(* CODESYS project Trike_PLC_Project.project
   Company: Schneider Electric
   Title: Compact / CANopen / HMI Controller SCU
   Description: ********Disclaimer Of Warranty********
      THE INFORMATION CONTAINED HEREIN IS PROVIDED "AS IS" WITHOUT WARRANTIES OF ANY KIND, EITHER EXPRESS OR IMPLIED, INCLUDING WITHOUT LIMITATION, ALL IMPLIED WARRANTIES OF MERCHANTABILITY, FITNESS FOR A PARTICULAR PURPOSE, NON-INFRINGEMENT OR OTHER VIOLATION OF RIGHTS. SCHNEIDER ELECTRIC DOES NOT WARRANT OR MAKE ANY REPRESENTATIONS REGARDING THE USE, VALIDITY, ACCURACY, OR RELIABILITY OF, OR THE RESULTS OF THE USE OF, OR OTHERWISE, RESPECTING THE MATERIALS, SPECIFICATIONS, CHARACTERISTICS OR OTHER INFORMATION SPECIFIED HEREIN. FURTHERMORE, ALL WARRANTIES, CONDITIONS, REPRESENTATIONS, INDEMNITIES AND GUARANTEES WITH RESPECT TO THE ACCURACY, OPERATION, CAPACITY, SPEED, FUNCTIONALITY, QUALIFICATIONS, OR CAPABILITIES OF THE SOFTWARE, SYSTEMS AND SERVICES COMPRISING OR UTILIZED IN THE COURSE OF APPLYING THIS INFORMATION, SPECIFICATIONS, OR MATERIALS, WHETHER EXPRESS OR IMPLIED, ARISING BY LAW, CUSTOM, PRIOR ORAL OR WRITTEN STATEMENTS BY SCHNEIDER ELECTRIC, OR OTHERWISE (INCLUDING, BUT NOT LIMITED TO ANY WARRANTY OF SATISFACTORY QUALITY, MERCHANTABILITY, FITNESS FOR PARTICULAR PURPOSE, TITLE AND NON-INFRINGEMENT) ARE HEREBY EXPRESSLY EXCLUDED AND DISCLAIMED:
      ********Disclaimer Of Liability*********
      UNDER NO CIRCUMSTANCES (INCLUDING NEGLIGENCE OR FORESEEABLE MISUSE) WILL SCHNEIDER ELECTRIC BE LIABLE FOR ANY DIRECT, INDIRECT, SPECIAL, INCIDENTAL, PUNITIVE OR CONSEQUENTIAL DAMAGES (INCLUDING WITHOUT LIMITATION, BUSINESS INTERRUPTION, DELAYS, LOSS OF DATA OR PROFIT) ARISING OUT OF THE APPLICATION OF THE INFORMATION, SPECIFICATIONS, CHARACTERISTICS OR MATERIALS CONTAINED HEREIN EVEN IF SCHNEIDER ELECTRIC HAS BEEN ADVISED OF THE POSSIBILITY OF SUCH DAMAGES.
      ************************************
      The information, program and configuration contained herein are provided as general training on the products concerned, in part, by way of theoretical and/or hypothetical examples.  Only you, the user, can be aware of all the conditions and factors present during setup, operation, and maintenance of your machine and its application; therefore, only you, the user, can determine the automation equipment and the related safeties and interlocks which can be properly used.  When selecting automation and control equipment and related software for a particular application, you must refer to the applicable local and national standards and regulations.
      ************************************
      Copyright © 2017 Schneider Electric. All rights reserved.
   Author: Machine Solutions
   Version: 4.3.0.0

Project tree, tasks and I/O mapping:
  HMISAC : HMISCUxA5, Schneider Electric, order no. HMISCUxA5, version 3.5.3.59
      settings: OpcUa Enable = False
    application Application
      libraries: MachineEnergyDashboard, 4.1.0.0 (Schneider Electric); Toolbox, 2.2.0.0 (Schneider Electric); SM3_Basic, 3.5.3.83 (3S - Smart Software Solutions GmbH)
      task MAST (cyclic, interval 20 ms, priority 15, watchdog 100 ms x 3) calls Preprocessing, Prg_Joystick6000, Prg_MicroCAN, Prg_Dunker_0A, Prg_Dunker_0B, Prg_Dunker_0C, Prg_Dunker_0D, Prg_Speedgoat, AlarmManager, MAIN, OutputMapping, Prg_WriteParameter
      global variables GVL_Retain
      LXM28A_Node03/
        global variables GVL_LXM28A_Node03
        program Prg_LXM28A_Node03 [CFC]: A02_Ctrl_Lexium, A01_GetNodeState
      program Preprocessing [CFC]: A04_DrvCmd_LXM28A_Node04, A05_DrvCmd_LXM32i_Node11, A03_DrvCmd_LXM28A_Node03
      global variables GVL
      global variables GVL_HmiVar
      LXM32i_Node11/
        global variables GVL_LXM32i_Node11
        program Prg_LXM32i_Node11 [CFC]: A02_Ctrl_Lexium, A01_GetNodeState
      program Prg_WriteParameter [ST]: A_WriteParameter_LXM2804, A_WriteParameter_LXM2803
      Symbols
      program MAIN [ST]: A02_CANopen_State, A04_Device_Error_State, A01_CANopen_Slave_State
      program OutputMapping [LD]
      program AlarmManager [CFC]: A06_Alarms_LXM32i_Node11, A05_Alarms_LXM28A_Node04, A01_Alarms_EStop, A04_Alarms_LXM28A_Node03
      global variables GVL_AlarmMsg
      LXM28A_Node04/
        global variables GVL_LXM28A_Node04
        program Prg_LXM28A_Node04 [CFC]: A01_GetNodeState, A02_Ctrl_Lexium
      Joystick_SD6000/
        program Prg_Joystick6000 [CFC]: A01_GetNodeState
        global variables GVL_Joystick6000
      MicroCAN4aiBOX/
        global variables GVL_MicroCAN
        program Prg_MicroCAN [CFC]: A01_GetNodeState
      Dunker_0A/
        global variables GVL_Dunker_0A
        program Prg_Dunker_0A [CFC]: A01_GetNodeState, A02_Ctrl_Dunker_0A
      Dunker_0B/
        global variables GVL_Dunker_0B
        program Prg_Dunker_0B [CFC]: A01_GetNodeState
      Dunker_0D/
        global variables GVL_Dunker_0D
        program Prg_Dunker_0D [CFC]: A01_GetNodeState
      Dunker_0C/
        global variables GVL_Dunker_0C
        program Prg_Dunker_0C [CFC]: A01_getNodeState
      Speedgoat/
        global variables GVL_Speedgoat
        program Prg_Speedgoat [CFC]: A01_GetNodeState
    HMI Application
    COM1
    Ethernet
    USB
      SoMachine_Network_Manager2 : SoMachine-Network Manager, Schneider Electric, version 4.0.0.2
    CAN
      CANopen_Optimized : CANopen Optimized, Schneider Electric, order no. 1806, version 3.0.1.24
          settings: Heartbeat in Milliseconds = 3000; Heartbeat Node ID = 1; Can Open Node ID = 1; ConfigVersion = 50659584
        LXM28A_Node04 : Lexium 28, Schneider Electric, order no. 0, version 1.4.2.0
            settings: General Options.Optional Device = TRUE; General Options.Not initialize = TRUE; General Options.Reset Node = TRUE; NODEIDSAVED = 23; SDO Timeout = 1000000; EXPERTSETTINGS = True; Emergency-General Parameters.Emergency COBID = 16#97; PDO 16#1400.COBID = 16#0217; PDO 16#1401.COBID = 16#0317; PDO 16#1402.COBID = 16#80000417; PDO 16#1403.COBID = 16#80000517; PDO 16#1800.COBID = 16#40000197; PDO 16#1801.COBID = 16#40000297; PDO 16#1801.Inhibit Time = 100; Generic COBID = '$NODEID+16#C0000280'; PDO 16#1802.COBID = 16#40000397; PDO 16#1802.Inhibit Time = 100; Generic COBID = '$NODEID+16#C0000380'; PDO 16#1803.COBID = 16#C0000497; Generic COBID = '$NODEID+16#C0000480'; driveModeCtrl.Subindex = 16#00; RefA16.Subindex = 16#00; RefB32.Subindex = 16#00; Controlword.Subindex = 16#00; Target Position.Subindex = 16#00; Controlword.Subindex = 16#00; Target Velocity.Subindex = 16#00; driveStat.Subindex = 16#00; mfStat.Subindex = 16#00; motionStat.Subindex = 16#00; driveInput.Subindex = 16#00; Statusword.Subindex = 16#00; Position Actual Value.Subindex = 16#00; Statusword.Subindex = 16#00; Velocity Actual Value.Subindex = 16#00; SDO List.Set Guardtime.Index = 16#100C; SDO List.Set Guardtime.Subindex = 16#00; SDO List.Set Guardtime.Value = 16#00000000; SDO List.Set Guardtime.Size = 16; SDO List.Set Guardtime.AbortIfError = FALSE;
              SDO List.Set Guardtime.JumpToLine = FALSE; SDO List.Set Guardtime.Line = 0; SDO List.Set Lifetime.Index = 16#100D; SDO List.Set Lifetime.Subindex = 16#00; SDO List.Set Lifetime.Value = 16#00000000; SDO List.Set Lifetime.Size = 8; SDO List.Set Lifetime.AbortIfError = FALSE; SDO List.Set Lifetime.JumpToLine = FALSE; SDO List.Set Lifetime.Line = 0; SDO List.Disable Emcy CobID.Index = 16#1014; SDO List.Disable Emcy CobID.Subindex = 16#00; SDO List.Disable Emcy CobID.Value = 16#80000097; SDO List.Disable Emcy CobID.Size = 32; SDO List.Disable Emcy CobID.AbortIfError = FALSE; SDO List.Disable Emcy CobID.JumpToLine = FALSE; SDO List.Disable Emcy CobID.Line = 0; SDO List.Set Emcy CobID.Index = 16#1014; SDO List.Set Emcy CobID.Subindex = 16#00; SDO List.Set Emcy CobID.Value = 16#00000097; SDO List.Set Emcy CobID.Size = 32; SDO List.Set Emcy CobID.AbortIfError = FALSE; SDO List.Set Emcy CobID.JumpToLine = FALSE; SDO List.Set Emcy CobID.Line = 0; SDO List.Set Heartbeat Consumer.Index = 16#1016; SDO List.Set Heartbeat Consumer.Subindex = 16#01; SDO List.Set Heartbeat Consumer.Value = 0; SDO List.Set Heartbeat Consumer.Size = 32; SDO List.Set Heartbeat Consumer.AbortIfError = FALSE; SDO List.Set Heartbeat Consumer.JumpToLine = FALSE; SDO List.Set Heartbeat Consumer.Line = 0; SDO List.Set Heartbeat Consumer.Index = 16#1016; SDO List.Set Heartbeat Consumer.Subindex = 16#02; SDO List.Set Heartbeat Consumer.Value = 0; SDO List.Set Heartbeat Consumer.Size = 32; SDO List.Set Heartbeat Consumer.AbortIfError = FALSE; SDO List.Set Heartbeat Consumer.JumpToLine = FALSE; SDO List.Set Heartbeat Consumer.Line = 0; SDO List.Set Heartbeat Consumer.Index = 16#1016; SDO List.Set Heartbeat Consumer.Subindex = 16#03; SDO List.Set Heartbeat Consumer.Value = 0;
              SDO List.Set Heartbeat Consumer.Size = 32; SDO List.Set Heartbeat Consumer.AbortIfError = FALSE; SDO List.Set Heartbeat Consumer.JumpToLine = FALSE; SDO List.Set Heartbeat Consumer.Line = 0; SDO List.Set Heartbeat Producer.Index = 16#1017; SDO List.Set Heartbeat Producer.Subindex = 16#00; SDO List.Set Heartbeat Producer.Value = 16#00000000; SDO List.Set Heartbeat Producer.Size = 16; SDO List.Set Heartbeat Producer.AbortIfError = FALSE; SDO List.Set Heartbeat Producer.JumpToLine = FALSE; SDO List.Set Heartbeat Producer.Line = 0; SDO List.Disable PDO.Index = 16#1400; SDO List.Disable PDO.Subindex = 16#01; SDO List.Disable PDO.Value = 16#80000217; SDO List.Disable PDO.Size = 32; SDO List.Disable PDO.AbortIfError = FALSE; SDO List.Disable PDO.JumpToLine = FALSE; SDO List.Disable PDO.Line = 0; SDO List.Set transmission type.Index = 16#1400; SDO List.Set transmission type.Subindex = 16#02; SDO List.Set transmission type.Value = 16#FF; SDO List.Set transmission type.Size = 8; SDO List.Set transmission type.AbortIfError = FALSE; SDO List.Set transmission type.JumpToLine = FALSE; SDO List.Set transmission type.Line = 0; SDO List.Clear pdo mapping.Index = 16#1600; SDO List.Clear pdo mapping.Subindex = 16#00; SDO List.Clear pdo mapping.Value = 16#0; SDO List.Clear pdo mapping.Size = 8; SDO List.Clear pdo mapping.AbortIfError = FALSE; SDO List.Clear pdo mapping.JumpToLine = FALSE; SDO List.Clear pdo mapping.Line = 0; SDO List.Set Mapping.Index = 16#1600; SDO List.Set Mapping.Subindex = 16#01; SDO List.Set Mapping.Value = 16#430C0010; SDO List.Set Mapping.Size = 32; SDO List.Set Mapping.AbortIfError = FALSE; SDO List.Set Mapping.JumpToLine = FALSE; SDO List.Set Mapping.Line = 0; SDO List.Set Mapping.Index = 16#1600;
              SDO List.Set Mapping.Subindex = 16#02; SDO List.Set Mapping.Value = 16#430D0010; SDO List.Set Mapping.Size = 32; SDO List.Set Mapping.AbortIfError = FALSE; SDO List.Set Mapping.JumpToLine = FALSE; SDO List.Set Mapping.Line = 0; SDO List.Set Mapping.Index = 16#1600; SDO List.Set Mapping.Subindex = 16#03; SDO List.Set Mapping.Value = 16#430E0020; SDO List.Set Mapping.Size = 32; SDO List.Set Mapping.AbortIfError = FALSE; SDO List.Set Mapping.JumpToLine = FALSE; SDO List.Set Mapping.Line = 0; SDO List.Set number of pdos.Index = 16#1600; SDO List.Set number of pdos.Subindex = 16#00; SDO List.Set number of pdos.Value = 16#03; SDO List.Set number of pdos.Size = 8; SDO List.Set number of pdos.AbortIfError = FALSE; SDO List.Set number of pdos.JumpToLine = FALSE; SDO List.Set number of pdos.Line = 0; SDO List.Set and enable COB-ID.Index = 16#1400; SDO List.Set and enable COB-ID.Subindex = 16#01; SDO List.Set and enable COB-ID.Value = 16#00000217; SDO List.Set and enable COB-ID.Size = 32; SDO List.Set and enable COB-ID.AbortIfError = FALSE; SDO List.Set and enable COB-ID.JumpToLine = FALSE; SDO List.Set and enable COB-ID.Line = 0; SDO List.Set transmission type.Index = 16#1401; SDO List.Set transmission type.Subindex = 16#02; SDO List.Set transmission type.Value = 16#FF; SDO List.Set transmission type.Size = 8; SDO List.Set transmission type.AbortIfError = FALSE; SDO List.Set transmission type.JumpToLine = FALSE; SDO List.Set transmission type.Line = 0; SDO List.Clear pdo mapping.Index = 16#1601; SDO List.Clear pdo mapping.Subindex = 16#00; SDO List.Clear pdo mapping.Value = 16#0; SDO List.Clear pdo mapping.Size = 8; SDO List.Clear pdo mapping.AbortIfError = FALSE; SDO List.Clear pdo mapping.JumpToLine = FALSE;
              SDO List.Clear pdo mapping.Line = 0; SDO List.Set Mapping.Index = 16#1601; SDO List.Set Mapping.Subindex = 16#01; SDO List.Set Mapping.Value = 16#60400010; SDO List.Set Mapping.Size = 32; SDO List.Set Mapping.AbortIfError = FALSE; SDO List.Set Mapping.JumpToLine = FALSE; SDO List.Set Mapping.Line = 0; SDO List.Set Mapping.Index = 16#1601; SDO List.Set Mapping.Subindex = 16#02; SDO List.Set Mapping.Value = 16#607A0020; SDO List.Set Mapping.Size = 32; SDO List.Set Mapping.AbortIfError = FALSE; SDO List.Set Mapping.JumpToLine = FALSE; SDO List.Set Mapping.Line = 0; SDO List.Set number of pdos.Index = 16#1601; SDO List.Set number of pdos.Subindex = 16#00; SDO List.Set number of pdos.Value = 16#02; SDO List.Set number of pdos.Size = 8; SDO List.Set number of pdos.AbortIfError = FALSE; SDO List.Set number of pdos.JumpToLine = FALSE; SDO List.Set number of pdos.Line = 0; SDO List.Set and enable COB-ID.Index = 16#1401; SDO List.Set and enable COB-ID.Subindex = 16#01; SDO List.Set and enable COB-ID.Value = 16#00000317; SDO List.Set and enable COB-ID.Size = 32; SDO List.Set and enable COB-ID.AbortIfError = FALSE; SDO List.Set and enable COB-ID.JumpToLine = FALSE; SDO List.Set and enable COB-ID.Line = 0; SDO List.Disable PDO.Index = 16#1800; SDO List.Disable PDO.Subindex = 16#01; SDO List.Disable PDO.Value = 16#C0000197; SDO List.Disable PDO.Size = 32; SDO List.Disable PDO.AbortIfError = FALSE; SDO List.Disable PDO.JumpToLine = FALSE; SDO List.Disable PDO.Line = 0; SDO List.Set transmission type.Index = 16#1800; SDO List.Set transmission type.Subindex = 16#02; SDO List.Set transmission type.Value = 16#FF; SDO List.Set transmission type.Size = 8;
              SDO List.Set transmission type.AbortIfError = FALSE; SDO List.Set transmission type.JumpToLine = FALSE; SDO List.Set transmission type.Line = 0; SDO List.Set inhibit time.Index = 16#1800; SDO List.Set inhibit time.Subindex = 16#03; SDO List.Set inhibit time.Value = 16#0064; SDO List.Set inhibit time.Size = 16; SDO List.Set inhibit time.AbortIfError = FALSE; SDO List.Set inhibit time.JumpToLine = FALSE; SDO List.Set inhibit time.Line = 0; SDO List.Set event time.Index = 16#1800; SDO List.Set event time.Subindex = 16#05; SDO List.Set event time.Value = 16#0000; SDO List.Set event time.Size = 16; SDO List.Set event time.AbortIfError = FALSE; SDO List.Set event time.JumpToLine = FALSE; SDO List.Set event time.Line = 0; SDO List.Clear pdo mapping.Index = 16#1A00; SDO List.Clear pdo mapping.Subindex = 16#00; SDO List.Clear pdo mapping.Value = 16#0; SDO List.Clear pdo mapping.Size = 8; SDO List.Clear pdo mapping.AbortIfError = FALSE; SDO List.Clear pdo mapping.JumpToLine = FALSE; SDO List.Clear pdo mapping.Line = 0; SDO List.Set Mapping.Index = 16#1A00; SDO List.Set Mapping.Subindex = 16#01; SDO List.Set Mapping.Value = 16#430F0010; SDO List.Set Mapping.Size = 32; SDO List.Set Mapping.AbortIfError = FALSE; SDO List.Set Mapping.JumpToLine = FALSE; SDO List.Set Mapping.Line = 0; SDO List.Set Mapping.Index = 16#1A00; SDO List.Set Mapping.Subindex = 16#02; SDO List.Set Mapping.Value = 16#43100010; SDO List.Set Mapping.Size = 32; SDO List.Set Mapping.AbortIfError = FALSE; SDO List.Set Mapping.JumpToLine = FALSE; SDO List.Set Mapping.Line = 0; SDO List.Set Mapping.Index = 16#1A00; SDO List.Set Mapping.Subindex = 16#03;
              SDO List.Set Mapping.Value = 16#43110010; SDO List.Set Mapping.Size = 32; SDO List.Set Mapping.AbortIfError = FALSE; SDO List.Set Mapping.JumpToLine = FALSE; SDO List.Set Mapping.Line = 0; SDO List.Set Mapping.Index = 16#1A00; SDO List.Set Mapping.Subindex = 16#04; SDO List.Set Mapping.Value = 16#430B0010; SDO List.Set Mapping.Size = 32; SDO List.Set Mapping.AbortIfError = FALSE; SDO List.Set Mapping.JumpToLine = FALSE; SDO List.Set Mapping.Line = 0; SDO List.Set number of pdos.Index = 16#1A00; SDO List.Set number of pdos.Subindex = 16#00; SDO List.Set number of pdos.Value = 16#04; SDO List.Set number of pdos.Size = 8; SDO List.Set number of pdos.AbortIfError = FALSE; SDO List.Set number of pdos.JumpToLine = FALSE; SDO List.Set number of pdos.Line = 0; SDO List.Set and enable COB-ID.Index = 16#1800; SDO List.Set and enable COB-ID.Subindex = 16#01; SDO List.Set and enable COB-ID.Value = 16#40000197; SDO List.Set and enable COB-ID.Size = 32; SDO List.Set and enable COB-ID.AbortIfError = FALSE; SDO List.Set and enable COB-ID.JumpToLine = FALSE; SDO List.Set and enable COB-ID.Line = 0; SDO List.Set transmission type.Index = 16#1801; SDO List.Set transmission type.Subindex = 16#02; SDO List.Set transmission type.Value = 16#FF; SDO List.Set transmission type.Size = 8; SDO List.Set transmission type.AbortIfError = FALSE; SDO List.Set transmission type.JumpToLine = FALSE; SDO List.Set transmission type.Line = 0; SDO List.Set inhibit time.Index = 16#1801; SDO List.Set inhibit time.Subindex = 16#03; SDO List.Set inhibit time.Value = 16#0064; SDO List.Set inhibit time.Size = 16; SDO List.Set inhibit time.AbortIfError = FALSE; SDO List.Set inhibit time.JumpToLine = FALSE; SDO List.Set inhibit time.Line = 0;
              SDO List.Set event time.Index = 16#1801; SDO List.Set event time.Subindex = 16#05; SDO List.Set event time.Value = 16#0064; SDO List.Set event time.Size = 16; SDO List.Set event time.AbortIfError = FALSE; SDO List.Set event time.JumpToLine = FALSE; SDO List.Set event time.Line = 0; SDO List.Clear pdo mapping.Index = 16#1A01; SDO List.Clear pdo mapping.Subindex = 16#00; SDO List.Clear pdo mapping.Value = 16#0; SDO List.Clear pdo mapping.Size = 8; SDO List.Clear pdo mapping.AbortIfError = FALSE; SDO List.Clear pdo mapping.JumpToLine = FALSE; SDO List.Clear pdo mapping.Line = 0; SDO List.Set Mapping.Index = 16#1A01; SDO List.Set Mapping.Subindex = 16#01; SDO List.Set Mapping.Value = 16#60410010; SDO List.Set Mapping.Size = 32; SDO List.Set Mapping.AbortIfError = FALSE; SDO List.Set Mapping.JumpToLine = FALSE; SDO List.Set Mapping.Line = 0; SDO List.Set Mapping.Index = 16#1A01; SDO List.Set Mapping.Subindex = 16#02; SDO List.Set Mapping.Value = 16#60640020; SDO List.Set Mapping.Size = 32; SDO List.Set Mapping.AbortIfError = FALSE; SDO List.Set Mapping.JumpToLine = FALSE; SDO List.Set Mapping.Line = 0; SDO List.Set number of pdos.Index = 16#1A01; SDO List.Set number of pdos.Subindex = 16#00; SDO List.Set number of pdos.Value = 16#02; SDO List.Set number of pdos.Size = 8; SDO List.Set number of pdos.AbortIfError = FALSE; SDO List.Set number of pdos.JumpToLine = FALSE; SDO List.Set number of pdos.Line = 0; SDO List.Set and enable COB-ID.Index = 16#1801; SDO List.Set and enable COB-ID.Subindex = 16#01; SDO List.Set and enable COB-ID.Value = 16#40000297; SDO List.Set and enable COB-ID.Size = 32; SDO List.Set and enable COB-ID.AbortIfError = FALSE;
              SDO List.Set and enable COB-ID.JumpToLine = FALSE; SDO List.Set and enable COB-ID.Line = 0; SDO List.Set transmission type.Index = 16#1802; SDO List.Set transmission type.Subindex = 16#02; SDO List.Set transmission type.Value = 16#FF; SDO List.Set transmission type.Size = 8; SDO List.Set transmission type.AbortIfError = FALSE; SDO List.Set transmission type.JumpToLine = FALSE; SDO List.Set transmission type.Line = 0; SDO List.Set inhibit time.Index = 16#1802; SDO List.Set inhibit time.Subindex = 16#03; SDO List.Set inhibit time.Value = 16#0064; SDO List.Set inhibit time.Size = 16; SDO List.Set inhibit time.AbortIfError = FALSE; SDO List.Set inhibit time.JumpToLine = FALSE; SDO List.Set inhibit time.Line = 0; SDO List.Set event time.Index = 16#1802; SDO List.Set event time.Subindex = 16#05; SDO List.Set event time.Value = 16#0064; SDO List.Set event time.Size = 16; SDO List.Set event time.AbortIfError = FALSE; SDO List.Set event time.JumpToLine = FALSE; SDO List.Set event time.Line = 0; SDO List.Clear pdo mapping.Index = 16#1A02; SDO List.Clear pdo mapping.Subindex = 16#00; SDO List.Clear pdo mapping.Value = 16#0; SDO List.Clear pdo mapping.Size = 8; SDO List.Clear pdo mapping.AbortIfError = FALSE; SDO List.Clear pdo mapping.JumpToLine = FALSE; SDO List.Clear pdo mapping.Line = 0; SDO List.Set Mapping.Index = 16#1A02; SDO List.Set Mapping.Subindex = 16#01; SDO List.Set Mapping.Value = 16#60410010; SDO List.Set Mapping.Size = 32; SDO List.Set Mapping.AbortIfError = FALSE; SDO List.Set Mapping.JumpToLine = FALSE; SDO List.Set Mapping.Line = 0; SDO List.Set Mapping.Index = 16#1A02; SDO List.Set Mapping.Subindex = 16#02; SDO List.Set Mapping.Value = 16#606C0020;
              SDO List.Set Mapping.Size = 32; SDO List.Set Mapping.AbortIfError = FALSE; SDO List.Set Mapping.JumpToLine = FALSE; SDO List.Set Mapping.Line = 0; SDO List.Set number of pdos.Index = 16#1A02; SDO List.Set number of pdos.Subindex = 16#00; SDO List.Set number of pdos.Value = 16#02; SDO List.Set number of pdos.Size = 8; SDO List.Set number of pdos.AbortIfError = FALSE; SDO List.Set number of pdos.JumpToLine = FALSE; SDO List.Set number of pdos.Line = 0; SDO List.Set and enable COB-ID.Index = 16#1802; SDO List.Set and enable COB-ID.Subindex = 16#01; SDO List.Set and enable COB-ID.Value = 16#40000397; SDO List.Set and enable COB-ID.Size = 32; SDO List.Set and enable COB-ID.AbortIfError = FALSE; SDO List.Set and enable COB-ID.JumpToLine = FALSE; SDO List.Set and enable COB-ID.Line = 0; SDO List.PLCopen Mode.Index = 16#430A; SDO List.PLCopen Mode.Subindex = 16#00; SDO List.PLCopen Mode.Value = 1; SDO List.PLCopen Mode.Size = 16; SDO List.PLCopen Mode.AbortIfError = FALSE; SDO List.PLCopen Mode.JumpToLine = FALSE; SDO List.PLCopen Mode.Line = 0; SDO List.PDO1 Event Mask.Index = 16#4312; SDO List.PDO1 Event Mask.Subindex = 16#00; SDO List.PDO1 Event Mask.Value = 15; SDO List.PDO1 Event Mask.Size = 16; SDO List.PDO1 Event Mask.AbortIfError = FALSE; SDO List.PDO1 Event Mask.JumpToLine = FALSE; SDO List.PDO1 Event Mask.Line = 0; SDO List.ReadyToSwitchOn automatically.Index = 16#4320; SDO List.ReadyToSwitchOn automatically.Subindex = 16#00; SDO List.ReadyToSwitchOn automatically.Value = 0; SDO List.ReadyToSwitchOn automatically.Size = 16; SDO List.ReadyToSwitchOn automatically.AbortIfError = FALSE; SDO List.ReadyToSwitchOn automatically.JumpToLine = FALSE; SDO List.ReadyToSwitchOn automatically.Line = 0; SDO List.Torque Slope Enable.Index = 16#450F;
              SDO List.Torque Slope Enable.Subindex = 16#00; SDO List.Torque Slope Enable.Value = 1; SDO List.Torque Slope Enable.Size = 16; SDO List.Torque Slope Enable.AbortIfError = FALSE; SDO List.Torque Slope Enable.JumpToLine = FALSE; SDO List.Torque Slope Enable.Line = 0; ConfigVersion = 50659584
            input  Application.GVL_LXM28A_Node04.diActlPos : DINT  // Position Actual Value
            input  Application.GVL_LXM28A_Node04.diActlVelo : DINT  // Velocity Actual Value
            unmapped channels: driveModeCtrl, RefA16, RefB32, Controlword, Target Position, driveStat, mfStat, motionStat, driveInput, Statusword, Statusword
        LXM28A_Node03 : Lexium 28, Schneider Electric, order no. 0, version 1.4.2.0
            settings: General Options.Optional Device = TRUE; General Options.Not initialize = TRUE; General Options.Reset Node = TRUE; NODEIDSAVED = 22; SDO Timeout = 1000000; EXPERTSETTINGS = True; Emergency-General Parameters.Emergency COBID = 16#96; PDO 16#1400.COBID = 16#0216; PDO 16#1401.COBID = 16#80000316; PDO 16#1402.COBID = 16#80000416; PDO 16#1403.COBID = 16#80000516; PDO 16#1800.COBID = 16#40000196; PDO 16#1801.COBID = 16#40000296; PDO 16#1801.Inhibit Time = 100; Generic COBID = '$NODEID+16#C0000280'; PDO 16#1802.COBID = 16#40000396; PDO 16#1802.Inhibit Time = 100; Generic COBID = '$NODEID+16#C0000380'; PDO 16#1803.COBID = 16#C0000496; Generic COBID = '$NODEID+16#C0000480'; driveModeCtrl.Subindex = 16#00; RefA16.Subindex = 16#00; RefB32.Subindex = 16#00; Controlword.Subindex = 16#00; Target Position.Subindex = 16#00; Controlword.Subindex = 16#00; Target Velocity.Subindex = 16#00; driveStat.Subindex = 16#00; mfStat.Subindex = 16#00; motionStat.Subindex = 16#00; driveInput.Subindex = 16#00; Statusword.Subindex = 16#00; Position Actual Value.Subindex = 16#00; Statusword.Subindex = 16#00; Velocity Actual Value.Subindex = 16#00; SDO List.Set Guardtime.Index = 16#100C; SDO List.Set Guardtime.Subindex = 16#00; SDO List.Set Guardtime.Value = 16#00000000; SDO List.Set Guardtime.Size = 16; SDO List.Set Guardtime.AbortIfError = FALSE;
              SDO List.Set Guardtime.JumpToLine = FALSE; SDO List.Set Guardtime.Line = 0; SDO List.Set Lifetime.Index = 16#100D; SDO List.Set Lifetime.Subindex = 16#00; SDO List.Set Lifetime.Value = 16#00000000; SDO List.Set Lifetime.Size = 8; SDO List.Set Lifetime.AbortIfError = FALSE; SDO List.Set Lifetime.JumpToLine = FALSE; SDO List.Set Lifetime.Line = 0; SDO List.Disable Emcy CobID.Index = 16#1014; SDO List.Disable Emcy CobID.Subindex = 16#00; SDO List.Disable Emcy CobID.Value = 16#80000096; SDO List.Disable Emcy CobID.Size = 32; SDO List.Disable Emcy CobID.AbortIfError = FALSE; SDO List.Disable Emcy CobID.JumpToLine = FALSE; SDO List.Disable Emcy CobID.Line = 0; SDO List.Set Emcy CobID.Index = 16#1014; SDO List.Set Emcy CobID.Subindex = 16#00; SDO List.Set Emcy CobID.Value = 16#00000096; SDO List.Set Emcy CobID.Size = 32; SDO List.Set Emcy CobID.AbortIfError = FALSE; SDO List.Set Emcy CobID.JumpToLine = FALSE; SDO List.Set Emcy CobID.Line = 0; SDO List.Set Heartbeat Consumer.Index = 16#1016; SDO List.Set Heartbeat Consumer.Subindex = 16#01; SDO List.Set Heartbeat Consumer.Value = 0; SDO List.Set Heartbeat Consumer.Size = 32; SDO List.Set Heartbeat Consumer.AbortIfError = FALSE; SDO List.Set Heartbeat Consumer.JumpToLine = FALSE; SDO List.Set Heartbeat Consumer.Line = 0; SDO List.Set Heartbeat Consumer.Index = 16#1016; SDO List.Set Heartbeat Consumer.Subindex = 16#02; SDO List.Set Heartbeat Consumer.Value = 0; SDO List.Set Heartbeat Consumer.Size = 32; SDO List.Set Heartbeat Consumer.AbortIfError = FALSE; SDO List.Set Heartbeat Consumer.JumpToLine = FALSE; SDO List.Set Heartbeat Consumer.Line = 0; SDO List.Set Heartbeat Consumer.Index = 16#1016; SDO List.Set Heartbeat Consumer.Subindex = 16#03; SDO List.Set Heartbeat Consumer.Value = 0;
              SDO List.Set Heartbeat Consumer.Size = 32; SDO List.Set Heartbeat Consumer.AbortIfError = FALSE; SDO List.Set Heartbeat Consumer.JumpToLine = FALSE; SDO List.Set Heartbeat Consumer.Line = 0; SDO List.Set Heartbeat Producer.Index = 16#1017; SDO List.Set Heartbeat Producer.Subindex = 16#00; SDO List.Set Heartbeat Producer.Value = 16#00000000; SDO List.Set Heartbeat Producer.Size = 16; SDO List.Set Heartbeat Producer.AbortIfError = FALSE; SDO List.Set Heartbeat Producer.JumpToLine = FALSE; SDO List.Set Heartbeat Producer.Line = 0; SDO List.Disable PDO.Index = 16#1400; SDO List.Disable PDO.Subindex = 16#01; SDO List.Disable PDO.Value = 16#80000216; SDO List.Disable PDO.Size = 32; SDO List.Disable PDO.AbortIfError = FALSE; SDO List.Disable PDO.JumpToLine = FALSE; SDO List.Disable PDO.Line = 0; SDO List.Set transmission type.Index = 16#1400; SDO List.Set transmission type.Subindex = 16#02; SDO List.Set transmission type.Value = 16#FF; SDO List.Set transmission type.Size = 8; SDO List.Set transmission type.AbortIfError = FALSE; SDO List.Set transmission type.JumpToLine = FALSE; SDO List.Set transmission type.Line = 0; SDO List.Clear pdo mapping.Index = 16#1600; SDO List.Clear pdo mapping.Subindex = 16#00; SDO List.Clear pdo mapping.Value = 16#0; SDO List.Clear pdo mapping.Size = 8; SDO List.Clear pdo mapping.AbortIfError = FALSE; SDO List.Clear pdo mapping.JumpToLine = FALSE; SDO List.Clear pdo mapping.Line = 0; SDO List.Set Mapping.Index = 16#1600; SDO List.Set Mapping.Subindex = 16#01; SDO List.Set Mapping.Value = 16#430C0010; SDO List.Set Mapping.Size = 32; SDO List.Set Mapping.AbortIfError = FALSE; SDO List.Set Mapping.JumpToLine = FALSE; SDO List.Set Mapping.Line = 0; SDO List.Set Mapping.Index = 16#1600;
              SDO List.Set Mapping.Subindex = 16#02; SDO List.Set Mapping.Value = 16#430D0010; SDO List.Set Mapping.Size = 32; SDO List.Set Mapping.AbortIfError = FALSE; SDO List.Set Mapping.JumpToLine = FALSE; SDO List.Set Mapping.Line = 0; SDO List.Set Mapping.Index = 16#1600; SDO List.Set Mapping.Subindex = 16#03; SDO List.Set Mapping.Value = 16#430E0020; SDO List.Set Mapping.Size = 32; SDO List.Set Mapping.AbortIfError = FALSE; SDO List.Set Mapping.JumpToLine = FALSE; SDO List.Set Mapping.Line = 0; SDO List.Set number of pdos.Index = 16#1600; SDO List.Set number of pdos.Subindex = 16#00; SDO List.Set number of pdos.Value = 16#03; SDO List.Set number of pdos.Size = 8; SDO List.Set number of pdos.AbortIfError = FALSE; SDO List.Set number of pdos.JumpToLine = FALSE; SDO List.Set number of pdos.Line = 0; SDO List.Set and enable COB-ID.Index = 16#1400; SDO List.Set and enable COB-ID.Subindex = 16#01; SDO List.Set and enable COB-ID.Value = 16#00000216; SDO List.Set and enable COB-ID.Size = 32; SDO List.Set and enable COB-ID.AbortIfError = FALSE; SDO List.Set and enable COB-ID.JumpToLine = FALSE; SDO List.Set and enable COB-ID.Line = 0; SDO List.Disable PDO.Index = 16#1800; SDO List.Disable PDO.Subindex = 16#01; SDO List.Disable PDO.Value = 16#C0000196; SDO List.Disable PDO.Size = 32; SDO List.Disable PDO.AbortIfError = FALSE; SDO List.Disable PDO.JumpToLine = FALSE; SDO List.Disable PDO.Line = 0; SDO List.Set transmission type.Index = 16#1800; SDO List.Set transmission type.Subindex = 16#02; SDO List.Set transmission type.Value = 16#FF; SDO List.Set transmission type.Size = 8; SDO List.Set transmission type.AbortIfError = FALSE; SDO List.Set transmission type.JumpToLine = FALSE;
              SDO List.Set transmission type.Line = 0; SDO List.Set inhibit time.Index = 16#1800; SDO List.Set inhibit time.Subindex = 16#03; SDO List.Set inhibit time.Value = 16#0064; SDO List.Set inhibit time.Size = 16; SDO List.Set inhibit time.AbortIfError = FALSE; SDO List.Set inhibit time.JumpToLine = FALSE; SDO List.Set inhibit time.Line = 0; SDO List.Set event time.Index = 16#1800; SDO List.Set event time.Subindex = 16#05; SDO List.Set event time.Value = 16#0000; SDO List.Set event time.Size = 16; SDO List.Set event time.AbortIfError = FALSE; SDO List.Set event time.JumpToLine = FALSE; SDO List.Set event time.Line = 0; SDO List.Clear pdo mapping.Index = 16#1A00; SDO List.Clear pdo mapping.Subindex = 16#00; SDO List.Clear pdo mapping.Value = 16#0; SDO List.Clear pdo mapping.Size = 8; SDO List.Clear pdo mapping.AbortIfError = FALSE; SDO List.Clear pdo mapping.JumpToLine = FALSE; SDO List.Clear pdo mapping.Line = 0; SDO List.Set Mapping.Index = 16#1A00; SDO List.Set Mapping.Subindex = 16#01; SDO List.Set Mapping.Value = 16#430F0010; SDO List.Set Mapping.Size = 32; SDO List.Set Mapping.AbortIfError = FALSE; SDO List.Set Mapping.JumpToLine = FALSE; SDO List.Set Mapping.Line = 0; SDO List.Set Mapping.Index = 16#1A00; SDO List.Set Mapping.Subindex = 16#02; SDO List.Set Mapping.Value = 16#43100010; SDO List.Set Mapping.Size = 32; SDO List.Set Mapping.AbortIfError = FALSE; SDO List.Set Mapping.JumpToLine = FALSE; SDO List.Set Mapping.Line = 0; SDO List.Set Mapping.Index = 16#1A00; SDO List.Set Mapping.Subindex = 16#03; SDO List.Set Mapping.Value = 16#43110010; SDO List.Set Mapping.Size = 32;
              SDO List.Set Mapping.AbortIfError = FALSE; SDO List.Set Mapping.JumpToLine = FALSE; SDO List.Set Mapping.Line = 0; SDO List.Set Mapping.Index = 16#1A00; SDO List.Set Mapping.Subindex = 16#04; SDO List.Set Mapping.Value = 16#430B0010; SDO List.Set Mapping.Size = 32; SDO List.Set Mapping.AbortIfError = FALSE; SDO List.Set Mapping.JumpToLine = FALSE; SDO List.Set Mapping.Line = 0; SDO List.Set number of pdos.Index = 16#1A00; SDO List.Set number of pdos.Subindex = 16#00; SDO List.Set number of pdos.Value = 16#04; SDO List.Set number of pdos.Size = 8; SDO List.Set number of pdos.AbortIfError = FALSE; SDO List.Set number of pdos.JumpToLine = FALSE; SDO List.Set number of pdos.Line = 0; SDO List.Set and enable COB-ID.Index = 16#1800; SDO List.Set and enable COB-ID.Subindex = 16#01; SDO List.Set and enable COB-ID.Value = 16#40000196; SDO List.Set and enable COB-ID.Size = 32; SDO List.Set and enable COB-ID.AbortIfError = FALSE; SDO List.Set and enable COB-ID.JumpToLine = FALSE; SDO List.Set and enable COB-ID.Line = 0; SDO List.Set transmission type.Index = 16#1801; SDO List.Set transmission type.Subindex = 16#02; SDO List.Set transmission type.Value = 16#FF; SDO List.Set transmission type.Size = 8; SDO List.Set transmission type.AbortIfError = FALSE; SDO List.Set transmission type.JumpToLine = FALSE; SDO List.Set transmission type.Line = 0; SDO List.Set inhibit time.Index = 16#1801; SDO List.Set inhibit time.Subindex = 16#03; SDO List.Set inhibit time.Value = 16#0064; SDO List.Set inhibit time.Size = 16; SDO List.Set inhibit time.AbortIfError = FALSE; SDO List.Set inhibit time.JumpToLine = FALSE; SDO List.Set inhibit time.Line = 0; SDO List.Set event time.Index = 16#1801; SDO List.Set event time.Subindex = 16#05;
              SDO List.Set event time.Value = 16#0064; SDO List.Set event time.Size = 16; SDO List.Set event time.AbortIfError = FALSE; SDO List.Set event time.JumpToLine = FALSE; SDO List.Set event time.Line = 0; SDO List.Clear pdo mapping.Index = 16#1A01; SDO List.Clear pdo mapping.Subindex = 16#00; SDO List.Clear pdo mapping.Value = 16#0; SDO List.Clear pdo mapping.Size = 8; SDO List.Clear pdo mapping.AbortIfError = FALSE; SDO List.Clear pdo mapping.JumpToLine = FALSE; SDO List.Clear pdo mapping.Line = 0; SDO List.Set Mapping.Index = 16#1A01; SDO List.Set Mapping.Subindex = 16#01; SDO List.Set Mapping.Value = 16#60410010; SDO List.Set Mapping.Size = 32; SDO List.Set Mapping.AbortIfError = FALSE; SDO List.Set Mapping.JumpToLine = FALSE; SDO List.Set Mapping.Line = 0; SDO List.Set Mapping.Index = 16#1A01; SDO List.Set Mapping.Subindex = 16#02; SDO List.Set Mapping.Value = 16#60640020; SDO List.Set Mapping.Size = 32; SDO List.Set Mapping.AbortIfError = FALSE; SDO List.Set Mapping.JumpToLine = FALSE; SDO List.Set Mapping.Line = 0; SDO List.Set number of pdos.Index = 16#1A01; SDO List.Set number of pdos.Subindex = 16#00; SDO List.Set number of pdos.Value = 16#02; SDO List.Set number of pdos.Size = 8; SDO List.Set number of pdos.AbortIfError = FALSE; SDO List.Set number of pdos.JumpToLine = FALSE; SDO List.Set number of pdos.Line = 0; SDO List.Set and enable COB-ID.Index = 16#1801; SDO List.Set and enable COB-ID.Subindex = 16#01; SDO List.Set and enable COB-ID.Value = 16#40000296; SDO List.Set and enable COB-ID.Size = 32; SDO List.Set and enable COB-ID.AbortIfError = FALSE; SDO List.Set and enable COB-ID.JumpToLine = FALSE; SDO List.Set and enable COB-ID.Line = 0;
              SDO List.Set transmission type.Index = 16#1802; SDO List.Set transmission type.Subindex = 16#02; SDO List.Set transmission type.Value = 16#FF; SDO List.Set transmission type.Size = 8; SDO List.Set transmission type.AbortIfError = FALSE; SDO List.Set transmission type.JumpToLine = FALSE; SDO List.Set transmission type.Line = 0; SDO List.Set inhibit time.Index = 16#1802; SDO List.Set inhibit time.Subindex = 16#03; SDO List.Set inhibit time.Value = 16#0064; SDO List.Set inhibit time.Size = 16; SDO List.Set inhibit time.AbortIfError = FALSE; SDO List.Set inhibit time.JumpToLine = FALSE; SDO List.Set inhibit time.Line = 0; SDO List.Set event time.Index = 16#1802; SDO List.Set event time.Subindex = 16#05; SDO List.Set event time.Value = 16#0064; SDO List.Set event time.Size = 16; SDO List.Set event time.AbortIfError = FALSE; SDO List.Set event time.JumpToLine = FALSE; SDO List.Set event time.Line = 0; SDO List.Clear pdo mapping.Index = 16#1A02; SDO List.Clear pdo mapping.Subindex = 16#00; SDO List.Clear pdo mapping.Value = 16#0; SDO List.Clear pdo mapping.Size = 8; SDO List.Clear pdo mapping.AbortIfError = FALSE; SDO List.Clear pdo mapping.JumpToLine = FALSE; SDO List.Clear pdo mapping.Line = 0; SDO List.Set Mapping.Index = 16#1A02; SDO List.Set Mapping.Subindex = 16#01; SDO List.Set Mapping.Value = 16#60410010; SDO List.Set Mapping.Size = 32; SDO List.Set Mapping.AbortIfError = FALSE; SDO List.Set Mapping.JumpToLine = FALSE; SDO List.Set Mapping.Line = 0; SDO List.Set Mapping.Index = 16#1A02; SDO List.Set Mapping.Subindex = 16#02; SDO List.Set Mapping.Value = 16#606C0020; SDO List.Set Mapping.Size = 32; SDO List.Set Mapping.AbortIfError = FALSE;
              SDO List.Set Mapping.JumpToLine = FALSE; SDO List.Set Mapping.Line = 0; SDO List.Set number of pdos.Index = 16#1A02; SDO List.Set number of pdos.Subindex = 16#00; SDO List.Set number of pdos.Value = 16#02; SDO List.Set number of pdos.Size = 8; SDO List.Set number of pdos.AbortIfError = FALSE; SDO List.Set number of pdos.JumpToLine = FALSE; SDO List.Set number of pdos.Line = 0; SDO List.Set and enable COB-ID.Index = 16#1802; SDO List.Set and enable COB-ID.Subindex = 16#01; SDO List.Set and enable COB-ID.Value = 16#40000396; SDO List.Set and enable COB-ID.Size = 32; SDO List.Set and enable COB-ID.AbortIfError = FALSE; SDO List.Set and enable COB-ID.JumpToLine = FALSE; SDO List.Set and enable COB-ID.Line = 0; SDO List.PLCopen Mode.Index = 16#430A; SDO List.PLCopen Mode.Subindex = 16#00; SDO List.PLCopen Mode.Value = 1; SDO List.PLCopen Mode.Size = 16; SDO List.PLCopen Mode.AbortIfError = FALSE; SDO List.PLCopen Mode.JumpToLine = FALSE; SDO List.PLCopen Mode.Line = 0; SDO List.PDO1 Event Mask.Index = 16#4312; SDO List.PDO1 Event Mask.Subindex = 16#00; SDO List.PDO1 Event Mask.Value = 15; SDO List.PDO1 Event Mask.Size = 16; SDO List.PDO1 Event Mask.AbortIfError = FALSE; SDO List.PDO1 Event Mask.JumpToLine = FALSE; SDO List.PDO1 Event Mask.Line = 0; SDO List.ReadyToSwitchOn automatically.Index = 16#4320; SDO List.ReadyToSwitchOn automatically.Subindex = 16#00; SDO List.ReadyToSwitchOn automatically.Value = 0; SDO List.ReadyToSwitchOn automatically.Size = 16; SDO List.ReadyToSwitchOn automatically.AbortIfError = FALSE; SDO List.ReadyToSwitchOn automatically.JumpToLine = FALSE; SDO List.ReadyToSwitchOn automatically.Line = 0; SDO List.Torque Slope Enable.Index = 16#450F; SDO List.Torque Slope Enable.Subindex = 16#00; SDO List.Torque Slope Enable.Value = 1;
              SDO List.Torque Slope Enable.Size = 16; SDO List.Torque Slope Enable.AbortIfError = FALSE; SDO List.Torque Slope Enable.JumpToLine = FALSE; SDO List.Torque Slope Enable.Line = 0; ConfigVersion = 50659584
            input  Application.GVL_LXM28A_Node03.diActlPos : DINT  // Position Actual Value
            input  Application.GVL_LXM28A_Node03.diActlVelo : DINT  // Velocity Actual Value
            unmapped channels: driveModeCtrl, RefA16, RefB32, driveStat, mfStat, motionStat, driveInput, Statusword, Statusword
        LXM32i_Node11 : Lexium 32 i, Schneider Electric, order no. 93800, version 1.2.6.0
            settings: General Options.Optional Device = TRUE; General Options.Not initialize = TRUE; NODEIDSAVED = 21; SDO Timeout = 1000000; Explicit Deactivate PDOs = FALSE; EXPERTSETTINGS = True; Emergency-General Parameters.Emergency COBID = 16#95; PDO 16#1400.COBID = 16#0215; PDO 16#1401.COBID = 16#80000315; PDO 16#1402.COBID = 16#80000415; PDO 16#1403.COBID = 16#80000515; PDO 16#1800.COBID = 16#40000195; PDO 16#1801.COBID = 16#40000295; PDO 16#1801.Inhibit Time = 100; Generic COBID = '$NODEID+16#C0000280'; PDO 16#1802.COBID = 16#40000395; PDO 16#1802.Inhibit Time = 100; Generic COBID = '$NODEID+16#C0000380'; PDO 16#1803.COBID = 16#C0000495; Generic COBID = '$NODEID+16#C0000480'; Controlword.Subindex = 16#00; Target position.Subindex = 16#00; Controlword.Subindex = 16#00; Target velocity.Subindex = 16#00; Statusword.Subindex = 16#00; Position actual value.Subindex = 16#00; Statusword.Subindex = 16#00; Velocity actual value.Subindex = 16#00; SDO List.Set Guardtime.Index = 16#100C; SDO List.Set Guardtime.Subindex = 16#00; SDO List.Set Guardtime.Value = 16#00000000; SDO List.Set Guardtime.Size = 16; SDO List.Set Guardtime.AbortIfError = FALSE; SDO List.Set Guardtime.JumpToLine = FALSE; SDO List.Set Guardtime.Line = 0; SDO List.Set Lifetime.Index = 16#100D; SDO List.Set Lifetime.Subindex = 16#00; SDO List.Set Lifetime.Value = 16#00000000; SDO List.Set Lifetime.Size = 8; SDO List.Set Lifetime.AbortIfError = FALSE;
              SDO List.Set Lifetime.JumpToLine = FALSE; SDO List.Set Lifetime.Line = 0; SDO List.Disable Emcy CobID.Index = 16#1014; SDO List.Disable Emcy CobID.Subindex = 16#00; SDO List.Disable Emcy CobID.Value = 16#80000095; SDO List.Disable Emcy CobID.Size = 32; SDO List.Disable Emcy CobID.AbortIfError = FALSE; SDO List.Disable Emcy CobID.JumpToLine = FALSE; SDO List.Disable Emcy CobID.Line = 0; SDO List.Set Emcy CobID.Index = 16#1014; SDO List.Set Emcy CobID.Subindex = 16#00; SDO List.Set Emcy CobID.Value = 16#00000095; SDO List.Set Emcy CobID.Size = 32; SDO List.Set Emcy CobID.AbortIfError = FALSE; SDO List.Set Emcy CobID.JumpToLine = FALSE; SDO List.Set Emcy CobID.Line = 0; SDO List.Set Heartbeat Consumer.Index = 16#1016; SDO List.Set Heartbeat Consumer.Subindex = 16#01; SDO List.Set Heartbeat Consumer.Value = 0; SDO List.Set Heartbeat Consumer.Size = 32; SDO List.Set Heartbeat Consumer.AbortIfError = FALSE; SDO List.Set Heartbeat Consumer.JumpToLine = FALSE; SDO List.Set Heartbeat Consumer.Line = 0; SDO List.Set Heartbeat Consumer.Index = 16#1016; SDO List.Set Heartbeat Consumer.Subindex = 16#02; SDO List.Set Heartbeat Consumer.Value = 0; SDO List.Set Heartbeat Consumer.Size = 32; SDO List.Set Heartbeat Consumer.AbortIfError = FALSE; SDO List.Set Heartbeat Consumer.JumpToLine = FALSE; SDO List.Set Heartbeat Consumer.Line = 0; SDO List.Set Heartbeat Consumer.Index = 16#1016; SDO List.Set Heartbeat Consumer.Subindex = 16#03; SDO List.Set Heartbeat Consumer.Value = 0; SDO List.Set Heartbeat Consumer.Size = 32; SDO List.Set Heartbeat Consumer.AbortIfError = FALSE; SDO List.Set Heartbeat Consumer.JumpToLine = FALSE; SDO List.Set Heartbeat Consumer.Line = 0; SDO List.Set Heartbeat Producer.Index = 16#1017; SDO List.Set Heartbeat Producer.Subindex = 16#00; SDO List.Set Heartbeat Producer.Value = 16#00000000;
              SDO List.Set Heartbeat Producer.Size = 16; SDO List.Set Heartbeat Producer.AbortIfError = FALSE; SDO List.Set Heartbeat Producer.JumpToLine = FALSE; SDO List.Set Heartbeat Producer.Line = 0; SDO List.Disable PDO.Index = 16#1400; SDO List.Disable PDO.Subindex = 16#01; SDO List.Disable PDO.Value = 16#80000215; SDO List.Disable PDO.Size = 32; SDO List.Disable PDO.AbortIfError = FALSE; SDO List.Disable PDO.JumpToLine = FALSE; SDO List.Disable PDO.Line = 0; SDO List.Set transmission type.Index = 16#1400; SDO List.Set transmission type.Subindex = 16#02; SDO List.Set transmission type.Value = 16#FF; SDO List.Set transmission type.Size = 8; SDO List.Set transmission type.AbortIfError = FALSE; SDO List.Set transmission type.JumpToLine = FALSE; SDO List.Set transmission type.Line = 0; SDO List.Clear pdo mapping.Index = 16#1600; SDO List.Clear pdo mapping.Subindex = 16#00; SDO List.Clear pdo mapping.Value = 16#0; SDO List.Clear pdo mapping.Size = 8; SDO List.Clear pdo mapping.AbortIfError = FALSE; SDO List.Clear pdo mapping.JumpToLine = FALSE; SDO List.Clear pdo mapping.Line = 0; SDO List.Set Mapping.Index = 16#1600; SDO List.Set Mapping.Subindex = 16#01; SDO List.Set Mapping.Value = 16#301B1F10; SDO List.Set Mapping.Size = 32; SDO List.Set Mapping.AbortIfError = FALSE; SDO List.Set Mapping.JumpToLine = FALSE; SDO List.Set Mapping.Line = 0; SDO List.Set Mapping.Index = 16#1600; SDO List.Set Mapping.Subindex = 16#02; SDO List.Set Mapping.Value = 16#301B2210; SDO List.Set Mapping.Size = 32; SDO List.Set Mapping.AbortIfError = FALSE; SDO List.Set Mapping.JumpToLine = FALSE; SDO List.Set Mapping.Line = 0; SDO List.Set Mapping.Index = 16#1600;
              SDO List.Set Mapping.Subindex = 16#03; SDO List.Set Mapping.Value = 16#301B2120; SDO List.Set Mapping.Size = 32; SDO List.Set Mapping.AbortIfError = FALSE; SDO List.Set Mapping.JumpToLine = FALSE; SDO List.Set Mapping.Line = 0; SDO List.Set number of pdos.Index = 16#1600; SDO List.Set number of pdos.Subindex = 16#00; SDO List.Set number of pdos.Value = 16#03; SDO List.Set number of pdos.Size = 8; SDO List.Set number of pdos.AbortIfError = FALSE; SDO List.Set number of pdos.JumpToLine = FALSE; SDO List.Set number of pdos.Line = 0; SDO List.Set and enable COB-ID.Index = 16#1400; SDO List.Set and enable COB-ID.Subindex = 16#01; SDO List.Set and enable COB-ID.Value = 16#00000215; SDO List.Set and enable COB-ID.Size = 32; SDO List.Set and enable COB-ID.AbortIfError = FALSE; SDO List.Set and enable COB-ID.JumpToLine = FALSE; SDO List.Set and enable COB-ID.Line = 0; SDO List.Disable PDO.Index = 16#1401; SDO List.Disable PDO.Subindex = 16#01; SDO List.Disable PDO.Value = 16#80000315; SDO List.Disable PDO.Size = 32; SDO List.Disable PDO.AbortIfError = FALSE; SDO List.Disable PDO.JumpToLine = FALSE; SDO List.Disable PDO.Line = 0; SDO List.Disable PDO.Index = 16#1402; SDO List.Disable PDO.Subindex = 16#01; SDO List.Disable PDO.Value = 16#80000415; SDO List.Disable PDO.Size = 32; SDO List.Disable PDO.AbortIfError = FALSE; SDO List.Disable PDO.JumpToLine = FALSE; SDO List.Disable PDO.Line = 0; SDO List.Disable PDO.Index = 16#1403; SDO List.Disable PDO.Subindex = 16#01; SDO List.Disable PDO.Value = 16#80000515; SDO List.Disable PDO.Size = 32; SDO List.Disable PDO.AbortIfError = FALSE; SDO List.Disable PDO.JumpToLine = FALSE;
              SDO List.Disable PDO.Line = 0; SDO List.Disable PDO.Index = 16#1800; SDO List.Disable PDO.Subindex = 16#01; SDO List.Disable PDO.Value = 16#C0000195; SDO List.Disable PDO.Size = 32; SDO List.Disable PDO.AbortIfError = FALSE; SDO List.Disable PDO.JumpToLine = FALSE; SDO List.Disable PDO.Line = 0; SDO List.Set transmission type.Index = 16#1800; SDO List.Set transmission type.Subindex = 16#02; SDO List.Set transmission type.Value = 16#FF; SDO List.Set transmission type.Size = 8; SDO List.Set transmission type.AbortIfError = FALSE; SDO List.Set transmission type.JumpToLine = FALSE; SDO List.Set transmission type.Line = 0; SDO List.Set inhibit time.Index = 16#1800; SDO List.Set inhibit time.Subindex = 16#03; SDO List.Set inhibit time.Value = 16#0064; SDO List.Set inhibit time.Size = 16; SDO List.Set inhibit time.AbortIfError = FALSE; SDO List.Set inhibit time.JumpToLine = FALSE; SDO List.Set inhibit time.Line = 0; SDO List.Set event time.Index = 16#1800; SDO List.Set event time.Subindex = 16#05; SDO List.Set event time.Value = 16#0000; SDO List.Set event time.Size = 16; SDO List.Set event time.AbortIfError = FALSE; SDO List.Set event time.JumpToLine = FALSE; SDO List.Set event time.Line = 0; SDO List.Clear pdo mapping.Index = 16#1A00; SDO List.Clear pdo mapping.Subindex = 16#00; SDO List.Clear pdo mapping.Value = 16#0; SDO List.Clear pdo mapping.Size = 8; SDO List.Clear pdo mapping.AbortIfError = FALSE; SDO List.Clear pdo mapping.JumpToLine = FALSE; SDO List.Clear pdo mapping.Line = 0; SDO List.Set Mapping.Index = 16#1A00; SDO List.Set Mapping.Subindex = 16#01; SDO List.Set Mapping.Value = 16#301B2510; SDO List.Set Mapping.Size = 32;
              SDO List.Set Mapping.AbortIfError = FALSE; SDO List.Set Mapping.JumpToLine = FALSE; SDO List.Set Mapping.Line = 0; SDO List.Set Mapping.Index = 16#1A00; SDO List.Set Mapping.Subindex = 16#02; SDO List.Set Mapping.Value = 16#301B2610; SDO List.Set Mapping.Size = 32; SDO List.Set Mapping.AbortIfError = FALSE; SDO List.Set Mapping.JumpToLine = FALSE; SDO List.Set Mapping.Line = 0; SDO List.Set Mapping.Index = 16#1A00; SDO List.Set Mapping.Subindex = 16#03; SDO List.Set Mapping.Value = 16#301B2710; SDO List.Set Mapping.Size = 32; SDO List.Set Mapping.AbortIfError = FALSE; SDO List.Set Mapping.JumpToLine = FALSE; SDO List.Set Mapping.Line = 0; SDO List.Set Mapping.Index = 16#1A00; SDO List.Set Mapping.Subindex = 16#04; SDO List.Set Mapping.Value = 16#301B2810; SDO List.Set Mapping.Size = 32; SDO List.Set Mapping.AbortIfError = FALSE; SDO List.Set Mapping.JumpToLine = FALSE; SDO List.Set Mapping.Line = 0; SDO List.Set number of pdos.Index = 16#1A00; SDO List.Set number of pdos.Subindex = 16#00; SDO List.Set number of pdos.Value = 16#04; SDO List.Set number of pdos.Size = 8; SDO List.Set number of pdos.AbortIfError = FALSE; SDO List.Set number of pdos.JumpToLine = FALSE; SDO List.Set number of pdos.Line = 0; SDO List.Set and enable COB-ID.Index = 16#1800; SDO List.Set and enable COB-ID.Subindex = 16#01; SDO List.Set and enable COB-ID.Value = 16#40000195; SDO List.Set and enable COB-ID.Size = 32; SDO List.Set and enable COB-ID.AbortIfError = FALSE; SDO List.Set and enable COB-ID.JumpToLine = FALSE; SDO List.Set and enable COB-ID.Line = 0; SDO List.Disable PDO.Index = 16#1801; SDO List.Disable PDO.Subindex = 16#01;
              SDO List.Disable PDO.Value = 16#C0000295; SDO List.Disable PDO.Size = 32; SDO List.Disable PDO.AbortIfError = FALSE; SDO List.Disable PDO.JumpToLine = FALSE; SDO List.Disable PDO.Line = 0; SDO List.Set transmission type.Index = 16#1801; SDO List.Set transmission type.Subindex = 16#02; SDO List.Set transmission type.Value = 16#FF; SDO List.Set transmission type.Size = 8; SDO List.Set transmission type.AbortIfError = FALSE; SDO List.Set transmission type.JumpToLine = FALSE; SDO List.Set transmission type.Line = 0; SDO List.Set inhibit time.Index = 16#1801; SDO List.Set inhibit time.Subindex = 16#03; SDO List.Set inhibit time.Value = 16#0064; SDO List.Set inhibit time.Size = 16; SDO List.Set inhibit time.AbortIfError = FALSE; SDO List.Set inhibit time.JumpToLine = FALSE; SDO List.Set inhibit time.Line = 0; SDO List.Set event time.Index = 16#1801; SDO List.Set event time.Subindex = 16#05; SDO List.Set event time.Value = 16#0064; SDO List.Set event time.Size = 16; SDO List.Set event time.AbortIfError = FALSE; SDO List.Set event time.JumpToLine = FALSE; SDO List.Set event time.Line = 0; SDO List.Clear pdo mapping.Index = 16#1A01; SDO List.Clear pdo mapping.Subindex = 16#00; SDO List.Clear pdo mapping.Value = 16#0; SDO List.Clear pdo mapping.Size = 8; SDO List.Clear pdo mapping.AbortIfError = FALSE; SDO List.Clear pdo mapping.JumpToLine = FALSE; SDO List.Clear pdo mapping.Line = 0; SDO List.Set Mapping.Index = 16#1A01; SDO List.Set Mapping.Subindex = 16#01; SDO List.Set Mapping.Value = 16#60410010; SDO List.Set Mapping.Size = 32; SDO List.Set Mapping.AbortIfError = FALSE; SDO List.Set Mapping.JumpToLine = FALSE; SDO List.Set Mapping.Line = 0;
              SDO List.Set Mapping.Index = 16#1A01; SDO List.Set Mapping.Subindex = 16#02; SDO List.Set Mapping.Value = 16#60640020; SDO List.Set Mapping.Size = 32; SDO List.Set Mapping.AbortIfError = FALSE; SDO List.Set Mapping.JumpToLine = FALSE; SDO List.Set Mapping.Line = 0; SDO List.Set number of pdos.Index = 16#1A01; SDO List.Set number of pdos.Subindex = 16#00; SDO List.Set number of pdos.Value = 16#02; SDO List.Set number of pdos.Size = 8; SDO List.Set number of pdos.AbortIfError = FALSE; SDO List.Set number of pdos.JumpToLine = FALSE; SDO List.Set number of pdos.Line = 0; SDO List.Set and enable COB-ID.Index = 16#1801; SDO List.Set and enable COB-ID.Subindex = 16#01; SDO List.Set and enable COB-ID.Value = 16#40000295; SDO List.Set and enable COB-ID.Size = 32; SDO List.Set and enable COB-ID.AbortIfError = FALSE; SDO List.Set and enable COB-ID.JumpToLine = FALSE; SDO List.Set and enable COB-ID.Line = 0; SDO List.Disable PDO.Index = 16#1802; SDO List.Disable PDO.Subindex = 16#01; SDO List.Disable PDO.Value = 16#C0000395; SDO List.Disable PDO.Size = 32; SDO List.Disable PDO.AbortIfError = FALSE; SDO List.Disable PDO.JumpToLine = FALSE; SDO List.Disable PDO.Line = 0; SDO List.Set transmission type.Index = 16#1802; SDO List.Set transmission type.Subindex = 16#02; SDO List.Set transmission type.Value = 16#FF; SDO List.Set transmission type.Size = 8; SDO List.Set transmission type.AbortIfError = FALSE; SDO List.Set transmission type.JumpToLine = FALSE; SDO List.Set transmission type.Line = 0; SDO List.Set inhibit time.Index = 16#1802; SDO List.Set inhibit time.Subindex = 16#03; SDO List.Set inhibit time.Value = 16#0064; SDO List.Set inhibit time.Size = 16; SDO List.Set inhibit time.AbortIfError = FALSE;
              SDO List.Set inhibit time.JumpToLine = FALSE; SDO List.Set inhibit time.Line = 0; SDO List.Set event time.Index = 16#1802; SDO List.Set event time.Subindex = 16#05; SDO List.Set event time.Value = 16#0064; SDO List.Set event time.Size = 16; SDO List.Set event time.AbortIfError = FALSE; SDO List.Set event time.JumpToLine = FALSE; SDO List.Set event time.Line = 0; SDO List.Clear pdo mapping.Index = 16#1A02; SDO List.Clear pdo mapping.Subindex = 16#00; SDO List.Clear pdo mapping.Value = 16#0; SDO List.Clear pdo mapping.Size = 8; SDO List.Clear pdo mapping.AbortIfError = FALSE; SDO List.Clear pdo mapping.JumpToLine = FALSE; SDO List.Clear pdo mapping.Line = 0; SDO List.Set Mapping.Index = 16#1A02; SDO List.Set Mapping.Subindex = 16#01; SDO List.Set Mapping.Value = 16#60410010; SDO List.Set Mapping.Size = 32; SDO List.Set Mapping.AbortIfError = FALSE; SDO List.Set Mapping.JumpToLine = FALSE; SDO List.Set Mapping.Line = 0; SDO List.Set Mapping.Index = 16#1A02; SDO List.Set Mapping.Subindex = 16#02; SDO List.Set Mapping.Value = 16#606C0020; SDO List.Set Mapping.Size = 32; SDO List.Set Mapping.AbortIfError = FALSE; SDO List.Set Mapping.JumpToLine = FALSE; SDO List.Set Mapping.Line = 0; SDO List.Set number of pdos.Index = 16#1A02; SDO List.Set number of pdos.Subindex = 16#00; SDO List.Set number of pdos.Value = 16#02; SDO List.Set number of pdos.Size = 8; SDO List.Set number of pdos.AbortIfError = FALSE; SDO List.Set number of pdos.JumpToLine = FALSE; SDO List.Set number of pdos.Line = 0; SDO List.Set and enable COB-ID.Index = 16#1802; SDO List.Set and enable COB-ID.Subindex = 16#01; SDO List.Set and enable COB-ID.Value = 16#40000395;
              SDO List.Set and enable COB-ID.Size = 32; SDO List.Set and enable COB-ID.AbortIfError = FALSE; SDO List.Set and enable COB-ID.JumpToLine = FALSE; SDO List.Set and enable COB-ID.Line = 0; SDO List.Disable PDO.Index = 16#1803; SDO List.Disable PDO.Subindex = 16#01; SDO List.Disable PDO.Value = 16#C0000495; SDO List.Disable PDO.Size = 32; SDO List.Disable PDO.AbortIfError = FALSE; SDO List.Disable PDO.JumpToLine = FALSE; SDO List.Disable PDO.Line = 0; SDO List.Automap SDO1.Index = 16#3041; SDO List.Automap SDO1.Subindex = 16#0B; SDO List.Automap SDO1.Value = 15; SDO List.Automap SDO1.Size = 16; SDO List.Automap SDO1.AbortIfError = FALSE; SDO List.Automap SDO1.JumpToLine = FALSE; SDO List.Automap SDO1.Line = 0; SDO List.Automap SDO2.Index = 16#301B; SDO List.Automap SDO2.Subindex = 16#08; SDO List.Automap SDO2.Value = 1; SDO List.Automap SDO2.Size = 16; SDO List.Automap SDO2.AbortIfError = FALSE; SDO List.Automap SDO2.JumpToLine = FALSE; SDO List.Automap SDO2.Line = 0; SDO List.Automap SDO3.Index = 16#3023; SDO List.Automap SDO3.Subindex = 16#09; SDO List.Automap SDO3.Value = 1; SDO List.Automap SDO3.Size = 16; SDO List.Automap SDO3.AbortIfError = FALSE; SDO List.Automap SDO3.JumpToLine = FALSE; SDO List.Automap SDO3.Line = 0; SDO List.IOsigLIMN.Index = 16#3006; SDO List.IOsigLIMN.Subindex = 16#0F; SDO List.IOsigLIMN.Value = 0; SDO List.IOsigLIMN.Size = 16; SDO List.IOsigLIMN.AbortIfError = FALSE; SDO List.IOsigLIMN.JumpToLine = FALSE; SDO List.IOsigLIMN.Line = 0; SDO List.IOsigLIMP.Index = 16#3006;
              SDO List.IOsigLIMP.Subindex = 16#10; SDO List.IOsigLIMP.Value = 0; SDO List.IOsigLIMP.Size = 16; SDO List.IOsigLIMP.AbortIfError = FALSE; SDO List.IOsigLIMP.JumpToLine = FALSE; SDO List.IOsigLIMP.Line = 0; ConfigVersion = 50659584
            input  Application.GVL_LXM32i_Node11.diActlPos : DINT  // Position actual value
            input  Application.GVL_LXM32i_Node11.diActlVelo : DINT  // Velocity actual value
            unmapped channels: driveModeCtrl, RefA16, RefB32, driveStat, mfStat, motionStat, driveInput, Statusword, Statusword
        BG75ci_0A : BG75ci, Dunkermotoren GmbH, order no. 0, version Revision=16#00000001, FileVersion=2.20, File=Dunker_BG75ci.eds
            settings: NODEIDSAVED = 10; SDO Timeout = 1000000; EXPERTSETTINGS = True; Emergency-General Parameters.Emergency COBID = 16#8A; Heartbeat-Producer Time = 3000; PDO 16#1400.COBID = 16#4000020A; PDO 16#1401.COBID = 16#4000030A; PDO 16#1402.COBID = 16#C000040A; PDO 16#1403.COBID = 16#C000050A; PDO 16#1404.COBID = 16#C0000000; Generic COBID = '16#C0000000'; PDO 16#1405.COBID = 16#C0000000; Generic COBID = '16#C0000000'; PDO 16#1406.COBID = 16#C0000000; Generic COBID = '16#C0000000'; PDO 16#1414.COBID = 16#C0000000; Generic COBID = '16#C0000000'; PDO 16#1800.COBID = 16#018A; PDO 16#1800.Inhibit Time = 1000; PDO 16#1800.Event Timer = 1000; PDO 16#1801.COBID = 16#028A; PDO 16#1801.Inhibit Time = 1000; PDO 16#1801.Event Timer = 1000; PDO 16#1802.COBID = 16#8000038A; PDO 16#1802.Event Timer = 0; PDO 16#1803.COBID = 16#8000048A; PDO 16#1803.Event Timer = 0; PDO 16#1804.Event Timer = 0; PDO 16#1805.Event Timer = 0; PDO 16#1806.Event Timer = 0; PDO 16#1814.Event Timer = 0; Heartbeat-Consuming1.Heartbeat-Time = 4500 ms; Controlword.Index = 16#6040; Controlword.Subindex = 16#00; Controlword.ObjectLength = 16; Brake.Index = 16#3150; Brake.Subindex = 16#00; Brake.ObjectLength = 16; Modes of operation.Index = 16#6060; Modes of operation.Subindex = 16#00;
              Modes of operation.ObjectLength = 8; Target position.Index = 16#607A; Target position.Subindex = 16#00; Target position.ObjectLength = 32; Target velocity.Index = 16#60FF; Target velocity.Subindex = 16#00; Target velocity.ObjectLength = 32; Statusword.Index = 16#6041; Statusword.Subindex = 16#00; Statusword.ObjectLength = 16; Modes of operation display.Index = 16#6061; Modes of operation display.Subindex = 16#00; Modes of operation display.ObjectLength = 8; Current actual value.Index = 16#6078; Current actual value.Subindex = 16#00; Current actual value.ObjectLength = 16; Torque actual value.Index = 16#6077; Torque actual value.Subindex = 16#00; Torque actual value.ObjectLength = 16; Position actual value.Index = 16#6064; Position actual value.Subindex = 16#00; Position actual value.ObjectLength = 32; Velocity actual value.Index = 16#606C; Velocity actual value.Subindex = 16#00; Velocity actual value.ObjectLength = 32; SDO List.Disable TIME.Index = 16#1012; SDO List.Disable TIME.Subindex = 16#00; SDO List.Disable TIME.Value = 16#00000100; SDO List.Disable TIME.Size = 32; SDO List.Disable TIME.AbortIfError = FALSE; SDO List.Disable TIME.JumpToLine = FALSE; SDO List.Disable TIME.Line = 0; SDO List.Set Guardtime.Index = 16#100C; SDO List.Set Guardtime.Subindex = 16#00; SDO List.Set Guardtime.Value = 16#00000000; SDO List.Set Guardtime.Size = 16; SDO List.Set Guardtime.AbortIfError = FALSE; SDO List.Set Guardtime.JumpToLine = FALSE; SDO List.Set Guardtime.Line = 0; SDO List.Set Lifetime.Index = 16#100D;
              SDO List.Set Lifetime.Subindex = 16#00; SDO List.Set Lifetime.Value = 16#00000000; SDO List.Set Lifetime.Size = 8; SDO List.Set Lifetime.AbortIfError = FALSE; SDO List.Set Lifetime.JumpToLine = FALSE; SDO List.Set Lifetime.Line = 0; SDO List.Disable Emcy CobID.Index = 16#1014; SDO List.Disable Emcy CobID.Subindex = 16#00; SDO List.Disable Emcy CobID.Value = 16#8000008A; SDO List.Disable Emcy CobID.Size = 32; SDO List.Disable Emcy CobID.AbortIfError = FALSE; SDO List.Disable Emcy CobID.JumpToLine = FALSE; SDO List.Disable Emcy CobID.Line = 0; SDO List.Set Emcy CobID.Index = 16#1014; SDO List.Set Emcy CobID.Subindex = 16#00; SDO List.Set Emcy CobID.Value = 16#0000008A; SDO List.Set Emcy CobID.Size = 32; SDO List.Set Emcy CobID.AbortIfError = FALSE; SDO List.Set Emcy CobID.JumpToLine = FALSE; SDO List.Set Emcy CobID.Line = 0; SDO List.Set Heartbeat Consumer.Index = 16#1016; SDO List.Set Heartbeat Consumer.Subindex = 16#01; SDO List.Set Heartbeat Consumer.Value = 16#00011194; SDO List.Set Heartbeat Consumer.Size = 32; SDO List.Set Heartbeat Consumer.AbortIfError = FALSE; SDO List.Set Heartbeat Consumer.JumpToLine = FALSE; SDO List.Set Heartbeat Consumer.Line = 0; SDO List.Set Heartbeat Consumer.Index = 16#1016; SDO List.Set Heartbeat Consumer.Subindex = 16#02; SDO List.Set Heartbeat Consumer.Value = 0; SDO List.Set Heartbeat Consumer.Size = 32; SDO List.Set Heartbeat Consumer.AbortIfError = FALSE; SDO List.Set Heartbeat Consumer.JumpToLine = FALSE; SDO List.Set Heartbeat Consumer.Line = 0; SDO List.Set Heartbeat Consumer.Index = 16#1016; SDO List.Set Heartbeat Consumer.Subindex = 16#03; SDO List.Set Heartbeat Consumer.Value = 0; SDO List.Set Heartbeat Consumer.Size = 32; SDO List.Set Heartbeat Consumer.AbortIfError = FALSE; SDO List.Set Heartbeat Consumer.JumpToLine = FALSE;
              SDO List.Set Heartbeat Consumer.Line = 0; SDO List.Set Heartbeat Consumer.Index = 16#1016; SDO List.Set Heartbeat Consumer.Subindex = 16#04; SDO List.Set Heartbeat Consumer.Value = 0; SDO List.Set Heartbeat Consumer.Size = 32; SDO List.Set Heartbeat Consumer.AbortIfError = FALSE; SDO List.Set Heartbeat Consumer.JumpToLine = FALSE; SDO List.Set Heartbeat Consumer.Line = 0; SDO List.Set Heartbeat Producer.Index = 16#1017; SDO List.Set Heartbeat Producer.Subindex = 16#00; SDO List.Set Heartbeat Producer.Value = 16#00000BB8; SDO List.Set Heartbeat Producer.Size = 16; SDO List.Set Heartbeat Producer.AbortIfError = FALSE; SDO List.Set Heartbeat Producer.JumpToLine = FALSE; SDO List.Set Heartbeat Producer.Line = 0; SDO List.Disable PDO.Index = 16#1400; SDO List.Disable PDO.Subindex = 16#01; SDO List.Disable PDO.Value = 16#C000020A; SDO List.Disable PDO.Size = 32; SDO List.Disable PDO.AbortIfError = FALSE; SDO List.Disable PDO.JumpToLine = FALSE; SDO List.Disable PDO.Line = 0; SDO List.Set transmission type.Index = 16#1400; SDO List.Set transmission type.Subindex = 16#02; SDO List.Set transmission type.Value = 16#FF; SDO List.Set transmission type.Size = 8; SDO List.Set transmission type.AbortIfError = FALSE; SDO List.Set transmission type.JumpToLine = FALSE; SDO List.Set transmission type.Line = 0; SDO List.Clear pdo mapping.Index = 16#1600; SDO List.Clear pdo mapping.Subindex = 16#00; SDO List.Clear pdo mapping.Value = 16#0; SDO List.Clear pdo mapping.Size = 8; SDO List.Clear pdo mapping.AbortIfError = FALSE; SDO List.Clear pdo mapping.JumpToLine = FALSE; SDO List.Clear pdo mapping.Line = 0; SDO List.Set Mapping.Index = 16#1600; SDO List.Set Mapping.Subindex = 16#01; SDO List.Set Mapping.Value = 16#60400010; SDO List.Set Mapping.Size = 32;
              SDO List.Set Mapping.AbortIfError = FALSE; SDO List.Set Mapping.JumpToLine = FALSE; SDO List.Set Mapping.Line = 0; SDO List.Set Mapping.Index = 16#1600; SDO List.Set Mapping.Subindex = 16#02; SDO List.Set Mapping.Value = 16#31500010; SDO List.Set Mapping.Size = 32; SDO List.Set Mapping.AbortIfError = FALSE; SDO List.Set Mapping.JumpToLine = FALSE; SDO List.Set Mapping.Line = 0; SDO List.Set Mapping.Index = 16#1600; SDO List.Set Mapping.Subindex = 16#03; SDO List.Set Mapping.Value = 16#60600008; SDO List.Set Mapping.Size = 32; SDO List.Set Mapping.AbortIfError = FALSE; SDO List.Set Mapping.JumpToLine = FALSE; SDO List.Set Mapping.Line = 0; SDO List.Set number of pdos.Index = 16#1600; SDO List.Set number of pdos.Subindex = 16#00; SDO List.Set number of pdos.Value = 16#03; SDO List.Set number of pdos.Size = 8; SDO List.Set number of pdos.AbortIfError = FALSE; SDO List.Set number of pdos.JumpToLine = FALSE; SDO List.Set number of pdos.Line = 0; SDO List.Set and enable COB-ID.Index = 16#1400; SDO List.Set and enable COB-ID.Subindex = 16#01; SDO List.Set and enable COB-ID.Value = 16#4000020A; SDO List.Set and enable COB-ID.Size = 32; SDO List.Set and enable COB-ID.AbortIfError = FALSE; SDO List.Set and enable COB-ID.JumpToLine = FALSE; SDO List.Set and enable COB-ID.Line = 0; SDO List.Disable PDO.Index = 16#1401; SDO List.Disable PDO.Subindex = 16#01; SDO List.Disable PDO.Value = 16#C000030A; SDO List.Disable PDO.Size = 32; SDO List.Disable PDO.AbortIfError = FALSE; SDO List.Disable PDO.JumpToLine = FALSE; SDO List.Disable PDO.Line = 0; SDO List.Set transmission type.Index = 16#1401; SDO List.Set transmission type.Subindex = 16#02;
              SDO List.Set transmission type.Value = 16#FF; SDO List.Set transmission type.Size = 8; SDO List.Set transmission type.AbortIfError = FALSE; SDO List.Set transmission type.JumpToLine = FALSE; SDO List.Set transmission type.Line = 0; SDO List.Clear pdo mapping.Index = 16#1601; SDO List.Clear pdo mapping.Subindex = 16#00; SDO List.Clear pdo mapping.Value = 16#0; SDO List.Clear pdo mapping.Size = 8; SDO List.Clear pdo mapping.AbortIfError = FALSE; SDO List.Clear pdo mapping.JumpToLine = FALSE; SDO List.Clear pdo mapping.Line = 0; SDO List.Set Mapping.Index = 16#1601; SDO List.Set Mapping.Subindex = 16#01; SDO List.Set Mapping.Value = 16#607A0020; SDO List.Set Mapping.Size = 32; SDO List.Set Mapping.AbortIfError = FALSE; SDO List.Set Mapping.JumpToLine = FALSE; SDO List.Set Mapping.Line = 0; SDO List.Set Mapping.Index = 16#1601; SDO List.Set Mapping.Subindex = 16#02; SDO List.Set Mapping.Value = 16#60FF0020; SDO List.Set Mapping.Size = 32; SDO List.Set Mapping.AbortIfError = FALSE; SDO List.Set Mapping.JumpToLine = FALSE; SDO List.Set Mapping.Line = 0; SDO List.Set number of pdos.Index = 16#1601; SDO List.Set number of pdos.Subindex = 16#00; SDO List.Set number of pdos.Value = 16#02; SDO List.Set number of pdos.Size = 8; SDO List.Set number of pdos.AbortIfError = FALSE; SDO List.Set number of pdos.JumpToLine = FALSE; SDO List.Set number of pdos.Line = 0; SDO List.Set and enable COB-ID.Index = 16#1401; SDO List.Set and enable COB-ID.Subindex = 16#01; SDO List.Set and enable COB-ID.Value = 16#4000030A; SDO List.Set and enable COB-ID.Size = 32; SDO List.Set and enable COB-ID.AbortIfError = FALSE; SDO List.Set and enable COB-ID.JumpToLine = FALSE; SDO List.Set and enable COB-ID.Line = 0;
              SDO List.Disable PDO.Index = 16#1402; SDO List.Disable PDO.Subindex = 16#01; SDO List.Disable PDO.Value = 16#C000040A; SDO List.Disable PDO.Size = 32; SDO List.Disable PDO.AbortIfError = FALSE; SDO List.Disable PDO.JumpToLine = FALSE; SDO List.Disable PDO.Line = 0; SDO List.Disable PDO.Index = 16#1403; SDO List.Disable PDO.Subindex = 16#01; SDO List.Disable PDO.Value = 16#C000050A; SDO List.Disable PDO.Size = 32; SDO List.Disable PDO.AbortIfError = FALSE; SDO List.Disable PDO.JumpToLine = FALSE; SDO List.Disable PDO.Line = 0; SDO List.Disable PDO.Index = 16#1800; SDO List.Disable PDO.Subindex = 16#01; SDO List.Disable PDO.Value = 16#8000018A; SDO List.Disable PDO.Size = 32; SDO List.Disable PDO.AbortIfError = FALSE; SDO List.Disable PDO.JumpToLine = FALSE; SDO List.Disable PDO.Line = 0; SDO List.Set transmission type.Index = 16#1800; SDO List.Set transmission type.Subindex = 16#02; SDO List.Set transmission type.Value = 16#FF; SDO List.Set transmission type.Size = 8; SDO List.Set transmission type.AbortIfError = FALSE; SDO List.Set transmission type.JumpToLine = FALSE; SDO List.Set transmission type.Line = 0; SDO List.Set inhibit time.Index = 16#1800; SDO List.Set inhibit time.Subindex = 16#03; SDO List.Set inhibit time.Value = 16#03E8; SDO List.Set inhibit time.Size = 16; SDO List.Set inhibit time.AbortIfError = FALSE; SDO List.Set inhibit time.JumpToLine = FALSE; SDO List.Set inhibit time.Line = 0; SDO List.Set event time.Index = 16#1800; SDO List.Set event time.Subindex = 16#05; SDO List.Set event time.Value = 16#03E8; SDO List.Set event time.Size = 16; SDO List.Set event time.AbortIfError = FALSE;
              SDO List.Set event time.JumpToLine = FALSE; SDO List.Set event time.Line = 0; SDO List.Clear pdo mapping.Index = 16#1A00; SDO List.Clear pdo mapping.Subindex = 16#00; SDO List.Clear pdo mapping.Value = 16#0; SDO List.Clear pdo mapping.Size = 8; SDO List.Clear pdo mapping.AbortIfError = FALSE; SDO List.Clear pdo mapping.JumpToLine = FALSE; SDO List.Clear pdo mapping.Line = 0; SDO List.Set Mapping.Index = 16#1A00; SDO List.Set Mapping.Subindex = 16#01; SDO List.Set Mapping.Value = 16#60410010; SDO List.Set Mapping.Size = 32; SDO List.Set Mapping.AbortIfError = FALSE; SDO List.Set Mapping.JumpToLine = FALSE; SDO List.Set Mapping.Line = 0; SDO List.Set Mapping.Index = 16#1A00; SDO List.Set Mapping.Subindex = 16#02; SDO List.Set Mapping.Value = 16#60610008; SDO List.Set Mapping.Size = 32; SDO List.Set Mapping.AbortIfError = FALSE; SDO List.Set Mapping.JumpToLine = FALSE; SDO List.Set Mapping.Line = 0; SDO List.Set Mapping.Index = 16#1A00; SDO List.Set Mapping.Subindex = 16#03; SDO List.Set Mapping.Value = 16#60780010; SDO List.Set Mapping.Size = 32; SDO List.Set Mapping.AbortIfError = FALSE; SDO List.Set Mapping.JumpToLine = FALSE; SDO List.Set Mapping.Line = 0; SDO List.Set Mapping.Index = 16#1A00; SDO List.Set Mapping.Subindex = 16#04; SDO List.Set Mapping.Value = 16#60770010; SDO List.Set Mapping.Size = 32; SDO List.Set Mapping.AbortIfError = FALSE; SDO List.Set Mapping.JumpToLine = FALSE; SDO List.Set Mapping.Line = 0; SDO List.Set number of pdos.Index = 16#1A00; SDO List.Set number of pdos.Subindex = 16#00; SDO List.Set number of pdos.Value = 16#04;
              SDO List.Set number of pdos.Size = 8; SDO List.Set number of pdos.AbortIfError = FALSE; SDO List.Set number of pdos.JumpToLine = FALSE; SDO List.Set number of pdos.Line = 0; SDO List.Set and enable COB-ID.Index = 16#1800; SDO List.Set and enable COB-ID.Subindex = 16#01; SDO List.Set and enable COB-ID.Value = 16#0000018A; SDO List.Set and enable COB-ID.Size = 32; SDO List.Set and enable COB-ID.AbortIfError = FALSE; SDO List.Set and enable COB-ID.JumpToLine = FALSE; SDO List.Set and enable COB-ID.Line = 0; SDO List.Disable PDO.Index = 16#1801; SDO List.Disable PDO.Subindex = 16#01; SDO List.Disable PDO.Value = 16#8000028A; SDO List.Disable PDO.Size = 32; SDO List.Disable PDO.AbortIfError = FALSE; SDO List.Disable PDO.JumpToLine = FALSE; SDO List.Disable PDO.Line = 0; SDO List.Set transmission type.Index = 16#1801; SDO List.Set transmission type.Subindex = 16#02; SDO List.Set transmission type.Value = 16#FF; SDO List.Set transmission type.Size = 8; SDO List.Set transmission type.AbortIfError = FALSE; SDO List.Set transmission type.JumpToLine = FALSE; SDO List.Set transmission type.Line = 0; SDO List.Set inhibit time.Index = 16#1801; SDO List.Set inhibit time.Subindex = 16#03; SDO List.Set inhibit time.Value = 16#03E8; SDO List.Set inhibit time.Size = 16; SDO List.Set inhibit time.AbortIfError = FALSE; SDO List.Set inhibit time.JumpToLine = FALSE; SDO List.Set inhibit time.Line = 0; SDO List.Clear pdo mapping.Index = 16#1A01; SDO List.Clear pdo mapping.Subindex = 16#00; SDO List.Clear pdo mapping.Value = 16#0; SDO List.Clear pdo mapping.Size = 8; SDO List.Clear pdo mapping.AbortIfError = FALSE; SDO List.Clear pdo mapping.JumpToLine = FALSE; SDO List.Clear pdo mapping.Line = 0; SDO List.Set Mapping.Index = 16#1A01;
              SDO List.Set Mapping.Subindex = 16#01; SDO List.Set Mapping.Value = 16#60640020; SDO List.Set Mapping.Size = 32; SDO List.Set Mapping.AbortIfError = FALSE; SDO List.Set Mapping.JumpToLine = FALSE; SDO List.Set Mapping.Line = 0; SDO List.Set Mapping.Index = 16#1A01; SDO List.Set Mapping.Subindex = 16#02; SDO List.Set Mapping.Value = 16#606C0020; SDO List.Set Mapping.Size = 32; SDO List.Set Mapping.AbortIfError = FALSE; SDO List.Set Mapping.JumpToLine = FALSE; SDO List.Set Mapping.Line = 0; SDO List.Set number of pdos.Index = 16#1A01; SDO List.Set number of pdos.Subindex = 16#00; SDO List.Set number of pdos.Value = 16#02; SDO List.Set number of pdos.Size = 8; SDO List.Set number of pdos.AbortIfError = FALSE; SDO List.Set number of pdos.JumpToLine = FALSE; SDO List.Set number of pdos.Line = 0; SDO List.Set and enable COB-ID.Index = 16#1801; SDO List.Set and enable COB-ID.Subindex = 16#01; SDO List.Set and enable COB-ID.Value = 16#0000028A; SDO List.Set and enable COB-ID.Size = 32; SDO List.Set and enable COB-ID.AbortIfError = FALSE; SDO List.Set and enable COB-ID.JumpToLine = FALSE; SDO List.Set and enable COB-ID.Line = 0; SDO List.Disable PDO.Index = 16#1802; SDO List.Disable PDO.Subindex = 16#01; SDO List.Disable PDO.Value = 16#8000038A; SDO List.Disable PDO.Size = 32; SDO List.Disable PDO.AbortIfError = FALSE; SDO List.Disable PDO.JumpToLine = FALSE; SDO List.Disable PDO.Line = 0; SDO List.Disable PDO.Index = 16#1803; SDO List.Disable PDO.Subindex = 16#01; SDO List.Disable PDO.Value = 16#8000048A; SDO List.Disable PDO.Size = 32; SDO List.Disable PDO.AbortIfError = FALSE; SDO List.Disable PDO.JumpToLine = FALSE;
              SDO List.Disable PDO.Line = 0; ConfigVersion = 50659584
            unmapped channels: Controlword, Brake, Modes of operation, Target position, Target velocity, Statusword, Modes of operation display, Current actual value, Torque actual value, Position actual value, Velocity actual value
        BG75ci_0B : BG75ci, Dunkermotoren GmbH, order no. 0, version Revision=16#00000001, FileVersion=2.20, File=Dunker_BG75ci.eds
            settings: NODEIDSAVED = 11; SDO Timeout = 1000000; EXPERTSETTINGS = True; Emergency-General Parameters.Emergency COBID = 16#8B; Heartbeat-Producer Time = 3000; PDO 16#1400.COBID = 16#4000020B; PDO 16#1401.COBID = 16#4000030B; PDO 16#1402.COBID = 16#C000040B; PDO 16#1403.COBID = 16#C000050B; PDO 16#1404.COBID = 16#C0000000; Generic COBID = '16#C0000000'; PDO 16#1405.COBID = 16#C0000000; Generic COBID = '16#C0000000'; PDO 16#1406.COBID = 16#C0000000; Generic COBID = '16#C0000000'; PDO 16#1414.COBID = 16#C0000000; Generic COBID = '16#C0000000'; PDO 16#1800.COBID = 16#018B; PDO 16#1800.Inhibit Time = 1000; PDO 16#1800.Event Timer = 1000; PDO 16#1801.COBID = 16#028B; PDO 16#1801.Inhibit Time = 1000; PDO 16#1801.Event Timer = 1000; PDO 16#1802.COBID = 16#8000038B; PDO 16#1802.Event Timer = 0; PDO 16#1803.COBID = 16#8000048B; PDO 16#1803.Event Timer = 0; PDO 16#1804.Event Timer = 0; PDO 16#1805.Event Timer = 0; PDO 16#1806.Event Timer = 0; PDO 16#1814.Event Timer = 0; Heartbeat-Consuming1.Heartbeat-Time = 4500 ms; Controlword.Index = 16#6040; Controlword.Subindex = 16#00; Controlword.ObjectLength = 16; Brake.Index = 16#3150; Brake.Subindex = 16#00; Brake.ObjectLength = 16; Modes of operation.Index = 16#6060; Modes of operation.Subindex = 16#00;
              Modes of operation.ObjectLength = 8; Target position.Index = 16#607A; Target position.Subindex = 16#00; Target position.ObjectLength = 32; Target velocity.Index = 16#60FF; Target velocity.Subindex = 16#00; Target velocity.ObjectLength = 32; Statusword.Index = 16#6041; Statusword.Subindex = 16#00; Statusword.ObjectLength = 16; Modes of operation display.Index = 16#6061; Modes of operation display.Subindex = 16#00; Modes of operation display.ObjectLength = 8; Current actual value.Index = 16#6078; Current actual value.Subindex = 16#00; Current actual value.ObjectLength = 16; Torque actual value.Index = 16#6077; Torque actual value.Subindex = 16#00; Torque actual value.ObjectLength = 16; Position actual value.Index = 16#6064; Position actual value.Subindex = 16#00; Position actual value.ObjectLength = 32; Velocity actual value.Index = 16#606C; Velocity actual value.Subindex = 16#00; Velocity actual value.ObjectLength = 32; SDO List.Disable TIME.Index = 16#1012; SDO List.Disable TIME.Subindex = 16#00; SDO List.Disable TIME.Value = 16#00000100; SDO List.Disable TIME.Size = 32; SDO List.Disable TIME.AbortIfError = FALSE; SDO List.Disable TIME.JumpToLine = FALSE; SDO List.Disable TIME.Line = 0; SDO List.Set Guardtime.Index = 16#100C; SDO List.Set Guardtime.Subindex = 16#00; SDO List.Set Guardtime.Value = 16#00000000; SDO List.Set Guardtime.Size = 16; SDO List.Set Guardtime.AbortIfError = FALSE; SDO List.Set Guardtime.JumpToLine = FALSE; SDO List.Set Guardtime.Line = 0; SDO List.Set Lifetime.Index = 16#100D;
              SDO List.Set Lifetime.Subindex = 16#00; SDO List.Set Lifetime.Value = 16#00000000; SDO List.Set Lifetime.Size = 8; SDO List.Set Lifetime.AbortIfError = FALSE; SDO List.Set Lifetime.JumpToLine = FALSE; SDO List.Set Lifetime.Line = 0; SDO List.Disable Emcy CobID.Index = 16#1014; SDO List.Disable Emcy CobID.Subindex = 16#00; SDO List.Disable Emcy CobID.Value = 16#8000008B; SDO List.Disable Emcy CobID.Size = 32; SDO List.Disable Emcy CobID.AbortIfError = FALSE; SDO List.Disable Emcy CobID.JumpToLine = FALSE; SDO List.Disable Emcy CobID.Line = 0; SDO List.Set Emcy CobID.Index = 16#1014; SDO List.Set Emcy CobID.Subindex = 16#00; SDO List.Set Emcy CobID.Value = 16#0000008B; SDO List.Set Emcy CobID.Size = 32; SDO List.Set Emcy CobID.AbortIfError = FALSE; SDO List.Set Emcy CobID.JumpToLine = FALSE; SDO List.Set Emcy CobID.Line = 0; SDO List.Set Heartbeat Consumer.Index = 16#1016; SDO List.Set Heartbeat Consumer.Subindex = 16#01; SDO List.Set Heartbeat Consumer.Value = 16#00011194; SDO List.Set Heartbeat Consumer.Size = 32; SDO List.Set Heartbeat Consumer.AbortIfError = FALSE; SDO List.Set Heartbeat Consumer.JumpToLine = FALSE; SDO List.Set Heartbeat Consumer.Line = 0; SDO List.Set Heartbeat Consumer.Index = 16#1016; SDO List.Set Heartbeat Consumer.Subindex = 16#02; SDO List.Set Heartbeat Consumer.Value = 0; SDO List.Set Heartbeat Consumer.Size = 32; SDO List.Set Heartbeat Consumer.AbortIfError = FALSE; SDO List.Set Heartbeat Consumer.JumpToLine = FALSE; SDO List.Set Heartbeat Consumer.Line = 0; SDO List.Set Heartbeat Consumer.Index = 16#1016; SDO List.Set Heartbeat Consumer.Subindex = 16#03; SDO List.Set Heartbeat Consumer.Value = 0; SDO List.Set Heartbeat Consumer.Size = 32; SDO List.Set Heartbeat Consumer.AbortIfError = FALSE; SDO List.Set Heartbeat Consumer.JumpToLine = FALSE;
              SDO List.Set Heartbeat Consumer.Line = 0; SDO List.Set Heartbeat Consumer.Index = 16#1016; SDO List.Set Heartbeat Consumer.Subindex = 16#04; SDO List.Set Heartbeat Consumer.Value = 0; SDO List.Set Heartbeat Consumer.Size = 32; SDO List.Set Heartbeat Consumer.AbortIfError = FALSE; SDO List.Set Heartbeat Consumer.JumpToLine = FALSE; SDO List.Set Heartbeat Consumer.Line = 0; SDO List.Set Heartbeat Producer.Index = 16#1017; SDO List.Set Heartbeat Producer.Subindex = 16#00; SDO List.Set Heartbeat Producer.Value = 16#00000BB8; SDO List.Set Heartbeat Producer.Size = 16; SDO List.Set Heartbeat Producer.AbortIfError = FALSE; SDO List.Set Heartbeat Producer.JumpToLine = FALSE; SDO List.Set Heartbeat Producer.Line = 0; SDO List.Disable PDO.Index = 16#1400; SDO List.Disable PDO.Subindex = 16#01; SDO List.Disable PDO.Value = 16#C000020B; SDO List.Disable PDO.Size = 32; SDO List.Disable PDO.AbortIfError = FALSE; SDO List.Disable PDO.JumpToLine = FALSE; SDO List.Disable PDO.Line = 0; SDO List.Set transmission type.Index = 16#1400; SDO List.Set transmission type.Subindex = 16#02; SDO List.Set transmission type.Value = 16#FF; SDO List.Set transmission type.Size = 8; SDO List.Set transmission type.AbortIfError = FALSE; SDO List.Set transmission type.JumpToLine = FALSE; SDO List.Set transmission type.Line = 0; SDO List.Clear pdo mapping.Index = 16#1600; SDO List.Clear pdo mapping.Subindex = 16#00; SDO List.Clear pdo mapping.Value = 16#0; SDO List.Clear pdo mapping.Size = 8; SDO List.Clear pdo mapping.AbortIfError = FALSE; SDO List.Clear pdo mapping.JumpToLine = FALSE; SDO List.Clear pdo mapping.Line = 0; SDO List.Set Mapping.Index = 16#1600; SDO List.Set Mapping.Subindex = 16#01; SDO List.Set Mapping.Value = 16#60400010; SDO List.Set Mapping.Size = 32;
              SDO List.Set Mapping.AbortIfError = FALSE; SDO List.Set Mapping.JumpToLine = FALSE; SDO List.Set Mapping.Line = 0; SDO List.Set Mapping.Index = 16#1600; SDO List.Set Mapping.Subindex = 16#02; SDO List.Set Mapping.Value = 16#31500010; SDO List.Set Mapping.Size = 32; SDO List.Set Mapping.AbortIfError = FALSE; SDO List.Set Mapping.JumpToLine = FALSE; SDO List.Set Mapping.Line = 0; SDO List.Set Mapping.Index = 16#1600; SDO List.Set Mapping.Subindex = 16#03; SDO List.Set Mapping.Value = 16#60600008; SDO List.Set Mapping.Size = 32; SDO List.Set Mapping.AbortIfError = FALSE; SDO List.Set Mapping.JumpToLine = FALSE; SDO List.Set Mapping.Line = 0; SDO List.Set number of pdos.Index = 16#1600; SDO List.Set number of pdos.Subindex = 16#00; SDO List.Set number of pdos.Value = 16#03; SDO List.Set number of pdos.Size = 8; SDO List.Set number of pdos.AbortIfError = FALSE; SDO List.Set number of pdos.JumpToLine = FALSE; SDO List.Set number of pdos.Line = 0; SDO List.Set and enable COB-ID.Index = 16#1400; SDO List.Set and enable COB-ID.Subindex = 16#01; SDO List.Set and enable COB-ID.Value = 16#4000020B; SDO List.Set and enable COB-ID.Size = 32; SDO List.Set and enable COB-ID.AbortIfError = FALSE; SDO List.Set and enable COB-ID.JumpToLine = FALSE; SDO List.Set and enable COB-ID.Line = 0; SDO List.Disable PDO.Index = 16#1401; SDO List.Disable PDO.Subindex = 16#01; SDO List.Disable PDO.Value = 16#C000030B; SDO List.Disable PDO.Size = 32; SDO List.Disable PDO.AbortIfError = FALSE; SDO List.Disable PDO.JumpToLine = FALSE; SDO List.Disable PDO.Line = 0; SDO List.Set transmission type.Index = 16#1401; SDO List.Set transmission type.Subindex = 16#02;
              SDO List.Set transmission type.Value = 16#FF; SDO List.Set transmission type.Size = 8; SDO List.Set transmission type.AbortIfError = FALSE; SDO List.Set transmission type.JumpToLine = FALSE; SDO List.Set transmission type.Line = 0; SDO List.Clear pdo mapping.Index = 16#1601; SDO List.Clear pdo mapping.Subindex = 16#00; SDO List.Clear pdo mapping.Value = 16#0; SDO List.Clear pdo mapping.Size = 8; SDO List.Clear pdo mapping.AbortIfError = FALSE; SDO List.Clear pdo mapping.JumpToLine = FALSE; SDO List.Clear pdo mapping.Line = 0; SDO List.Set Mapping.Index = 16#1601; SDO List.Set Mapping.Subindex = 16#01; SDO List.Set Mapping.Value = 16#607A0020; SDO List.Set Mapping.Size = 32; SDO List.Set Mapping.AbortIfError = FALSE; SDO List.Set Mapping.JumpToLine = FALSE; SDO List.Set Mapping.Line = 0; SDO List.Set Mapping.Index = 16#1601; SDO List.Set Mapping.Subindex = 16#02; SDO List.Set Mapping.Value = 16#60FF0020; SDO List.Set Mapping.Size = 32; SDO List.Set Mapping.AbortIfError = FALSE; SDO List.Set Mapping.JumpToLine = FALSE; SDO List.Set Mapping.Line = 0; SDO List.Set number of pdos.Index = 16#1601; SDO List.Set number of pdos.Subindex = 16#00; SDO List.Set number of pdos.Value = 16#02; SDO List.Set number of pdos.Size = 8; SDO List.Set number of pdos.AbortIfError = FALSE; SDO List.Set number of pdos.JumpToLine = FALSE; SDO List.Set number of pdos.Line = 0; SDO List.Set and enable COB-ID.Index = 16#1401; SDO List.Set and enable COB-ID.Subindex = 16#01; SDO List.Set and enable COB-ID.Value = 16#4000030B; SDO List.Set and enable COB-ID.Size = 32; SDO List.Set and enable COB-ID.AbortIfError = FALSE; SDO List.Set and enable COB-ID.JumpToLine = FALSE; SDO List.Set and enable COB-ID.Line = 0;
              SDO List.Disable PDO.Index = 16#1402; SDO List.Disable PDO.Subindex = 16#01; SDO List.Disable PDO.Value = 16#C000040B; SDO List.Disable PDO.Size = 32; SDO List.Disable PDO.AbortIfError = FALSE; SDO List.Disable PDO.JumpToLine = FALSE; SDO List.Disable PDO.Line = 0; SDO List.Disable PDO.Index = 16#1403; SDO List.Disable PDO.Subindex = 16#01; SDO List.Disable PDO.Value = 16#C000050B; SDO List.Disable PDO.Size = 32; SDO List.Disable PDO.AbortIfError = FALSE; SDO List.Disable PDO.JumpToLine = FALSE; SDO List.Disable PDO.Line = 0; SDO List.Disable PDO.Index = 16#1800; SDO List.Disable PDO.Subindex = 16#01; SDO List.Disable PDO.Value = 16#8000018B; SDO List.Disable PDO.Size = 32; SDO List.Disable PDO.AbortIfError = FALSE; SDO List.Disable PDO.JumpToLine = FALSE; SDO List.Disable PDO.Line = 0; SDO List.Set transmission type.Index = 16#1800; SDO List.Set transmission type.Subindex = 16#02; SDO List.Set transmission type.Value = 16#FF; SDO List.Set transmission type.Size = 8; SDO List.Set transmission type.AbortIfError = FALSE; SDO List.Set transmission type.JumpToLine = FALSE; SDO List.Set transmission type.Line = 0; SDO List.Set inhibit time.Index = 16#1800; SDO List.Set inhibit time.Subindex = 16#03; SDO List.Set inhibit time.Value = 16#03E8; SDO List.Set inhibit time.Size = 16; SDO List.Set inhibit time.AbortIfError = FALSE; SDO List.Set inhibit time.JumpToLine = FALSE; SDO List.Set inhibit time.Line = 0; SDO List.Set event time.Index = 16#1800; SDO List.Set event time.Subindex = 16#05; SDO List.Set event time.Value = 16#03E8; SDO List.Set event time.Size = 16; SDO List.Set event time.AbortIfError = FALSE;
              SDO List.Set event time.JumpToLine = FALSE; SDO List.Set event time.Line = 0; SDO List.Clear pdo mapping.Index = 16#1A00; SDO List.Clear pdo mapping.Subindex = 16#00; SDO List.Clear pdo mapping.Value = 16#0; SDO List.Clear pdo mapping.Size = 8; SDO List.Clear pdo mapping.AbortIfError = FALSE; SDO List.Clear pdo mapping.JumpToLine = FALSE; SDO List.Clear pdo mapping.Line = 0; SDO List.Set Mapping.Index = 16#1A00; SDO List.Set Mapping.Subindex = 16#01; SDO List.Set Mapping.Value = 16#60410010; SDO List.Set Mapping.Size = 32; SDO List.Set Mapping.AbortIfError = FALSE; SDO List.Set Mapping.JumpToLine = FALSE; SDO List.Set Mapping.Line = 0; SDO List.Set Mapping.Index = 16#1A00; SDO List.Set Mapping.Subindex = 16#02; SDO List.Set Mapping.Value = 16#60610008; SDO List.Set Mapping.Size = 32; SDO List.Set Mapping.AbortIfError = FALSE; SDO List.Set Mapping.JumpToLine = FALSE; SDO List.Set Mapping.Line = 0; SDO List.Set Mapping.Index = 16#1A00; SDO List.Set Mapping.Subindex = 16#03; SDO List.Set Mapping.Value = 16#60780010; SDO List.Set Mapping.Size = 32; SDO List.Set Mapping.AbortIfError = FALSE; SDO List.Set Mapping.JumpToLine = FALSE; SDO List.Set Mapping.Line = 0; SDO List.Set Mapping.Index = 16#1A00; SDO List.Set Mapping.Subindex = 16#04; SDO List.Set Mapping.Value = 16#60770010; SDO List.Set Mapping.Size = 32; SDO List.Set Mapping.AbortIfError = FALSE; SDO List.Set Mapping.JumpToLine = FALSE; SDO List.Set Mapping.Line = 0; SDO List.Set number of pdos.Index = 16#1A00; SDO List.Set number of pdos.Subindex = 16#00; SDO List.Set number of pdos.Value = 16#04;
              SDO List.Set number of pdos.Size = 8; SDO List.Set number of pdos.AbortIfError = FALSE; SDO List.Set number of pdos.JumpToLine = FALSE; SDO List.Set number of pdos.Line = 0; SDO List.Set and enable COB-ID.Index = 16#1800; SDO List.Set and enable COB-ID.Subindex = 16#01; SDO List.Set and enable COB-ID.Value = 16#0000018B; SDO List.Set and enable COB-ID.Size = 32; SDO List.Set and enable COB-ID.AbortIfError = FALSE; SDO List.Set and enable COB-ID.JumpToLine = FALSE; SDO List.Set and enable COB-ID.Line = 0; SDO List.Disable PDO.Index = 16#1801; SDO List.Disable PDO.Subindex = 16#01; SDO List.Disable PDO.Value = 16#8000028B; SDO List.Disable PDO.Size = 32; SDO List.Disable PDO.AbortIfError = FALSE; SDO List.Disable PDO.JumpToLine = FALSE; SDO List.Disable PDO.Line = 0; SDO List.Set transmission type.Index = 16#1801; SDO List.Set transmission type.Subindex = 16#02; SDO List.Set transmission type.Value = 16#FF; SDO List.Set transmission type.Size = 8; SDO List.Set transmission type.AbortIfError = FALSE; SDO List.Set transmission type.JumpToLine = FALSE; SDO List.Set transmission type.Line = 0; SDO List.Set inhibit time.Index = 16#1801; SDO List.Set inhibit time.Subindex = 16#03; SDO List.Set inhibit time.Value = 16#03E8; SDO List.Set inhibit time.Size = 16; SDO List.Set inhibit time.AbortIfError = FALSE; SDO List.Set inhibit time.JumpToLine = FALSE; SDO List.Set inhibit time.Line = 0; SDO List.Clear pdo mapping.Index = 16#1A01; SDO List.Clear pdo mapping.Subindex = 16#00; SDO List.Clear pdo mapping.Value = 16#0; SDO List.Clear pdo mapping.Size = 8; SDO List.Clear pdo mapping.AbortIfError = FALSE; SDO List.Clear pdo mapping.JumpToLine = FALSE; SDO List.Clear pdo mapping.Line = 0; SDO List.Set Mapping.Index = 16#1A01;
              SDO List.Set Mapping.Subindex = 16#01; SDO List.Set Mapping.Value = 16#60640020; SDO List.Set Mapping.Size = 32; SDO List.Set Mapping.AbortIfError = FALSE; SDO List.Set Mapping.JumpToLine = FALSE; SDO List.Set Mapping.Line = 0; SDO List.Set Mapping.Index = 16#1A01; SDO List.Set Mapping.Subindex = 16#02; SDO List.Set Mapping.Value = 16#606C0020; SDO List.Set Mapping.Size = 32; SDO List.Set Mapping.AbortIfError = FALSE; SDO List.Set Mapping.JumpToLine = FALSE; SDO List.Set Mapping.Line = 0; SDO List.Set number of pdos.Index = 16#1A01; SDO List.Set number of pdos.Subindex = 16#00; SDO List.Set number of pdos.Value = 16#02; SDO List.Set number of pdos.Size = 8; SDO List.Set number of pdos.AbortIfError = FALSE; SDO List.Set number of pdos.JumpToLine = FALSE; SDO List.Set number of pdos.Line = 0; SDO List.Set and enable COB-ID.Index = 16#1801; SDO List.Set and enable COB-ID.Subindex = 16#01; SDO List.Set and enable COB-ID.Value = 16#0000028B; SDO List.Set and enable COB-ID.Size = 32; SDO List.Set and enable COB-ID.AbortIfError = FALSE; SDO List.Set and enable COB-ID.JumpToLine = FALSE; SDO List.Set and enable COB-ID.Line = 0; SDO List.Disable PDO.Index = 16#1802; SDO List.Disable PDO.Subindex = 16#01; SDO List.Disable PDO.Value = 16#8000038B; SDO List.Disable PDO.Size = 32; SDO List.Disable PDO.AbortIfError = FALSE; SDO List.Disable PDO.JumpToLine = FALSE; SDO List.Disable PDO.Line = 0; SDO List.Disable PDO.Index = 16#1803; SDO List.Disable PDO.Subindex = 16#01; SDO List.Disable PDO.Value = 16#8000048B; SDO List.Disable PDO.Size = 32; SDO List.Disable PDO.AbortIfError = FALSE; SDO List.Disable PDO.JumpToLine = FALSE;
              SDO List.Disable PDO.Line = 0; ConfigVersion = 50659584
            unmapped channels: Controlword, Brake, Modes of operation, Target position, Target velocity, Statusword, Modes of operation display, Current actual value, Torque actual value, Position actual value, Velocity actual value
        BG75ci_0C : BG75ci, Dunkermotoren GmbH, order no. 0, version Revision=16#00000001, FileVersion=2.20, File=Dunker_BG75ci.eds
            settings: NODEIDSAVED = 12; SDO Timeout = 1000000; EXPERTSETTINGS = True; Emergency-General Parameters.Emergency COBID = 16#8C; Heartbeat-Producer Time = 3000; PDO 16#1400.COBID = 16#4000020C; PDO 16#1401.COBID = 16#4000030C; PDO 16#1402.COBID = 16#C000040C; PDO 16#1403.COBID = 16#C000050C; PDO 16#1404.COBID = 16#C0000000; Generic COBID = '16#C0000000'; PDO 16#1405.COBID = 16#C0000000; Generic COBID = '16#C0000000'; PDO 16#1406.COBID = 16#C0000000; Generic COBID = '16#C0000000'; PDO 16#1414.COBID = 16#C0000000; Generic COBID = '16#C0000000'; PDO 16#1800.COBID = 16#018C; PDO 16#1800.Inhibit Time = 1000; PDO 16#1800.Event Timer = 1000; PDO 16#1801.COBID = 16#028C; PDO 16#1801.Inhibit Time = 1000; PDO 16#1801.Event Timer = 1000; PDO 16#1802.COBID = 16#8000038C; PDO 16#1802.Event Timer = 0; PDO 16#1803.COBID = 16#8000048C; PDO 16#1803.Event Timer = 0; PDO 16#1804.Event Timer = 0; PDO 16#1805.Event Timer = 0; PDO 16#1806.Event Timer = 0; PDO 16#1814.Event Timer = 0; Heartbeat-Consuming1.Heartbeat-Time = 4500 ms; Controlword.Index = 16#6040; Controlword.Subindex = 16#00; Controlword.ObjectLength = 16; Brake.Index = 16#3150; Brake.Subindex = 16#00; Brake.ObjectLength = 16; Modes of operation.Index = 16#6060; Modes of operation.Subindex = 16#00;
              Modes of operation.ObjectLength = 8; Target position.Index = 16#607A; Target position.Subindex = 16#00; Target position.ObjectLength = 32; Target velocity.Index = 16#60FF; Target velocity.Subindex = 16#00; Target velocity.ObjectLength = 32; Statusword.Index = 16#6041; Statusword.Subindex = 16#00; Statusword.ObjectLength = 16; Modes of operation display.Index = 16#6061; Modes of operation display.Subindex = 16#00; Modes of operation display.ObjectLength = 8; Current actual value.Index = 16#6078; Current actual value.Subindex = 16#00; Current actual value.ObjectLength = 16; Torque actual value.Index = 16#6077; Torque actual value.Subindex = 16#00; Torque actual value.ObjectLength = 16; Position actual value.Index = 16#6064; Position actual value.Subindex = 16#00; Position actual value.ObjectLength = 32; Velocity actual value.Index = 16#606C; Velocity actual value.Subindex = 16#00; Velocity actual value.ObjectLength = 32; SDO List.Disable TIME.Index = 16#1012; SDO List.Disable TIME.Subindex = 16#00; SDO List.Disable TIME.Value = 16#00000100; SDO List.Disable TIME.Size = 32; SDO List.Disable TIME.AbortIfError = FALSE; SDO List.Disable TIME.JumpToLine = FALSE; SDO List.Disable TIME.Line = 0; SDO List.Set Guardtime.Index = 16#100C; SDO List.Set Guardtime.Subindex = 16#00; SDO List.Set Guardtime.Value = 16#00000000; SDO List.Set Guardtime.Size = 16; SDO List.Set Guardtime.AbortIfError = FALSE; SDO List.Set Guardtime.JumpToLine = FALSE; SDO List.Set Guardtime.Line = 0; SDO List.Set Lifetime.Index = 16#100D;
              SDO List.Set Lifetime.Subindex = 16#00; SDO List.Set Lifetime.Value = 16#00000000; SDO List.Set Lifetime.Size = 8; SDO List.Set Lifetime.AbortIfError = FALSE; SDO List.Set Lifetime.JumpToLine = FALSE; SDO List.Set Lifetime.Line = 0; SDO List.Disable Emcy CobID.Index = 16#1014; SDO List.Disable Emcy CobID.Subindex = 16#00; SDO List.Disable Emcy CobID.Value = 16#8000008C; SDO List.Disable Emcy CobID.Size = 32; SDO List.Disable Emcy CobID.AbortIfError = FALSE; SDO List.Disable Emcy CobID.JumpToLine = FALSE; SDO List.Disable Emcy CobID.Line = 0; SDO List.Set Emcy CobID.Index = 16#1014; SDO List.Set Emcy CobID.Subindex = 16#00; SDO List.Set Emcy CobID.Value = 16#0000008C; SDO List.Set Emcy CobID.Size = 32; SDO List.Set Emcy CobID.AbortIfError = FALSE; SDO List.Set Emcy CobID.JumpToLine = FALSE; SDO List.Set Emcy CobID.Line = 0; SDO List.Set Heartbeat Consumer.Index = 16#1016; SDO List.Set Heartbeat Consumer.Subindex = 16#01; SDO List.Set Heartbeat Consumer.Value = 16#00011194; SDO List.Set Heartbeat Consumer.Size = 32; SDO List.Set Heartbeat Consumer.AbortIfError = FALSE; SDO List.Set Heartbeat Consumer.JumpToLine = FALSE; SDO List.Set Heartbeat Consumer.Line = 0; SDO List.Set Heartbeat Consumer.Index = 16#1016; SDO List.Set Heartbeat Consumer.Subindex = 16#02; SDO List.Set Heartbeat Consumer.Value = 0; SDO List.Set Heartbeat Consumer.Size = 32; SDO List.Set Heartbeat Consumer.AbortIfError = FALSE; SDO List.Set Heartbeat Consumer.JumpToLine = FALSE; SDO List.Set Heartbeat Consumer.Line = 0; SDO List.Set Heartbeat Consumer.Index = 16#1016; SDO List.Set Heartbeat Consumer.Subindex = 16#03; SDO List.Set Heartbeat Consumer.Value = 0; SDO List.Set Heartbeat Consumer.Size = 32; SDO List.Set Heartbeat Consumer.AbortIfError = FALSE; SDO List.Set Heartbeat Consumer.JumpToLine = FALSE;
              SDO List.Set Heartbeat Consumer.Line = 0; SDO List.Set Heartbeat Consumer.Index = 16#1016; SDO List.Set Heartbeat Consumer.Subindex = 16#04; SDO List.Set Heartbeat Consumer.Value = 0; SDO List.Set Heartbeat Consumer.Size = 32; SDO List.Set Heartbeat Consumer.AbortIfError = FALSE; SDO List.Set Heartbeat Consumer.JumpToLine = FALSE; SDO List.Set Heartbeat Consumer.Line = 0; SDO List.Set Heartbeat Producer.Index = 16#1017; SDO List.Set Heartbeat Producer.Subindex = 16#00; SDO List.Set Heartbeat Producer.Value = 16#00000BB8; SDO List.Set Heartbeat Producer.Size = 16; SDO List.Set Heartbeat Producer.AbortIfError = FALSE; SDO List.Set Heartbeat Producer.JumpToLine = FALSE; SDO List.Set Heartbeat Producer.Line = 0; SDO List.Disable PDO.Index = 16#1400; SDO List.Disable PDO.Subindex = 16#01; SDO List.Disable PDO.Value = 16#C000020C; SDO List.Disable PDO.Size = 32; SDO List.Disable PDO.AbortIfError = FALSE; SDO List.Disable PDO.JumpToLine = FALSE; SDO List.Disable PDO.Line = 0; SDO List.Set transmission type.Index = 16#1400; SDO List.Set transmission type.Subindex = 16#02; SDO List.Set transmission type.Value = 16#FF; SDO List.Set transmission type.Size = 8; SDO List.Set transmission type.AbortIfError = FALSE; SDO List.Set transmission type.JumpToLine = FALSE; SDO List.Set transmission type.Line = 0; SDO List.Clear pdo mapping.Index = 16#1600; SDO List.Clear pdo mapping.Subindex = 16#00; SDO List.Clear pdo mapping.Value = 16#0; SDO List.Clear pdo mapping.Size = 8; SDO List.Clear pdo mapping.AbortIfError = FALSE; SDO List.Clear pdo mapping.JumpToLine = FALSE; SDO List.Clear pdo mapping.Line = 0; SDO List.Set Mapping.Index = 16#1600; SDO List.Set Mapping.Subindex = 16#01; SDO List.Set Mapping.Value = 16#60400010; SDO List.Set Mapping.Size = 32;
              SDO List.Set Mapping.AbortIfError = FALSE; SDO List.Set Mapping.JumpToLine = FALSE; SDO List.Set Mapping.Line = 0; SDO List.Set Mapping.Index = 16#1600; SDO List.Set Mapping.Subindex = 16#02; SDO List.Set Mapping.Value = 16#31500010; SDO List.Set Mapping.Size = 32; SDO List.Set Mapping.AbortIfError = FALSE; SDO List.Set Mapping.JumpToLine = FALSE; SDO List.Set Mapping.Line = 0; SDO List.Set Mapping.Index = 16#1600; SDO List.Set Mapping.Subindex = 16#03; SDO List.Set Mapping.Value = 16#60600008; SDO List.Set Mapping.Size = 32; SDO List.Set Mapping.AbortIfError = FALSE; SDO List.Set Mapping.JumpToLine = FALSE; SDO List.Set Mapping.Line = 0; SDO List.Set number of pdos.Index = 16#1600; SDO List.Set number of pdos.Subindex = 16#00; SDO List.Set number of pdos.Value = 16#03; SDO List.Set number of pdos.Size = 8; SDO List.Set number of pdos.AbortIfError = FALSE; SDO List.Set number of pdos.JumpToLine = FALSE; SDO List.Set number of pdos.Line = 0; SDO List.Set and enable COB-ID.Index = 16#1400; SDO List.Set and enable COB-ID.Subindex = 16#01; SDO List.Set and enable COB-ID.Value = 16#4000020C; SDO List.Set and enable COB-ID.Size = 32; SDO List.Set and enable COB-ID.AbortIfError = FALSE; SDO List.Set and enable COB-ID.JumpToLine = FALSE; SDO List.Set and enable COB-ID.Line = 0; SDO List.Disable PDO.Index = 16#1401; SDO List.Disable PDO.Subindex = 16#01; SDO List.Disable PDO.Value = 16#C000030C; SDO List.Disable PDO.Size = 32; SDO List.Disable PDO.AbortIfError = FALSE; SDO List.Disable PDO.JumpToLine = FALSE; SDO List.Disable PDO.Line = 0; SDO List.Set transmission type.Index = 16#1401; SDO List.Set transmission type.Subindex = 16#02;
              SDO List.Set transmission type.Value = 16#FF; SDO List.Set transmission type.Size = 8; SDO List.Set transmission type.AbortIfError = FALSE; SDO List.Set transmission type.JumpToLine = FALSE; SDO List.Set transmission type.Line = 0; SDO List.Clear pdo mapping.Index = 16#1601; SDO List.Clear pdo mapping.Subindex = 16#00; SDO List.Clear pdo mapping.Value = 16#0; SDO List.Clear pdo mapping.Size = 8; SDO List.Clear pdo mapping.AbortIfError = FALSE; SDO List.Clear pdo mapping.JumpToLine = FALSE; SDO List.Clear pdo mapping.Line = 0; SDO List.Set Mapping.Index = 16#1601; SDO List.Set Mapping.Subindex = 16#01; SDO List.Set Mapping.Value = 16#607A0020; SDO List.Set Mapping.Size = 32; SDO List.Set Mapping.AbortIfError = FALSE; SDO List.Set Mapping.JumpToLine = FALSE; SDO List.Set Mapping.Line = 0; SDO List.Set Mapping.Index = 16#1601; SDO List.Set Mapping.Subindex = 16#02; SDO List.Set Mapping.Value = 16#60FF0020; SDO List.Set Mapping.Size = 32; SDO List.Set Mapping.AbortIfError = FALSE; SDO List.Set Mapping.JumpToLine = FALSE; SDO List.Set Mapping.Line = 0; SDO List.Set number of pdos.Index = 16#1601; SDO List.Set number of pdos.Subindex = 16#00; SDO List.Set number of pdos.Value = 16#02; SDO List.Set number of pdos.Size = 8; SDO List.Set number of pdos.AbortIfError = FALSE; SDO List.Set number of pdos.JumpToLine = FALSE; SDO List.Set number of pdos.Line = 0; SDO List.Set and enable COB-ID.Index = 16#1401; SDO List.Set and enable COB-ID.Subindex = 16#01; SDO List.Set and enable COB-ID.Value = 16#4000030C; SDO List.Set and enable COB-ID.Size = 32; SDO List.Set and enable COB-ID.AbortIfError = FALSE; SDO List.Set and enable COB-ID.JumpToLine = FALSE; SDO List.Set and enable COB-ID.Line = 0;
              SDO List.Disable PDO.Index = 16#1402; SDO List.Disable PDO.Subindex = 16#01; SDO List.Disable PDO.Value = 16#C000040C; SDO List.Disable PDO.Size = 32; SDO List.Disable PDO.AbortIfError = FALSE; SDO List.Disable PDO.JumpToLine = FALSE; SDO List.Disable PDO.Line = 0; SDO List.Disable PDO.Index = 16#1403; SDO List.Disable PDO.Subindex = 16#01; SDO List.Disable PDO.Value = 16#C000050C; SDO List.Disable PDO.Size = 32; SDO List.Disable PDO.AbortIfError = FALSE; SDO List.Disable PDO.JumpToLine = FALSE; SDO List.Disable PDO.Line = 0; SDO List.Disable PDO.Index = 16#1800; SDO List.Disable PDO.Subindex = 16#01; SDO List.Disable PDO.Value = 16#8000018C; SDO List.Disable PDO.Size = 32; SDO List.Disable PDO.AbortIfError = FALSE; SDO List.Disable PDO.JumpToLine = FALSE; SDO List.Disable PDO.Line = 0; SDO List.Set transmission type.Index = 16#1800; SDO List.Set transmission type.Subindex = 16#02; SDO List.Set transmission type.Value = 16#FF; SDO List.Set transmission type.Size = 8; SDO List.Set transmission type.AbortIfError = FALSE; SDO List.Set transmission type.JumpToLine = FALSE; SDO List.Set transmission type.Line = 0; SDO List.Set inhibit time.Index = 16#1800; SDO List.Set inhibit time.Subindex = 16#03; SDO List.Set inhibit time.Value = 16#03E8; SDO List.Set inhibit time.Size = 16; SDO List.Set inhibit time.AbortIfError = FALSE; SDO List.Set inhibit time.JumpToLine = FALSE; SDO List.Set inhibit time.Line = 0; SDO List.Set event time.Index = 16#1800; SDO List.Set event time.Subindex = 16#05; SDO List.Set event time.Value = 16#03E8; SDO List.Set event time.Size = 16; SDO List.Set event time.AbortIfError = FALSE;
              SDO List.Set event time.JumpToLine = FALSE; SDO List.Set event time.Line = 0; SDO List.Clear pdo mapping.Index = 16#1A00; SDO List.Clear pdo mapping.Subindex = 16#00; SDO List.Clear pdo mapping.Value = 16#0; SDO List.Clear pdo mapping.Size = 8; SDO List.Clear pdo mapping.AbortIfError = FALSE; SDO List.Clear pdo mapping.JumpToLine = FALSE; SDO List.Clear pdo mapping.Line = 0; SDO List.Set Mapping.Index = 16#1A00; SDO List.Set Mapping.Subindex = 16#01; SDO List.Set Mapping.Value = 16#60410010; SDO List.Set Mapping.Size = 32; SDO List.Set Mapping.AbortIfError = FALSE; SDO List.Set Mapping.JumpToLine = FALSE; SDO List.Set Mapping.Line = 0; SDO List.Set Mapping.Index = 16#1A00; SDO List.Set Mapping.Subindex = 16#02; SDO List.Set Mapping.Value = 16#60610008; SDO List.Set Mapping.Size = 32; SDO List.Set Mapping.AbortIfError = FALSE; SDO List.Set Mapping.JumpToLine = FALSE; SDO List.Set Mapping.Line = 0; SDO List.Set Mapping.Index = 16#1A00; SDO List.Set Mapping.Subindex = 16#03; SDO List.Set Mapping.Value = 16#60780010; SDO List.Set Mapping.Size = 32; SDO List.Set Mapping.AbortIfError = FALSE; SDO List.Set Mapping.JumpToLine = FALSE; SDO List.Set Mapping.Line = 0; SDO List.Set Mapping.Index = 16#1A00; SDO List.Set Mapping.Subindex = 16#04; SDO List.Set Mapping.Value = 16#60770010; SDO List.Set Mapping.Size = 32; SDO List.Set Mapping.AbortIfError = FALSE; SDO List.Set Mapping.JumpToLine = FALSE; SDO List.Set Mapping.Line = 0; SDO List.Set number of pdos.Index = 16#1A00; SDO List.Set number of pdos.Subindex = 16#00; SDO List.Set number of pdos.Value = 16#04;
              SDO List.Set number of pdos.Size = 8; SDO List.Set number of pdos.AbortIfError = FALSE; SDO List.Set number of pdos.JumpToLine = FALSE; SDO List.Set number of pdos.Line = 0; SDO List.Set and enable COB-ID.Index = 16#1800; SDO List.Set and enable COB-ID.Subindex = 16#01; SDO List.Set and enable COB-ID.Value = 16#0000018C; SDO List.Set and enable COB-ID.Size = 32; SDO List.Set and enable COB-ID.AbortIfError = FALSE; SDO List.Set and enable COB-ID.JumpToLine = FALSE; SDO List.Set and enable COB-ID.Line = 0; SDO List.Disable PDO.Index = 16#1801; SDO List.Disable PDO.Subindex = 16#01; SDO List.Disable PDO.Value = 16#8000028C; SDO List.Disable PDO.Size = 32; SDO List.Disable PDO.AbortIfError = FALSE; SDO List.Disable PDO.JumpToLine = FALSE; SDO List.Disable PDO.Line = 0; SDO List.Set transmission type.Index = 16#1801; SDO List.Set transmission type.Subindex = 16#02; SDO List.Set transmission type.Value = 16#FF; SDO List.Set transmission type.Size = 8; SDO List.Set transmission type.AbortIfError = FALSE; SDO List.Set transmission type.JumpToLine = FALSE; SDO List.Set transmission type.Line = 0; SDO List.Set inhibit time.Index = 16#1801; SDO List.Set inhibit time.Subindex = 16#03; SDO List.Set inhibit time.Value = 16#03E8; SDO List.Set inhibit time.Size = 16; SDO List.Set inhibit time.AbortIfError = FALSE; SDO List.Set inhibit time.JumpToLine = FALSE; SDO List.Set inhibit time.Line = 0; SDO List.Clear pdo mapping.Index = 16#1A01; SDO List.Clear pdo mapping.Subindex = 16#00; SDO List.Clear pdo mapping.Value = 16#0; SDO List.Clear pdo mapping.Size = 8; SDO List.Clear pdo mapping.AbortIfError = FALSE; SDO List.Clear pdo mapping.JumpToLine = FALSE; SDO List.Clear pdo mapping.Line = 0; SDO List.Set Mapping.Index = 16#1A01;
              SDO List.Set Mapping.Subindex = 16#01; SDO List.Set Mapping.Value = 16#60640020; SDO List.Set Mapping.Size = 32; SDO List.Set Mapping.AbortIfError = FALSE; SDO List.Set Mapping.JumpToLine = FALSE; SDO List.Set Mapping.Line = 0; SDO List.Set Mapping.Index = 16#1A01; SDO List.Set Mapping.Subindex = 16#02; SDO List.Set Mapping.Value = 16#606C0020; SDO List.Set Mapping.Size = 32; SDO List.Set Mapping.AbortIfError = FALSE; SDO List.Set Mapping.JumpToLine = FALSE; SDO List.Set Mapping.Line = 0; SDO List.Set number of pdos.Index = 16#1A01; SDO List.Set number of pdos.Subindex = 16#00; SDO List.Set number of pdos.Value = 16#02; SDO List.Set number of pdos.Size = 8; SDO List.Set number of pdos.AbortIfError = FALSE; SDO List.Set number of pdos.JumpToLine = FALSE; SDO List.Set number of pdos.Line = 0; SDO List.Set and enable COB-ID.Index = 16#1801; SDO List.Set and enable COB-ID.Subindex = 16#01; SDO List.Set and enable COB-ID.Value = 16#0000028C; SDO List.Set and enable COB-ID.Size = 32; SDO List.Set and enable COB-ID.AbortIfError = FALSE; SDO List.Set and enable COB-ID.JumpToLine = FALSE; SDO List.Set and enable COB-ID.Line = 0; SDO List.Disable PDO.Index = 16#1802; SDO List.Disable PDO.Subindex = 16#01; SDO List.Disable PDO.Value = 16#8000038C; SDO List.Disable PDO.Size = 32; SDO List.Disable PDO.AbortIfError = FALSE; SDO List.Disable PDO.JumpToLine = FALSE; SDO List.Disable PDO.Line = 0; SDO List.Disable PDO.Index = 16#1803; SDO List.Disable PDO.Subindex = 16#01; SDO List.Disable PDO.Value = 16#8000048C; SDO List.Disable PDO.Size = 32; SDO List.Disable PDO.AbortIfError = FALSE; SDO List.Disable PDO.JumpToLine = FALSE;
              SDO List.Disable PDO.Line = 0; ConfigVersion = 50659584
            unmapped channels: Controlword, Brake, Modes of operation, Target position, Target velocity, Statusword, Modes of operation display, Current actual value, Torque actual value, Position actual value, Velocity actual value
        BG75ci_0D : BG75ci, Dunkermotoren GmbH, order no. 0, version Revision=16#00000001, FileVersion=2.20, File=Dunker_BG75ci.eds
            settings: NODEIDSAVED = 13; SDO Timeout = 1000000; EXPERTSETTINGS = True; Emergency-General Parameters.Emergency COBID = 16#8D; Heartbeat-Producer Time = 3000; PDO 16#1400.COBID = 16#4000020D; PDO 16#1401.COBID = 16#4000030D; PDO 16#1402.COBID = 16#C000040D; PDO 16#1403.COBID = 16#C000050D; PDO 16#1404.COBID = 16#C0000000; Generic COBID = '16#C0000000'; PDO 16#1405.COBID = 16#C0000000; Generic COBID = '16#C0000000'; PDO 16#1406.COBID = 16#C0000000; Generic COBID = '16#C0000000'; PDO 16#1414.COBID = 16#C0000000; Generic COBID = '16#C0000000'; PDO 16#1800.COBID = 16#018D; PDO 16#1800.Inhibit Time = 1000; PDO 16#1800.Event Timer = 1000; PDO 16#1801.COBID = 16#028D; PDO 16#1801.Inhibit Time = 1000; PDO 16#1801.Event Timer = 1000; PDO 16#1802.COBID = 16#8000038D; PDO 16#1802.Event Timer = 0; PDO 16#1803.COBID = 16#8000048D; PDO 16#1803.Event Timer = 0; PDO 16#1804.Event Timer = 0; PDO 16#1805.Event Timer = 0; PDO 16#1806.Event Timer = 0; PDO 16#1814.Event Timer = 0; Heartbeat-Consuming1.Heartbeat-Time = 4500 ms; Controlword.Index = 16#6040; Controlword.Subindex = 16#00; Controlword.ObjectLength = 16; Brake.Index = 16#3150; Brake.Subindex = 16#00; Brake.ObjectLength = 16; Modes of operation.Index = 16#6060; Modes of operation.Subindex = 16#00;
              Modes of operation.ObjectLength = 8; Target position.Index = 16#607A; Target position.Subindex = 16#00; Target position.ObjectLength = 32; Target velocity.Index = 16#60FF; Target velocity.Subindex = 16#00; Target velocity.ObjectLength = 32; Statusword.Index = 16#6041; Statusword.Subindex = 16#00; Statusword.ObjectLength = 16; Modes of operation display.Index = 16#6061; Modes of operation display.Subindex = 16#00; Modes of operation display.ObjectLength = 8; Current actual value.Index = 16#6078; Current actual value.Subindex = 16#00; Current actual value.ObjectLength = 16; Torque actual value.Index = 16#6077; Torque actual value.Subindex = 16#00; Torque actual value.ObjectLength = 16; Position actual value.Index = 16#6064; Position actual value.Subindex = 16#00; Position actual value.ObjectLength = 32; Velocity actual value.Index = 16#606C; Velocity actual value.Subindex = 16#00; Velocity actual value.ObjectLength = 32; SDO List.Disable TIME.Index = 16#1012; SDO List.Disable TIME.Subindex = 16#00; SDO List.Disable TIME.Value = 16#00000100; SDO List.Disable TIME.Size = 32; SDO List.Disable TIME.AbortIfError = FALSE; SDO List.Disable TIME.JumpToLine = FALSE; SDO List.Disable TIME.Line = 0; SDO List.Set Guardtime.Index = 16#100C; SDO List.Set Guardtime.Subindex = 16#00; SDO List.Set Guardtime.Value = 16#00000000; SDO List.Set Guardtime.Size = 16; SDO List.Set Guardtime.AbortIfError = FALSE; SDO List.Set Guardtime.JumpToLine = FALSE; SDO List.Set Guardtime.Line = 0; SDO List.Set Lifetime.Index = 16#100D;
              SDO List.Set Lifetime.Subindex = 16#00; SDO List.Set Lifetime.Value = 16#00000000; SDO List.Set Lifetime.Size = 8; SDO List.Set Lifetime.AbortIfError = FALSE; SDO List.Set Lifetime.JumpToLine = FALSE; SDO List.Set Lifetime.Line = 0; SDO List.Disable Emcy CobID.Index = 16#1014; SDO List.Disable Emcy CobID.Subindex = 16#00; SDO List.Disable Emcy CobID.Value = 16#8000008D; SDO List.Disable Emcy CobID.Size = 32; SDO List.Disable Emcy CobID.AbortIfError = FALSE; SDO List.Disable Emcy CobID.JumpToLine = FALSE; SDO List.Disable Emcy CobID.Line = 0; SDO List.Set Emcy CobID.Index = 16#1014; SDO List.Set Emcy CobID.Subindex = 16#00; SDO List.Set Emcy CobID.Value = 16#0000008D; SDO List.Set Emcy CobID.Size = 32; SDO List.Set Emcy CobID.AbortIfError = FALSE; SDO List.Set Emcy CobID.JumpToLine = FALSE; SDO List.Set Emcy CobID.Line = 0; SDO List.Set Heartbeat Consumer.Index = 16#1016; SDO List.Set Heartbeat Consumer.Subindex = 16#01; SDO List.Set Heartbeat Consumer.Value = 16#00011194; SDO List.Set Heartbeat Consumer.Size = 32; SDO List.Set Heartbeat Consumer.AbortIfError = FALSE; SDO List.Set Heartbeat Consumer.JumpToLine = FALSE; SDO List.Set Heartbeat Consumer.Line = 0; SDO List.Set Heartbeat Consumer.Index = 16#1016; SDO List.Set Heartbeat Consumer.Subindex = 16#02; SDO List.Set Heartbeat Consumer.Value = 0; SDO List.Set Heartbeat Consumer.Size = 32; SDO List.Set Heartbeat Consumer.AbortIfError = FALSE; SDO List.Set Heartbeat Consumer.JumpToLine = FALSE; SDO List.Set Heartbeat Consumer.Line = 0; SDO List.Set Heartbeat Consumer.Index = 16#1016; SDO List.Set Heartbeat Consumer.Subindex = 16#03; SDO List.Set Heartbeat Consumer.Value = 0; SDO List.Set Heartbeat Consumer.Size = 32; SDO List.Set Heartbeat Consumer.AbortIfError = FALSE; SDO List.Set Heartbeat Consumer.JumpToLine = FALSE;
              SDO List.Set Heartbeat Consumer.Line = 0; SDO List.Set Heartbeat Consumer.Index = 16#1016; SDO List.Set Heartbeat Consumer.Subindex = 16#04; SDO List.Set Heartbeat Consumer.Value = 0; SDO List.Set Heartbeat Consumer.Size = 32; SDO List.Set Heartbeat Consumer.AbortIfError = FALSE; SDO List.Set Heartbeat Consumer.JumpToLine = FALSE; SDO List.Set Heartbeat Consumer.Line = 0; SDO List.Set Heartbeat Producer.Index = 16#1017; SDO List.Set Heartbeat Producer.Subindex = 16#00; SDO List.Set Heartbeat Producer.Value = 16#00000BB8; SDO List.Set Heartbeat Producer.Size = 16; SDO List.Set Heartbeat Producer.AbortIfError = FALSE; SDO List.Set Heartbeat Producer.JumpToLine = FALSE; SDO List.Set Heartbeat Producer.Line = 0; SDO List.Disable PDO.Index = 16#1400; SDO List.Disable PDO.Subindex = 16#01; SDO List.Disable PDO.Value = 16#C000020D; SDO List.Disable PDO.Size = 32; SDO List.Disable PDO.AbortIfError = FALSE; SDO List.Disable PDO.JumpToLine = FALSE; SDO List.Disable PDO.Line = 0; SDO List.Set transmission type.Index = 16#1400; SDO List.Set transmission type.Subindex = 16#02; SDO List.Set transmission type.Value = 16#FF; SDO List.Set transmission type.Size = 8; SDO List.Set transmission type.AbortIfError = FALSE; SDO List.Set transmission type.JumpToLine = FALSE; SDO List.Set transmission type.Line = 0; SDO List.Clear pdo mapping.Index = 16#1600; SDO List.Clear pdo mapping.Subindex = 16#00; SDO List.Clear pdo mapping.Value = 16#0; SDO List.Clear pdo mapping.Size = 8; SDO List.Clear pdo mapping.AbortIfError = FALSE; SDO List.Clear pdo mapping.JumpToLine = FALSE; SDO List.Clear pdo mapping.Line = 0; SDO List.Set Mapping.Index = 16#1600; SDO List.Set Mapping.Subindex = 16#01; SDO List.Set Mapping.Value = 16#60400010; SDO List.Set Mapping.Size = 32;
              SDO List.Set Mapping.AbortIfError = FALSE; SDO List.Set Mapping.JumpToLine = FALSE; SDO List.Set Mapping.Line = 0; SDO List.Set Mapping.Index = 16#1600; SDO List.Set Mapping.Subindex = 16#02; SDO List.Set Mapping.Value = 16#31500010; SDO List.Set Mapping.Size = 32; SDO List.Set Mapping.AbortIfError = FALSE; SDO List.Set Mapping.JumpToLine = FALSE; SDO List.Set Mapping.Line = 0; SDO List.Set Mapping.Index = 16#1600; SDO List.Set Mapping.Subindex = 16#03; SDO List.Set Mapping.Value = 16#60600008; SDO List.Set Mapping.Size = 32; SDO List.Set Mapping.AbortIfError = FALSE; SDO List.Set Mapping.JumpToLine = FALSE; SDO List.Set Mapping.Line = 0; SDO List.Set number of pdos.Index = 16#1600; SDO List.Set number of pdos.Subindex = 16#00; SDO List.Set number of pdos.Value = 16#03; SDO List.Set number of pdos.Size = 8; SDO List.Set number of pdos.AbortIfError = FALSE; SDO List.Set number of pdos.JumpToLine = FALSE; SDO List.Set number of pdos.Line = 0; SDO List.Set and enable COB-ID.Index = 16#1400; SDO List.Set and enable COB-ID.Subindex = 16#01; SDO List.Set and enable COB-ID.Value = 16#4000020D; SDO List.Set and enable COB-ID.Size = 32; SDO List.Set and enable COB-ID.AbortIfError = FALSE; SDO List.Set and enable COB-ID.JumpToLine = FALSE; SDO List.Set and enable COB-ID.Line = 0; SDO List.Disable PDO.Index = 16#1401; SDO List.Disable PDO.Subindex = 16#01; SDO List.Disable PDO.Value = 16#C000030D; SDO List.Disable PDO.Size = 32; SDO List.Disable PDO.AbortIfError = FALSE; SDO List.Disable PDO.JumpToLine = FALSE; SDO List.Disable PDO.Line = 0; SDO List.Set transmission type.Index = 16#1401; SDO List.Set transmission type.Subindex = 16#02;
              SDO List.Set transmission type.Value = 16#FF; SDO List.Set transmission type.Size = 8; SDO List.Set transmission type.AbortIfError = FALSE; SDO List.Set transmission type.JumpToLine = FALSE; SDO List.Set transmission type.Line = 0; SDO List.Clear pdo mapping.Index = 16#1601; SDO List.Clear pdo mapping.Subindex = 16#00; SDO List.Clear pdo mapping.Value = 16#0; SDO List.Clear pdo mapping.Size = 8; SDO List.Clear pdo mapping.AbortIfError = FALSE; SDO List.Clear pdo mapping.JumpToLine = FALSE; SDO List.Clear pdo mapping.Line = 0; SDO List.Set Mapping.Index = 16#1601; SDO List.Set Mapping.Subindex = 16#01; SDO List.Set Mapping.Value = 16#607A0020; SDO List.Set Mapping.Size = 32; SDO List.Set Mapping.AbortIfError = FALSE; SDO List.Set Mapping.JumpToLine = FALSE; SDO List.Set Mapping.Line = 0; SDO List.Set Mapping.Index = 16#1601; SDO List.Set Mapping.Subindex = 16#02; SDO List.Set Mapping.Value = 16#60FF0020; SDO List.Set Mapping.Size = 32; SDO List.Set Mapping.AbortIfError = FALSE; SDO List.Set Mapping.JumpToLine = FALSE; SDO List.Set Mapping.Line = 0; SDO List.Set number of pdos.Index = 16#1601; SDO List.Set number of pdos.Subindex = 16#00; SDO List.Set number of pdos.Value = 16#02; SDO List.Set number of pdos.Size = 8; SDO List.Set number of pdos.AbortIfError = FALSE; SDO List.Set number of pdos.JumpToLine = FALSE; SDO List.Set number of pdos.Line = 0; SDO List.Set and enable COB-ID.Index = 16#1401; SDO List.Set and enable COB-ID.Subindex = 16#01; SDO List.Set and enable COB-ID.Value = 16#4000030D; SDO List.Set and enable COB-ID.Size = 32; SDO List.Set and enable COB-ID.AbortIfError = FALSE; SDO List.Set and enable COB-ID.JumpToLine = FALSE; SDO List.Set and enable COB-ID.Line = 0;
              SDO List.Disable PDO.Index = 16#1402; SDO List.Disable PDO.Subindex = 16#01; SDO List.Disable PDO.Value = 16#C000040D; SDO List.Disable PDO.Size = 32; SDO List.Disable PDO.AbortIfError = FALSE; SDO List.Disable PDO.JumpToLine = FALSE; SDO List.Disable PDO.Line = 0; SDO List.Disable PDO.Index = 16#1403; SDO List.Disable PDO.Subindex = 16#01; SDO List.Disable PDO.Value = 16#C000050D; SDO List.Disable PDO.Size = 32; SDO List.Disable PDO.AbortIfError = FALSE; SDO List.Disable PDO.JumpToLine = FALSE; SDO List.Disable PDO.Line = 0; SDO List.Disable PDO.Index = 16#1800; SDO List.Disable PDO.Subindex = 16#01; SDO List.Disable PDO.Value = 16#8000018D; SDO List.Disable PDO.Size = 32; SDO List.Disable PDO.AbortIfError = FALSE; SDO List.Disable PDO.JumpToLine = FALSE; SDO List.Disable PDO.Line = 0; SDO List.Set transmission type.Index = 16#1800; SDO List.Set transmission type.Subindex = 16#02; SDO List.Set transmission type.Value = 16#FF; SDO List.Set transmission type.Size = 8; SDO List.Set transmission type.AbortIfError = FALSE; SDO List.Set transmission type.JumpToLine = FALSE; SDO List.Set transmission type.Line = 0; SDO List.Set inhibit time.Index = 16#1800; SDO List.Set inhibit time.Subindex = 16#03; SDO List.Set inhibit time.Value = 16#03E8; SDO List.Set inhibit time.Size = 16; SDO List.Set inhibit time.AbortIfError = FALSE; SDO List.Set inhibit time.JumpToLine = FALSE; SDO List.Set inhibit time.Line = 0; SDO List.Set event time.Index = 16#1800; SDO List.Set event time.Subindex = 16#05; SDO List.Set event time.Value = 16#03E8; SDO List.Set event time.Size = 16; SDO List.Set event time.AbortIfError = FALSE;
              SDO List.Set event time.JumpToLine = FALSE; SDO List.Set event time.Line = 0; SDO List.Clear pdo mapping.Index = 16#1A00; SDO List.Clear pdo mapping.Subindex = 16#00; SDO List.Clear pdo mapping.Value = 16#0; SDO List.Clear pdo mapping.Size = 8; SDO List.Clear pdo mapping.AbortIfError = FALSE; SDO List.Clear pdo mapping.JumpToLine = FALSE; SDO List.Clear pdo mapping.Line = 0; SDO List.Set Mapping.Index = 16#1A00; SDO List.Set Mapping.Subindex = 16#01; SDO List.Set Mapping.Value = 16#60410010; SDO List.Set Mapping.Size = 32; SDO List.Set Mapping.AbortIfError = FALSE; SDO List.Set Mapping.JumpToLine = FALSE; SDO List.Set Mapping.Line = 0; SDO List.Set Mapping.Index = 16#1A00; SDO List.Set Mapping.Subindex = 16#02; SDO List.Set Mapping.Value = 16#60610008; SDO List.Set Mapping.Size = 32; SDO List.Set Mapping.AbortIfError = FALSE; SDO List.Set Mapping.JumpToLine = FALSE; SDO List.Set Mapping.Line = 0; SDO List.Set Mapping.Index = 16#1A00; SDO List.Set Mapping.Subindex = 16#03; SDO List.Set Mapping.Value = 16#60780010; SDO List.Set Mapping.Size = 32; SDO List.Set Mapping.AbortIfError = FALSE; SDO List.Set Mapping.JumpToLine = FALSE; SDO List.Set Mapping.Line = 0; SDO List.Set Mapping.Index = 16#1A00; SDO List.Set Mapping.Subindex = 16#04; SDO List.Set Mapping.Value = 16#60770010; SDO List.Set Mapping.Size = 32; SDO List.Set Mapping.AbortIfError = FALSE; SDO List.Set Mapping.JumpToLine = FALSE; SDO List.Set Mapping.Line = 0; SDO List.Set number of pdos.Index = 16#1A00; SDO List.Set number of pdos.Subindex = 16#00; SDO List.Set number of pdos.Value = 16#04;
              SDO List.Set number of pdos.Size = 8; SDO List.Set number of pdos.AbortIfError = FALSE; SDO List.Set number of pdos.JumpToLine = FALSE; SDO List.Set number of pdos.Line = 0; SDO List.Set and enable COB-ID.Index = 16#1800; SDO List.Set and enable COB-ID.Subindex = 16#01; SDO List.Set and enable COB-ID.Value = 16#0000018D; SDO List.Set and enable COB-ID.Size = 32; SDO List.Set and enable COB-ID.AbortIfError = FALSE; SDO List.Set and enable COB-ID.JumpToLine = FALSE; SDO List.Set and enable COB-ID.Line = 0; SDO List.Disable PDO.Index = 16#1801; SDO List.Disable PDO.Subindex = 16#01; SDO List.Disable PDO.Value = 16#8000028D; SDO List.Disable PDO.Size = 32; SDO List.Disable PDO.AbortIfError = FALSE; SDO List.Disable PDO.JumpToLine = FALSE; SDO List.Disable PDO.Line = 0; SDO List.Set transmission type.Index = 16#1801; SDO List.Set transmission type.Subindex = 16#02; SDO List.Set transmission type.Value = 16#FF; SDO List.Set transmission type.Size = 8; SDO List.Set transmission type.AbortIfError = FALSE; SDO List.Set transmission type.JumpToLine = FALSE; SDO List.Set transmission type.Line = 0; SDO List.Set inhibit time.Index = 16#1801; SDO List.Set inhibit time.Subindex = 16#03; SDO List.Set inhibit time.Value = 16#03E8; SDO List.Set inhibit time.Size = 16; SDO List.Set inhibit time.AbortIfError = FALSE; SDO List.Set inhibit time.JumpToLine = FALSE; SDO List.Set inhibit time.Line = 0; SDO List.Clear pdo mapping.Index = 16#1A01; SDO List.Clear pdo mapping.Subindex = 16#00; SDO List.Clear pdo mapping.Value = 16#0; SDO List.Clear pdo mapping.Size = 8; SDO List.Clear pdo mapping.AbortIfError = FALSE; SDO List.Clear pdo mapping.JumpToLine = FALSE; SDO List.Clear pdo mapping.Line = 0; SDO List.Set Mapping.Index = 16#1A01;
              SDO List.Set Mapping.Subindex = 16#01; SDO List.Set Mapping.Value = 16#60640020; SDO List.Set Mapping.Size = 32; SDO List.Set Mapping.AbortIfError = FALSE; SDO List.Set Mapping.JumpToLine = FALSE; SDO List.Set Mapping.Line = 0; SDO List.Set Mapping.Index = 16#1A01; SDO List.Set Mapping.Subindex = 16#02; SDO List.Set Mapping.Value = 16#606C0020; SDO List.Set Mapping.Size = 32; SDO List.Set Mapping.AbortIfError = FALSE; SDO List.Set Mapping.JumpToLine = FALSE; SDO List.Set Mapping.Line = 0; SDO List.Set number of pdos.Index = 16#1A01; SDO List.Set number of pdos.Subindex = 16#00; SDO List.Set number of pdos.Value = 16#02; SDO List.Set number of pdos.Size = 8; SDO List.Set number of pdos.AbortIfError = FALSE; SDO List.Set number of pdos.JumpToLine = FALSE; SDO List.Set number of pdos.Line = 0; SDO List.Set and enable COB-ID.Index = 16#1801; SDO List.Set and enable COB-ID.Subindex = 16#01; SDO List.Set and enable COB-ID.Value = 16#0000028D; SDO List.Set and enable COB-ID.Size = 32; SDO List.Set and enable COB-ID.AbortIfError = FALSE; SDO List.Set and enable COB-ID.JumpToLine = FALSE; SDO List.Set and enable COB-ID.Line = 0; SDO List.Disable PDO.Index = 16#1802; SDO List.Disable PDO.Subindex = 16#01; SDO List.Disable PDO.Value = 16#8000038D; SDO List.Disable PDO.Size = 32; SDO List.Disable PDO.AbortIfError = FALSE; SDO List.Disable PDO.JumpToLine = FALSE; SDO List.Disable PDO.Line = 0; SDO List.Disable PDO.Index = 16#1803; SDO List.Disable PDO.Subindex = 16#01; SDO List.Disable PDO.Value = 16#8000048D; SDO List.Disable PDO.Size = 32; SDO List.Disable PDO.AbortIfError = FALSE; SDO List.Disable PDO.JumpToLine = FALSE;
              SDO List.Disable PDO.Line = 0; ConfigVersion = 50659584
            unmapped channels: Controlword, Brake, Modes of operation, Target position, Target velocity, Statusword, Modes of operation display, Current actual value, Torque actual value, Position actual value, Velocity actual value
        Joystick_SD6000 : Joystick, Sauer-Danfoss, order no. 0, version Revision=16#00010001, FileVersion=1.1, File=Sauer-Danfoss JS6000 Joystick.eds
            settings: NODEIDSAVED = 2; SDO Timeout = 1000000; EXPERTSETTINGS = True; Emergency-General Parameters.Emergency COBID = 16#82; Heartbeat-Producer Time = 3000; PDO 16#1800.COBID = 16#0182; PDO 16#1801.COBID = 16#0282; PDO 16#1802.COBID = 16#40000382; Generic COBID = '16#40000382'; PDO 16#1803.COBID = 16#0482; Freeze Status.Subindex = 16#01; Button 1 to 8.Subindex = 16#02; Button 9 to 16.Subindex = 16#03; Button 17 to 24.Subindex = 16#04; Button 25 to 32.Subindex = 16#05; Proportional 1.Subindex = 16#01; Proportional 2.Subindex = 16#02; Proportional 3.Subindex = 16#03; Proportional 6.Subindex = 16#06; SDO List.Set Heartbeat Producer.Index = 16#1017; SDO List.Set Heartbeat Producer.Subindex = 16#00; SDO List.Set Heartbeat Producer.Value = 16#00000BB8; SDO List.Set Heartbeat Producer.Size = 16; SDO List.Set Heartbeat Producer.AbortIfError = FALSE; SDO List.Set Heartbeat Producer.JumpToLine = FALSE; SDO List.Set Heartbeat Producer.Line = 0; ConfigVersion = 50659584
            unmapped channels: Freeze Status, Button 1 to 8, Button 9 to 16, Button 17 to 24, Button 25 to 32, Proportional 1, Proportional 2, Proportional 3, Proportional 4, Proportional 6, Proportional 7, Proportional 8
        microCAN4aiBOX : µCAN.4.ai-BOX, MicroControl GmbH & Co. KG, order no. 12.44.001, version Revision=16#0302040A, FileVersion=1.1, File=mcan4aiv_box.eds
            settings: General Options.Reset Node = FALSE; NODEIDSAVED = 16; SDO Timeout = 1000000; EXPERTSETTINGS = True; Emergency-General Parameters.Emergency COBID = 16#90; Heartbeat-Producer Time = 3000; PDO 16#1800.COBID = 16#C0000190; PDO 16#1801.COBID = 16#C0000290; Heartbeat-Consuming1.Heartbeat-Time = 4500 ms; PV Channel 1.Subindex = 16#01; PV Channel 2.Subindex = 16#02; PV Channel 3.Subindex = 16#03; PV Channel 4.Subindex = 16#04; FV Channel 1.Subindex = 16#01; FV Channel 2.Subindex = 16#02; FV Channel 3.Subindex = 16#03; FV Channel 4.Subindex = 16#04; SDO List.Set Guardtime.Index = 16#100C; SDO List.Set Guardtime.Subindex = 16#00; SDO List.Set Guardtime.Value = 16#00000000; SDO List.Set Guardtime.Size = 16; SDO List.Set Guardtime.AbortIfError = FALSE; SDO List.Set Guardtime.JumpToLine = FALSE; SDO List.Set Guardtime.Line = 0; SDO List.Set Lifetime.Index = 16#100D; SDO List.Set Lifetime.Subindex = 16#00; SDO List.Set Lifetime.Value = 16#00000000; SDO List.Set Lifetime.Size = 8; SDO List.Set Lifetime.AbortIfError = FALSE; SDO List.Set Lifetime.JumpToLine = FALSE; SDO List.Set Lifetime.Line = 0; SDO List.Disable Emcy CobID.Index = 16#1014; SDO List.Disable Emcy CobID.Subindex = 16#00; SDO List.Disable Emcy CobID.Value = 16#80000090; SDO List.Disable Emcy CobID.Size = 32; SDO List.Disable Emcy CobID.AbortIfError = FALSE; SDO List.Disable Emcy CobID.JumpToLine = FALSE; SDO List.Disable Emcy CobID.Line = 0; SDO List.Set Emcy CobID.Index = 16#1014; SDO List.Set Emcy CobID.Subindex = 16#00;
              SDO List.Set Emcy CobID.Value = 16#00000090; SDO List.Set Emcy CobID.Size = 32; SDO List.Set Emcy CobID.AbortIfError = FALSE; SDO List.Set Emcy CobID.JumpToLine = FALSE; SDO List.Set Emcy CobID.Line = 0; SDO List.Set Heartbeat Consumer.Index = 16#1016; SDO List.Set Heartbeat Consumer.Subindex = 16#01; SDO List.Set Heartbeat Consumer.Value = 16#00011194; SDO List.Set Heartbeat Consumer.Size = 32; SDO List.Set Heartbeat Consumer.AbortIfError = FALSE; SDO List.Set Heartbeat Consumer.JumpToLine = FALSE; SDO List.Set Heartbeat Consumer.Line = 0; SDO List.Set Heartbeat Consumer.Index = 16#1016; SDO List.Set Heartbeat Consumer.Subindex = 16#02; SDO List.Set Heartbeat Consumer.Value = 0; SDO List.Set Heartbeat Consumer.Size = 32; SDO List.Set Heartbeat Consumer.AbortIfError = FALSE; SDO List.Set Heartbeat Consumer.JumpToLine = FALSE; SDO List.Set Heartbeat Consumer.Line = 0; SDO List.Set Heartbeat Producer.Index = 16#1017; SDO List.Set Heartbeat Producer.Subindex = 16#00; SDO List.Set Heartbeat Producer.Value = 16#00000BB8; SDO List.Set Heartbeat Producer.Size = 16; SDO List.Set Heartbeat Producer.AbortIfError = FALSE; SDO List.Set Heartbeat Producer.JumpToLine = FALSE; SDO List.Set Heartbeat Producer.Line = 0; SDO List.Disable PDO.Index = 16#1800; SDO List.Disable PDO.Subindex = 16#01; SDO List.Disable PDO.Value = 16#C0000190; SDO List.Disable PDO.Size = 32; SDO List.Disable PDO.AbortIfError = FALSE; SDO List.Disable PDO.JumpToLine = FALSE; SDO List.Disable PDO.Line = 0; SDO List.Disable PDO.Index = 16#1801; SDO List.Disable PDO.Subindex = 16#01; SDO List.Disable PDO.Value = 16#C0000290; SDO List.Disable PDO.Size = 32; SDO List.Disable PDO.AbortIfError = FALSE; SDO List.Disable PDO.JumpToLine = FALSE; SDO List.Disable PDO.Line = 0;
              ConfigVersion = 50659584
        Baseline_S_real_time_target_machine : Baseline S real-time target machine, Speedgoat GmbH, order no. 0, version Revision=16#00000501, FileVersion=1.1, File=Speedgoat.eds
            settings: NODEIDSAVED = 5; SDO Timeout = 1000000; EXPERTSETTINGS = True; Heartbeat-Producer Time = 3000; SDO List.Set Heartbeat Producer.Index = 16#1017; SDO List.Set Heartbeat Producer.Subindex = 16#00; SDO List.Set Heartbeat Producer.Value = 16#00000BB8; SDO List.Set Heartbeat Producer.Size = 16; SDO List.Set Heartbeat Producer.AbortIfError = FALSE; SDO List.Set Heartbeat Producer.JumpToLine = FALSE; SDO List.Set Heartbeat Producer.Line = 0; ConfigVersion = 50659584
    Embedded Functions
      HSC : HSC, Schneider Electric, order no. HSC, version 3.5.3.59
      PTO_PWM : PTO_PWM, Schneider Electric, order no. PTO_PWM, version 3.5.3.59
      IO : IO, Schneider Electric, order no. IO, version 3.5.3.59
          input  Application.GVL.xButnRev : BOOL  // In.DI0
          input  Application.GVL.xButnStop : BOOL  // In.DI1
          input  Application.GVL.xButnFwd : BOOL  // In.DI2
          input  Application.GVL.xEStop : BOOL  // In.DI3
          input  Application.GVL.xDoorMain : BOOL  // In.DI4
          output Application.GVL.xGrenOperLEDon : BOOL  // Out.DQ0
          output Application.GVL.xWhitPwrLEDon : BOOL  // Out.DQ1
          output Application.GVL.xRedErrLEDon : BOOL  // Out.DQ2
          output Application.GVL.xDC_ContactorCtrl : BOOL  // Out.DQ3
          unmapped channels: In, Out
  6c0f7fb6-600b-4c93-9262-20cdc603757e
  Vijeo Designer Project Container
*)

// HMISAC/Application/GVL_Retain
VAR_GLOBAL RETAIN
	udiParaAccLXM2803		:UDINT:=64000000;	// value for profile acceleration in inc/s*s
	udiParaDecLXM2803		:UDINT:=64000000;	// value for profile deceleration in inc/s*s
	udiParaDecStopLXM2803	:UDINT:=640000000;	// value for quick stop deceleration in inc/s*s
	udiParaAccLXM2804		:UDINT:=64000000;	// value for profile acceleration in inc/s*s
	udiParaDecLXM2804		:UDINT:=64000000;	// value for profile deceleration in inc/s*s
	udiParaDecStopLXM2804	:UDINT:=640000000;	// value for quick stop deceleration in inc/s*s
END_VAR
(*
CANopen objects Lexium 28:
6083h	|	Profile Acceleration	|	UDINT	|	unit: inc/s*s
6084h	|	Profile Deceleration	|	UDINT	|	unit: inc/s*s
6085h	|	Quick Stop Deceleration	|	UDINT	|	unit: inc/s*s
Calculation example considering that, the default value for the scaling in CAN mode is 1.280.000 increments per revolution:
- number of revolutions per second: 64.000.0000 / 1.280.000 = 50 r/s*s
- acceleration in rpm/s: 50 * 60 = 3000 rpm/s
=> value 64.000.000 means an acceleration of 3000 rpm/s
*)

// HMISAC/Application/LXM28A_Node04/GVL_LXM28A_Node04
VAR_GLOBAL
	xMcbRdy			:BOOL; // Indicates the state of Motor Circuit Breaker. Mapped to the physical input where the accordingly auxiliary contact of the MCB is connected
	diActlPos		:DINT; // Indicates the actual position. Variable is mapped to TxPDO "Position actual value" of LXM28A
	diActlVelo		:DINT; // Indicates the actual velocity in rpm. Variable is mapped to TxPDO "Velocity actual value" of LXM28A

	xCmdEnPwr		:BOOL; // Command to enable the power stage of the LXM28
	xCmdRst			:BOOL; // Command to acknowledge an error on the LXM28
	xCmdStop		:BOOL; // Command to stop the LXM28
	xCmdJogFwd		:BOOL; // Command to start the drive in jog mode with positive direction
	xCmdJogRev		:BOOL; // Command to start the drive in jog mode with negative direction
	xCmdJogFast		:BOOL; // Defines the used velocity setpoint for jog operation
	diSetJogDist	:DINT := 1280000; // Defines the distance to move for one tip on jog operation. If value = 0 the continuous motion will be performed
	iWaitTimeJog	:INT  := 500; // Define time delay in ms for change to coninous motion after jog via distance
	diSetVeloJogSlow:DINT := 1280000; // Velocity setpoint for jog operation with slow speed
	diSetVeloJogFast:DINT := 3840000; // Velocity setpoint for jog operation with fast speed 
	xCmdMovVelo		:BOOL; // Command to start the drive with continuous velocity
	xCmdMovRel		:BOOL; // Command to start the drive for relative positioning
	xCmdMovAbs		:BOOL; // Command to start the drive for absolute positioning
	diSetVeloMovVelo:DINT := 1280000; // Velocity setpoint for velocity mode in rpm.
	diSetVeloMovRel	:DINT := 1280000; // Velocity setpoint for relative positioning in usr/s2
	diSetVeloMovAbs	:DINT := 1280000; // Velocity setpoint for absolute positioning in usr/s2
	diSetDistMovRel	:DINT; // Distance setpoint for relative positioning in usr
	diSetPosMovAbs	:DINT; // Target position for absoute positioning in usr
	xCmdHoming		:BOOL; // Command to start homing operation
	diSetHomePos	:DINT; // Position to set if homing is finished
	uiSetHomeMod	:UINT := 33; // Defines the mthod for homing operation. 33 = REF+ with index pulse, not inv., inside
	diSetVeloHome	:DINT := 1280000; // Velocity setpoint for search of the reference switch
	diSetVeloOutHome:DINT := 128000; // Velocity setpoint for movement back to edge of reference switch
		
	xStatEnbl		:BOOL; // Indicates the power stage is enabled
	xJogActv		:BOOL; // Indicates a jog operation is active
	xVeloActv		:BOOL; // Indicates the MC_MoveVelocity is active
	xRelActv		:BOOL; // Indicates the MC_MoveRelative is active
	xAbsActv		:BOOL; // Indicates the MC_MoveAbsolute is active
	dwErrID			:DWORD; // Contains the error ID of the LXM28
	xErr			:BOOL; // Indicates an error is detected (dwErrID <> 0)
	xHomeActv		:BOOL; // Indicates the MC_Home is active
	
	xComOk			:BOOL; // Indicates the CANopen node is in state "Operational"
	eComStat		:CIA405.DEVICE_STATE; // Node state provided by the FB Get_State
END_VAR

// HMISAC/Application/LXM28A_Node03/GVL_LXM28A_Node03
VAR_GLOBAL
	xMcbRdy			:BOOL; // Indicates the state of Motor Circuit Breaker. Mapped to the physical input where the accordingly auxiliary contact of the MCB is connected
	diActlPos		:DINT; // Indicates the actual position. Variable is mapped to TxPDO "Position actual value" of LXM28A
	diActlVelo		:DINT; // Indicates the actual velocity in rpm. Variable is mapped to TxPDO "Velocity actual value" of LXM28A

	xCmdEnPwr		:BOOL; // Command to enable the power stage of the LXM28
	xCmdRst			:BOOL; // Command to acknowledge an error on the LXM28
	xCmdStop		:BOOL; // Command to stop the LXM28
	xCmdJogFwd		:BOOL; // Command to start the drive in jog mode with positive direction
	xCmdJogRev		:BOOL; // Command to start the drive in jog mode with negative direction
	xCmdJogFast		:BOOL; // Defines the used velocity setpoint for jog operation
	diSetJogDist	:DINT := 1280000; // Defines the distance to move for one tip on jog operation. If value = 0 the continuous motion will be performed
	iWaitTimeJog	:INT  := 500; // Define time delay in ms for change to coninous motion after jog via distance
	diSetVeloJogSlow:DINT := 1280000; // Velocity setpoint for jog operation with slow speed
	diSetVeloJogFast:DINT := 3840000; // Velocity setpoint for jog operation with fast speed 
	xCmdMovVelo		:BOOL; // Command to start the drive with continuous velocity
	xCmdMovRel		:BOOL; // Command to start the drive for relative positioning
	xCmdMovAbs		:BOOL; // Command to start the drive for absolute positioning
	diSetVeloMovVelo:DINT := 1280000; // Velocity setpoint for velocity mode in rpm.
	diSetVeloMovRel	:DINT := 1280000; // Velocity setpoint for relative positioning in usr/s2
	diSetVeloMovAbs	:DINT := 1280000; // Velocity setpoint for absolute positioning in usr/s2
	diSetDistMovRel	:DINT; // Distance setpoint for relative positioning in usr
	diSetPosMovAbs	:DINT; // Target position for absoute positioning in usr
	xCmdHoming		:BOOL; // Command to start homing operation
	diSetHomePos	:DINT; // Position to set if homing is finished
	uiSetHomeMod	:UINT := 33; // Defines the method for homing operation. 33 = REF+ with index pulse, not inv., inside
	diSetVeloHome	:DINT := 1280000; // Velocity setpoint for search of the reference switch
	diSetVeloOutHome:DINT := 128000; // Velocity setpoint for movement back to edge of reference switch
		
	xStatEnbl		:BOOL; // Indicates the power stage is enabled
	xJogActv		:BOOL; // Indicates a jog operation is active
	xVeloActv		:BOOL; // Indicates the MC_MoveVelocity is active
	xRelActv		:BOOL; // Indicates the MC_MoveRelative is active
	xAbsActv		:BOOL; // Indicates the MC_MoveAbsolute is active
	dwErrID			:DWORD; // Contains the error ID of the LXM28
	xErr			:BOOL; // Indicates an error is detected (dwErrID <> 0)
	xHomeActv		:BOOL; // Indicates the MC_Home is active
	
	xComOk			:BOOL; // Indicates the CANopen node is in state "Operational"
	eComStat		:CIA405.DEVICE_STATE; // Node state provided by the FB Get_State
END_VAR

// HMISAC/Application/LXM32i_Node11/GVL_LXM32i_Node11
VAR_GLOBAL
	xMcbRdy		 	 : BOOL; // Indicates the state of Motor Circuit Breaker. Mapped to the physical input where the accordingly auxiliary contact of the MCB is connected
	diActlPos	  	 : DINT; // Indicates the actual position of the drive. Variable is mapped to TxPDO "Position actual value" of LXM32i
	diActlVelo	 	 : DINT; // Indicates the actual velocity of the drive in rpm. Variable is mapped to TxPDO "Velocity actual value" of LXM32i
	
	xCmdEnPwr	 	 : BOOL; // Command to enable the power stage of to the drive (maintained signal)
	xCmdRst		 	 : BOOL; // Command to reset the drive in case of detected error on the Lexium
	xCmdStop	 	 : BOOL; // Command To stop the LXM32i
	xCmdJogFwd	 	 : BOOL; // Command to jog the drive in positive direction
	xCmdJogRev	 	 : BOOL; // Command to jog the drive in negative direction
	xCmdJogFast  	 : BOOL; // Defines the used velocity setpoint for jog operation
	diSetJogDist 	 : DINT := 20; // Defines the distance to move for one tip on jog operation. If value = 0 the continuous motion will be performed
	iWaitTimeJog	 : INT := 500; // Define time delay in ms for change to coninous motion
	diSetVeloJogSlow : DINT := 60; // Velocity setpoint for jog operation with slow speed 
	diSetVeloJogFast : DINT := 180; // Velocity setpoint for jog operation with fast speed 
	xCmdMovVelo	 	 : BOOL; // Command to start the drive with continuous velocity
	xCmdMovRel	 	 : BOOL; // Command to start the drive for relative positioning
	xCmdMovAbs	 	 : BOOL; // Command to start the drive for absolute positioning
	diSetVeloMovVelo : DINT; // Velocity setpoint for velocity mode in rpm.
	diSetVeloMovRel	 : DINT := 60; // Velocity setpoint for relative positioning in rpm
	diSetVeloMovAbs	 : DINT := 60; // Velocity setpoint for absolute positioning in rpm
	diSetDistMovRel  : DINT; // Distance setpoint for relative positioning in increments
	diSetPosMovAbs	 : DINT; // Target position for absoute positioning in increments
	xCmdHoming	 	 : BOOL; // Command to start homing operation
	diSetHomePos 	 : DINT; // Position to set if homing is finished
	uiSetHomeMod 	 : UINT:=33; // Defines the method for homing operation. 33 = REF+ with index pulse, not inv., inside
	diSetVeloHome	 : DINT := 60; // Velocity setpoint for search of the reference switch
	diSetVeloOutHome : DINT := 6; // Velocity setpoint for movement back to edge of reference switch
	diSetPosOutHome	 : DINT; // Max. distance for movement back to edge of reference switch
	diSetPosDisHome  : DINT := 200; // Distance for positioning starting from edge of reference switch
	diSetDecStop 	 : DINT := 6000; //Set deceleration for stopping 
	
	xStatEnbl	 : BOOL; // If drive is powered xStatEnbl = True
	xJogActv	 : BOOL; // If the drive is operating in jog mode xJogActv = True
	xVeloActv	 : BOOL; // If the drive is operating in velocity mode xVeloActv = True
	xRelActv	 : BOOL; // If the drive is operating in relative position mode xRelActv = True
	xAbsActv	 : BOOL; // If the drive is operating in absolute position mode xAbsActv = True
	wErrID		 : WORD; // Shows the error ID of the LXM32i
	xErr		 : BOOL; // If error is present xErr = True
	xHomeActv	 : BOOL; // If the drive is operating in homing mode xHomeActv = True
	
	xComOk		 : BOOL; // Indicates the CANopen node is in state "Operational"
	eComStat	 : CIA405.DEVICE_STATE;	// Node state provided by the FB GET_STATE
END_VAR

// HMISAC/Application/GVL
VAR_GLOBAL
	// Communication status
	xPulse_1s 		: BOOL;			// Life bit to HMI	
	
	xCANopenSta		: BOOL;			// If CANopen bus is OK then xCANopenSta = TRUE
	xDev06ComOk		: BOOL;			// Indicates the CANopen node is in state "Operational"
	eDev06ComStat	: CIA405.DEVICE_STATE; // Node state provided by the FB Get_State
	
	// Architecture status
	xGrenOperLEDon	: BOOL;			// Green tower LED on indicates that all drives are in operational state
	xWhitPwrLEDon	: BOOL;			// White tower LED on indicates that at least one motor is powered
	xRedErrLEDon	: BOOL;			// Red tower LED on indicates an Error is present
	xBluSafeErrLEDon: BOOL;			// Blue tower LED on indicates that a Safety Problem is present
	xLXMErrSta		: BOOL;			// Min. one LXM is in error state
	

    // Contactor 
    xDC_ContactorCtrl : BOOL;
	xstart           : BOOL;
	
	
	// Local I/O's
	xEStop			: BOOL;			// If EStop is OK xEstop = True
	xDoorMain		: BOOL;			// If door guarding is OK xDoorMain = True
	xButnRev		: BOOL;			// Green Button for reverse command
	xButnStop		: BOOL;			// Red Button for stop command
	xButnFwd		: BOOL;			// Green Button for forward command

	xButnRevLEDon		: BOOL;		// Green Button LED on front door on
	xButnFwdLEDon		: BOOL;		// Yellow Button LED on front door on
	xEStopButnMainLEDon	: BOOL;		// Blue Button LED EStop on
	xDoorButnMainLEDon	: BOOL;		// Blue Button LED Door on
	
	iTemp1			: INT;			// Temperature sensor connected to analog input of OTB TM2AMI4LT
	iTemp2			: INT;			// Temperature sensor connected to analog input of OTB TM2AMI4LT
	iTemp3			: INT;			// Temperature sensor connected to analog input of OTB TM2AMI4LT
	iTemp4			: INT;			// Temperature sensor connected to analog input of OTB TM2AMI4LT
	iTemp5			: INT;			// Temperature sensor connected to analog input of OTB TM2ALM3LT
	iTemp6			: INT;			// Temperature sensor connected to analog input of OTB TM2ALM3LT
	iAnalogOut		: INT; 			// Analog output connected to analog output of OTB TM2ALM3LT
	
END_VAR

// HMISAC/Application/GVL_HmiVar
VAR_GLOBAL
	//LXM32i commands
	xCmdEnPwrLXM32i11		:BOOL; // HMI command to power the drive
	xCmdMovVeloLXM32i11		:BOOL; // HMI command to start the drive with continuous velocity operation
	diSetMovVeloLXM32i11	:DINT:= 60; // HMI command to set velocity for continuous velocity operation,  unit = 0.1 Hz
	xCmdMovRelLXM32i11		:BOOL; // HMI command to start the drive with relative positioning
	xCmdMovAbsLXM32i11		:BOOL; // HMI command to start the drive with absolute positioning
	xCmdJogRevLXM32i11		:BOOL; // HMI command to run axis in negative direction with "jog velocity"
	xCmdJogFwdLXM32i11		:BOOL; // HMI command to run axis in positive direction with "jog velocity"
	xCmdJogFastLXM32i11		:BOOL; // HMI command to enable fast velocity for "jog velocity"
	xCmdStopLXM32i11		:BOOL; // HMI command to stop the axis
	xCmdRstLXM32i11			:BOOL; // HMI command to acknowledge an error on the drive
	xCmdHomingLXM32i11		:BOOL; // HMI command to start homing operation
	
	//LXM28A commands
	xCmdEnPwrLXM28A03		:BOOL; // HMI command to power the drive
	xCmdMovVeloLXM28A03		:BOOL; // HMI command to start the drive with continuous velocity operation
	diSetMovVeloLXM28A03	:DINT:= 1280000; // HMI command to set velocity for continuous velocity operation,  unit = 0.1 Hz
	xCmdMovRelLXM28A03		:BOOL; // HMI command to start the drive with relative positioning
	xCmdMovAbsLXM28A03		:BOOL; // HMI command to start the drive with absolute positioning
	xCmdJogRevLXM28A03		:BOOL; // HMI command to run axis in negative direction with "jog velocity"
	xCmdJogFwdLXM28A03		:BOOL; // HMI command to run axis in positive direction with "jog velocity"
	xCmdJogFastLXM28A03		:BOOL; // HMI command to enable fast velocity for "jog velocity"
	xCmdStopLXM28A03		:BOOL; // HMI command to stop the axis
	xCmdRstLXM28A03			:BOOL; // HMI command to acknowledge an error on the drive
	xCmdHomingLXM28A03		:BOOL; // HMI command to start homing operation
	xCmdWriteParaLXM28A03	:BOOL; // Command to write the parameter to the LXM28 drive
	xWriteParaAccDoneLXM2803		:BOOL; // Status parameter was successfully written
	xWriteParaDecDoneLXM2803		:BOOL; // Status parameter was successfully written
	xWriteParaDecStopDoneLXM2803	:BOOL; // Status parameter was successfully written
	
	xCmdEnPwrLXM28A04		:BOOL; // HMI command to power the drive
	xCmdMovVeloLXM28A04		:BOOL; // HMI command to start the drive with continuous velocity operation
	diSetMovVeloLXM28A04	:DINT:= 1280000; // HMI command to set velocity for continuous velocity operation,  unit = 0.1 Hz
	xCmdMovRelLXM28A04		:BOOL; // HMI command to start the drive with relative positioning
	xCmdMovAbsLXM28A04		:BOOL; // HMI command to start the drive with absolute positioning
	xCmdJogRevLXM28A04		:BOOL; // HMI command to run axis in negative direction with "jog velocity"
	xCmdJogFwdLXM28A04		:BOOL; // HMI command to run axis in positive direction with "jog velocity"
	xCmdJogFastLXM28A04		:BOOL; // HMI command to enable fast velocity for "jog velocity"
	xCmdStopLXM28A04		:BOOL; // HMI command to stop the axis
	xCmdRstLXM28A04			:BOOL; // HMI command to acknowledge an error on the drive
	xCmdHomingLXM28A04		:BOOL; // HMI command to start homing operation
	xCmdWriteParaLXM28A04	:BOOL; // Command to write the parameter to the LXM28 drive
	xWriteParaAccDoneLXM2804		:BOOL; // Status parameter was successfully written
	xWriteParaDecDoneLXM2804		:BOOL; // Status parameter was successfully written
	xWriteParaDecStopDoneLXM2804	:BOOL; // Status parameter was successfully written

END_VAR

// HMISAC/Application/GVL_AlarmMsg
VAR_GLOBAL
	// Emergency alarms
	xEStopAlarm				: BOOL;	// Indicates if EStop is tripped
	xDoorGuardAlarm			: BOOL;	// Indicates if door guarding is tripped

	//Joystick Danfoss  JSD6000 alarms
	xComAlarmJSD6000A02 		: BOOL; // Indicates a communication fault
		
	//LXM28 alarms
	xMcbAlarmLXM28A03		: BOOL;	// Indicates if Mcb is not ready
	xComAlarmLXM28A03 		: BOOL; // Indicates a communication fault
	xAxisAlarmLXM28A03		: BOOL;	// Indicates a axis error
	xAlrmWriteParaLXM28A03	: BOOL; // Error occured during write parameter

	xMcbAlarmLXM28A04 		: BOOL;	// Indicates if Mcb is not ready
	xComAlarmLXM28A04 		: BOOL; // Indicates a communication fault
	xAxisAlarmLXM28A04		: BOOL;	// Indicates a axis error
	xAlrmWriteParaLXM28A04	: BOOL; // Error occured during write parameter
	
	//LXM32i alarms
	xMcbAlarmLXM32i11 		: BOOL;	// Indicates if Mcb is not ready
	xComAlarmLXM32i11 		: BOOL; // Indicates a communication fault
	xAxisAlarmLXM32i11		: BOOL;	// Indicates a axis error
	
END_VAR

// HMISAC/Application/Joystick_SD6000/GVL_Joystick6000
VAR_GLOBAL
	xComOk			:BOOL; // Indicates the CANopen node is in state "Operational"
	eComStat		:CIA405.DEVICE_STATE; // Node state provided by the FB Get_State
END_VAR

// HMISAC/Application/MicroCAN4aiBOX/GVL_MicroCAN
VAR_GLOBAL
	xComOk			:BOOL; // Indicates the CANopen node is in state "Operational"
	eComStat		:CIA405.DEVICE_STATE; // Node state provided by the FB Get_State
END_VAR

// HMISAC/Application/Dunker_0A/GVL_Dunker_0A
VAR_GLOBAL
	xComOk			:BOOL; // Indicates the CANopen node is in state "Operational"
	eComStat		:CIA405.DEVICE_STATE; // Node state provided by the FB Get_State

	xCmdEnPwr	 	 : BOOL:=1; // Command to enable the power stage of to the drive (maintained signal)
	xCmdRst		 	 : BOOL; // Command to reset the drive in case of detected error on the Lexium
	xCmdStop	 	 : BOOL; // Command To stop the LXM32i
	nAixState        : SMC_AXIS_STATE;
	xStatEnbl	     : BOOL; // If drive is powered xStatEnbl = True
//    x_on	         : BOOL; 
//    x_start	         : BOOL; 
//    str_driver	         : STRING(16); 
//    dw_driver	         : DWORD; 
END_VAR

// HMISAC/Application/Dunker_0B/GVL_Dunker_0B
VAR_GLOBAL
	xComOk			:BOOL; // Indicates the CANopen node is in state "Operational"
	eComStat		:CIA405.DEVICE_STATE; // Node state provided by the FB Get_State
END_VAR

// HMISAC/Application/Dunker_0C/GVL_Dunker_0C
VAR_GLOBAL
	xComOk			:BOOL; // Indicates the CANopen node is in state "Operational"
	eComStat		:CIA405.DEVICE_STATE; // Node state provided by the FB Get_State
END_VAR

// HMISAC/Application/Dunker_0D/GVL_Dunker_0D
VAR_GLOBAL
	xComOk			:BOOL; // Indicates the CANopen node is in state "Operational"
	eComStat		:CIA405.DEVICE_STATE; // Node state provided by the FB Get_State
END_VAR

// HMISAC/Application/Speedgoat/GVL_Speedgoat
VAR_GLOBAL
	xComOk			:BOOL; // Indicates the CANopen node is in state "Operational"
	eComStat		:CIA405.DEVICE_STATE; // Node state provided by the FB Get_State
END_VAR

// HMISAC/Application/Preprocessing
PROGRAM Preprocessing
VAR
	fbPowerEnableATV32_01	:SE_TBX.Toggle_FlipFlop;	// FB instance command Power Enable
	fbPowerEnableATV32_02	:SE_TBX.Toggle_FlipFlop;	// FB instance command Power Enable
	fbPowerEnableLXM28_03	:SE_TBX.Toggle_FlipFlop;	// FB instance command Power Enable
	fbPowerEnableLXM28_04	:SE_TBX.Toggle_FlipFlop;	// FB instance command Power Enable
	fbPowerEnableLXM32i_11	:SE_TBX.Toggle_FlipFlop;	// FB instance command Power Enable
	fbJogFastLXM28_03		:SE_TBX.Toggle_FlipFlop;	// FB instance command JogFast
	fbJogFastLXM28_04		:SE_TBX.Toggle_FlipFlop;	// FB instance command JogFast
	fbJogFastLXM32i_11		:SE_TBX.Toggle_FlipFlop;	// FB instance command JogFast
END_VAR
VAR // added by the converter: edge detectors and wires of the graphical bodies
    _rt1, _rt2, _rt3, _rt4, _rt5, _rt6, _rt7, _rt8, _rt9, _rt10, _rt11, _rt12, _rt13, _rt14, _rt15, _rt16, _rt17, _rt18, _rt19, _rt20, _rt21, _rt22, _rt23, _rt24, _rt25, _rt26, _rt27, _rt28, _rt29, _rt30, _rt31, _rt32, _rt33, _rt34, _rt35, _rt36, _rt37, _rt38, _rt39 : R_TRIG;
    _w1, _w2, _w3 : INT;
    _ft1, _ft2, _ft3 : F_TRIG;
END_VAR

ACTION A04_DrvCmd_LXM28A_Node04:
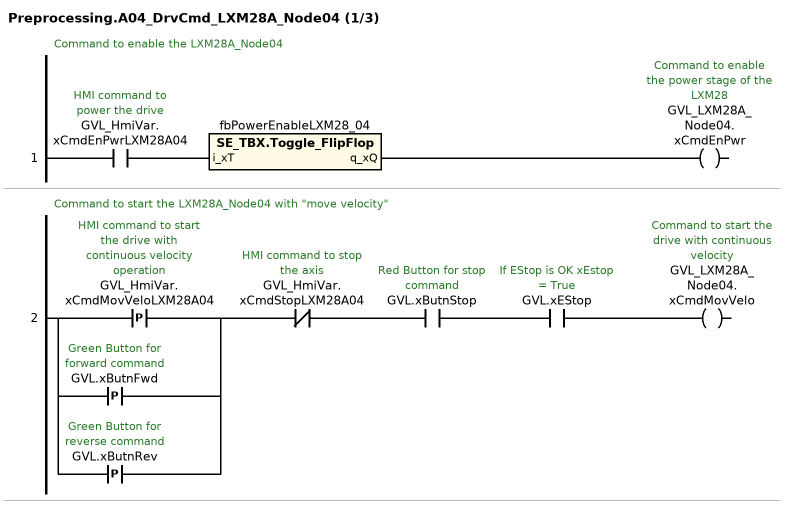
// NETWORK 1
// Command to enable the LXM28A_Node04
//   fbPowerEnableLXM28_04: FB instance command Power Enable
//   GVL_HmiVar.xCmdEnPwrLXM28A04: HMI command to power the drive
//   GVL_LXM28A_Node04.xCmdEnPwr: Command to enable the power stage of the LXM28
fbPowerEnableLXM28_04(i_xT := GVL_HmiVar.xCmdEnPwrLXM28A04); // SE_TBX.Toggle_FlipFlop
GVL_LXM28A_Node04.xCmdEnPwr := fbPowerEnableLXM28_04.q_xQ;

// NETWORK 2
// Command to start the LXM28A_Node04 with "move velocity"
//   GVL_HmiVar.xCmdMovVeloLXM28A04: HMI command to start the drive with continuous velocity operation
//   GVL.xButnFwd: Green Button for forward command
//   GVL.xButnRev: Green Button for reverse command
//   GVL_HmiVar.xCmdStopLXM28A04: HMI command to stop the axis
//   GVL.xButnStop: Red Button for stop command
//   GVL.xEStop: If EStop is OK xEstop = True
//   GVL_LXM28A_Node04.xCmdMovVelo: Command to start the drive with continuous velocity
_rt1(CLK := GVL_HmiVar.xCmdMovVeloLXM28A04);
_rt2(CLK := GVL.xButnFwd);
_rt3(CLK := GVL.xButnRev);
GVL_LXM28A_Node04.xCmdMovVelo := (_rt1.Q OR _rt2.Q OR _rt3.Q) AND NOT GVL_HmiVar.xCmdStopLXM28A04 AND GVL.xButnStop AND GVL.xEStop;

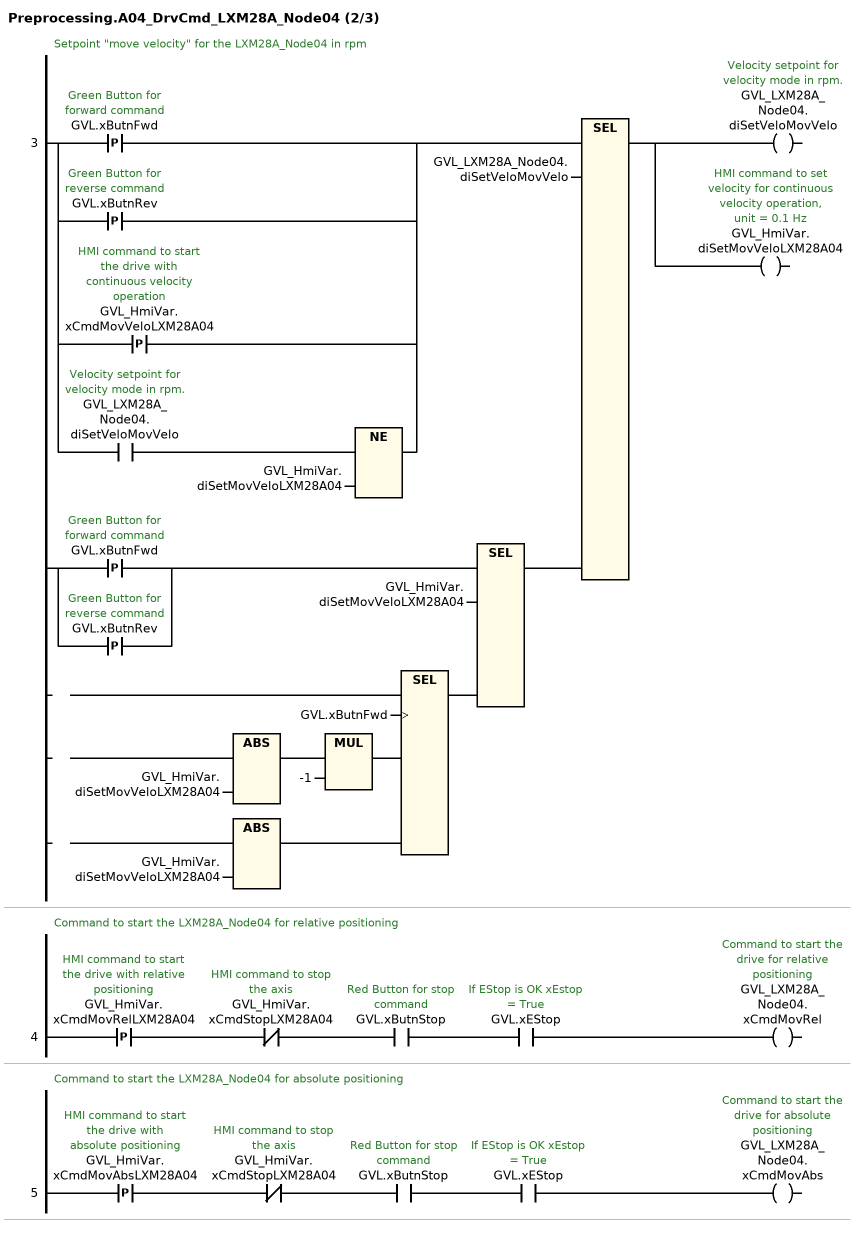
// NETWORK 3
// Setpoint "move velocity" for the LXM28A_Node04 in rpm
//   GVL.xButnFwd: Green Button for forward command
//   GVL.xButnRev: Green Button for reverse command
//   GVL_HmiVar.xCmdMovVeloLXM28A04: HMI command to start the drive with continuous velocity operation
//   GVL_LXM28A_Node04.diSetVeloMovVelo: Velocity setpoint for velocity mode in rpm.
//   GVL_HmiVar.diSetMovVeloLXM28A04: HMI command to set velocity for continuous velocity operation, unit = 0.1 Hz
_rt4(CLK := GVL.xButnFwd);
_rt5(CLK := GVL.xButnRev);
_rt6(CLK := GVL_HmiVar.xCmdMovVeloLXM28A04);
_rt7(CLK := GVL.xButnFwd);
_rt8(CLK := GVL.xButnRev);
_rt9(CLK := GVL.xButnFwd);
_w1 := SEL(_rt4.Q OR _rt5.Q OR _rt6.Q OR GVL_LXM28A_Node04.diSetVeloMovVelo <> GVL_HmiVar.diSetMovVeloLXM28A04, GVL_LXM28A_Node04.diSetVeloMovVelo, SEL(_rt7.Q OR _rt8.Q, GVL_HmiVar.diSetMovVeloLXM28A04, SEL(_rt9.Q, ABS(GVL_HmiVar.diSetMovVeloLXM28A04) * -1, ABS(GVL_HmiVar.diSetMovVeloLXM28A04))));
GVL_LXM28A_Node04.diSetVeloMovVelo := _w1;
GVL_HmiVar.diSetMovVeloLXM28A04 := _w1;

// NETWORK 4
// Command to start the LXM28A_Node04 for relative positioning
//   GVL_HmiVar.xCmdMovRelLXM28A04: HMI command to start the drive with relative positioning
//   GVL_HmiVar.xCmdStopLXM28A04: HMI command to stop the axis
//   GVL.xButnStop: Red Button for stop command
//   GVL.xEStop: If EStop is OK xEstop = True
//   GVL_LXM28A_Node04.xCmdMovRel: Command to start the drive for relative positioning
_rt10(CLK := GVL_HmiVar.xCmdMovRelLXM28A04);
GVL_LXM28A_Node04.xCmdMovRel := _rt10.Q AND NOT GVL_HmiVar.xCmdStopLXM28A04 AND GVL.xButnStop AND GVL.xEStop;

// NETWORK 5
// Command to start the LXM28A_Node04 for absolute positioning
//   GVL_HmiVar.xCmdMovAbsLXM28A04: HMI command to start the drive with absolute positioning
//   GVL_HmiVar.xCmdStopLXM28A04: HMI command to stop the axis
//   GVL.xButnStop: Red Button for stop command
//   GVL.xEStop: If EStop is OK xEstop = True
//   GVL_LXM28A_Node04.xCmdMovAbs: Command to start the drive for absolute positioning
_rt11(CLK := GVL_HmiVar.xCmdMovAbsLXM28A04);
GVL_LXM28A_Node04.xCmdMovAbs := _rt11.Q AND NOT GVL_HmiVar.xCmdStopLXM28A04 AND GVL.xButnStop AND GVL.xEStop;

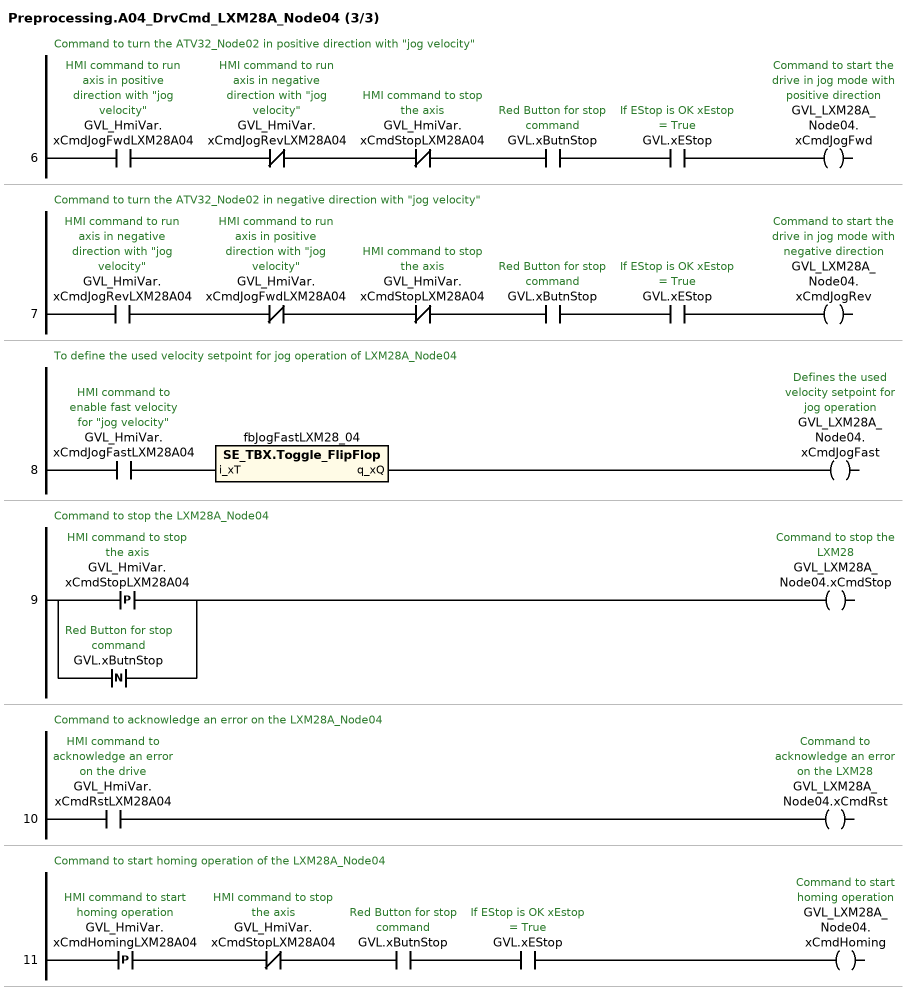
// NETWORK 6
// Command to turn the ATV32_Node02 in positive direction with "jog velocity"
//   GVL_HmiVar.xCmdJogFwdLXM28A04: HMI command to run axis in positive direction with "jog velocity"
//   GVL_HmiVar.xCmdJogRevLXM28A04: HMI command to run axis in negative direction with "jog velocity"
//   GVL_HmiVar.xCmdStopLXM28A04: HMI command to stop the axis
//   GVL.xButnStop: Red Button for stop command
//   GVL.xEStop: If EStop is OK xEstop = True
//   GVL_LXM28A_Node04.xCmdJogFwd: Command to start the drive in jog mode with positive direction
GVL_LXM28A_Node04.xCmdJogFwd := GVL_HmiVar.xCmdJogFwdLXM28A04 AND NOT GVL_HmiVar.xCmdJogRevLXM28A04 AND NOT GVL_HmiVar.xCmdStopLXM28A04 AND GVL.xButnStop AND GVL.xEStop;

// NETWORK 7
// Command to turn the ATV32_Node02 in negative direction with "jog velocity"
//   GVL_HmiVar.xCmdJogRevLXM28A04: HMI command to run axis in negative direction with "jog velocity"
//   GVL_HmiVar.xCmdJogFwdLXM28A04: HMI command to run axis in positive direction with "jog velocity"
//   GVL_HmiVar.xCmdStopLXM28A04: HMI command to stop the axis
//   GVL.xButnStop: Red Button for stop command
//   GVL.xEStop: If EStop is OK xEstop = True
//   GVL_LXM28A_Node04.xCmdJogRev: Command to start the drive in jog mode with negative direction
GVL_LXM28A_Node04.xCmdJogRev := GVL_HmiVar.xCmdJogRevLXM28A04 AND NOT GVL_HmiVar.xCmdJogFwdLXM28A04 AND NOT GVL_HmiVar.xCmdStopLXM28A04 AND GVL.xButnStop AND GVL.xEStop;

// NETWORK 8
// To define the used velocity setpoint for jog operation of LXM28A_Node04
//   fbJogFastLXM28_04: FB instance command JogFast
//   GVL_HmiVar.xCmdJogFastLXM28A04: HMI command to enable fast velocity for "jog velocity"
//   GVL_LXM28A_Node04.xCmdJogFast: Defines the used velocity setpoint for jog operation
fbJogFastLXM28_04(i_xT := GVL_HmiVar.xCmdJogFastLXM28A04); // SE_TBX.Toggle_FlipFlop
GVL_LXM28A_Node04.xCmdJogFast := fbJogFastLXM28_04.q_xQ;

// NETWORK 9
// Command to stop the LXM28A_Node04
//   GVL_HmiVar.xCmdStopLXM28A04: HMI command to stop the axis
//   GVL.xButnStop: Red Button for stop command
//   GVL_LXM28A_Node04.xCmdStop: Command to stop the LXM28
_rt12(CLK := GVL_HmiVar.xCmdStopLXM28A04);
_ft1(CLK := GVL.xButnStop);
GVL_LXM28A_Node04.xCmdStop := _rt12.Q OR _ft1.Q;

// NETWORK 10
// Command to acknowledge an error on the LXM28A_Node04
//   GVL_HmiVar.xCmdRstLXM28A04: HMI command to acknowledge an error on the drive
//   GVL_LXM28A_Node04.xCmdRst: Command to acknowledge an error on the LXM28
GVL_LXM28A_Node04.xCmdRst := GVL_HmiVar.xCmdRstLXM28A04;

// NETWORK 11
// Command to start homing operation of the LXM28A_Node04
//   GVL_HmiVar.xCmdHomingLXM28A04: HMI command to start homing operation
//   GVL_HmiVar.xCmdStopLXM28A04: HMI command to stop the axis
//   GVL.xButnStop: Red Button for stop command
//   GVL.xEStop: If EStop is OK xEstop = True
//   GVL_LXM28A_Node04.xCmdHoming: Command to start homing operation
_rt13(CLK := GVL_HmiVar.xCmdHomingLXM28A04);
GVL_LXM28A_Node04.xCmdHoming := _rt13.Q AND NOT GVL_HmiVar.xCmdStopLXM28A04 AND GVL.xButnStop AND GVL.xEStop;
END_ACTION

ACTION A05_DrvCmd_LXM32i_Node11:
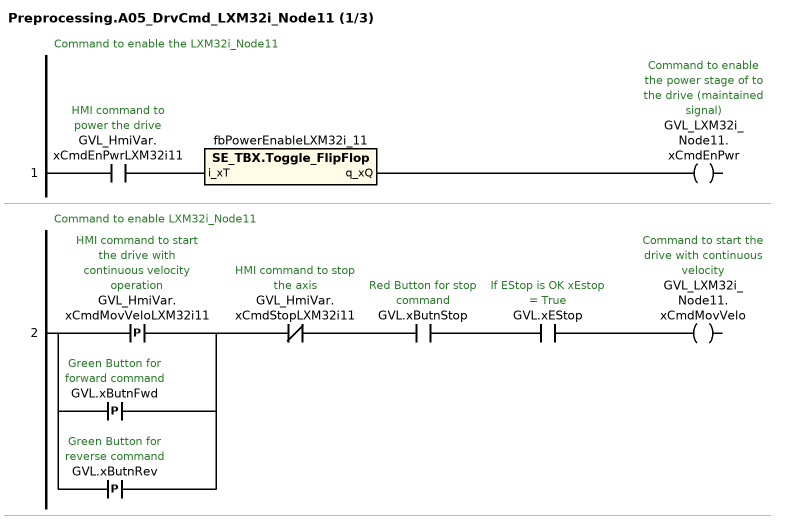
// NETWORK 1
// Command to enable the LXM32i_Node11
//   fbPowerEnableLXM32i_11: FB instance command Power Enable
//   GVL_HmiVar.xCmdEnPwrLXM32i11: HMI command to power the drive
//   GVL_LXM32i_Node11.xCmdEnPwr: Command to enable the power stage of to the drive (maintained signal)
fbPowerEnableLXM32i_11(i_xT := GVL_HmiVar.xCmdEnPwrLXM32i11); // SE_TBX.Toggle_FlipFlop
GVL_LXM32i_Node11.xCmdEnPwr := fbPowerEnableLXM32i_11.q_xQ;

// NETWORK 2
// Command to enable LXM32i_Node11
//   GVL_HmiVar.xCmdMovVeloLXM32i11: HMI command to start the drive with continuous velocity operation
//   GVL.xButnFwd: Green Button for forward command
//   GVL.xButnRev: Green Button for reverse command
//   GVL_HmiVar.xCmdStopLXM32i11: HMI command to stop the axis
//   GVL.xButnStop: Red Button for stop command
//   GVL.xEStop: If EStop is OK xEstop = True
//   GVL_LXM32i_Node11.xCmdMovVelo: Command to start the drive with continuous velocity
_rt14(CLK := GVL_HmiVar.xCmdMovVeloLXM32i11);
_rt15(CLK := GVL.xButnFwd);
_rt16(CLK := GVL.xButnRev);
GVL_LXM32i_Node11.xCmdMovVelo := (_rt14.Q OR _rt15.Q OR _rt16.Q) AND NOT GVL_HmiVar.xCmdStopLXM32i11 AND GVL.xButnStop AND GVL.xEStop;

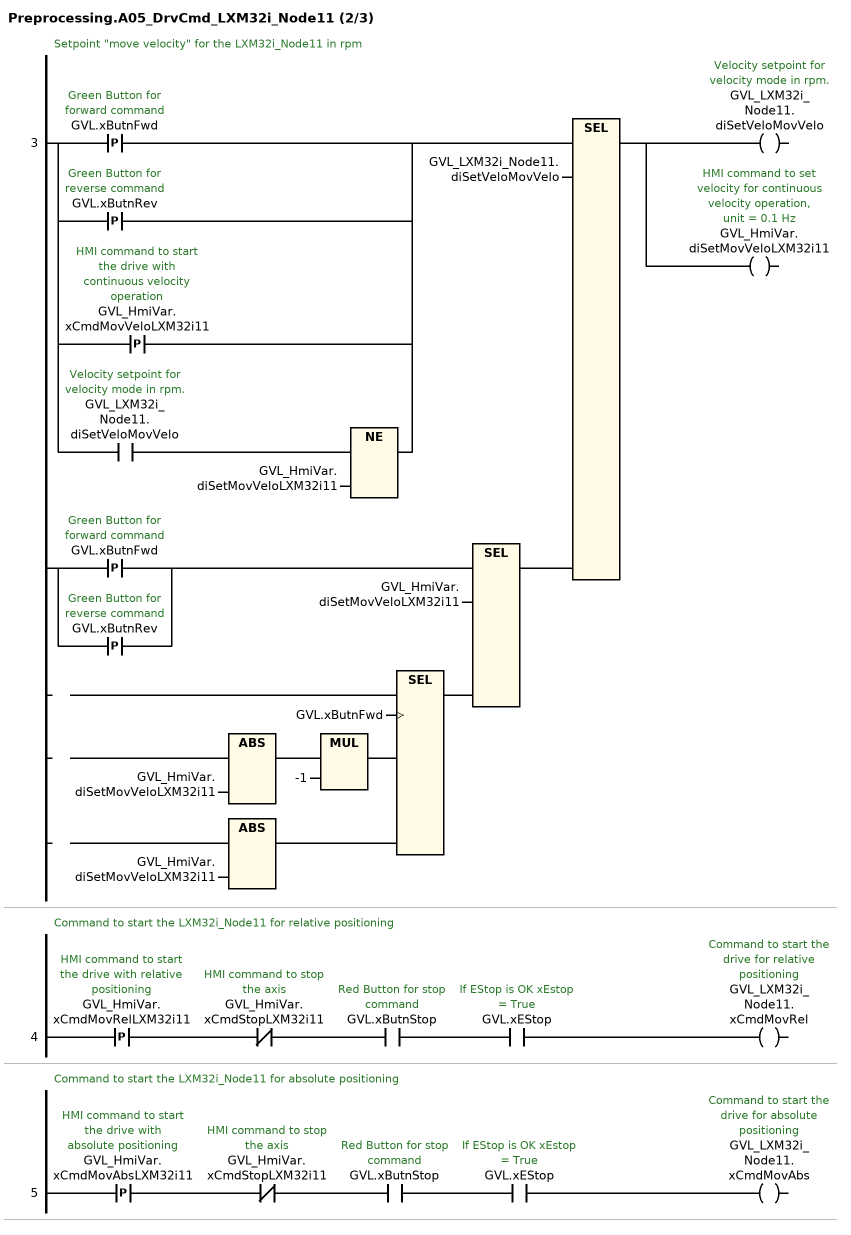
// NETWORK 3
// Setpoint "move velocity" for the LXM32i_Node11 in rpm
//   GVL.xButnFwd: Green Button for forward command
//   GVL.xButnRev: Green Button for reverse command
//   GVL_HmiVar.xCmdMovVeloLXM32i11: HMI command to start the drive with continuous velocity operation
//   GVL_LXM32i_Node11.diSetVeloMovVelo: Velocity setpoint for velocity mode in rpm.
//   GVL_HmiVar.diSetMovVeloLXM32i11: HMI command to set velocity for continuous velocity operation, unit = 0.1 Hz
_rt17(CLK := GVL.xButnFwd);
_rt18(CLK := GVL.xButnRev);
_rt19(CLK := GVL_HmiVar.xCmdMovVeloLXM32i11);
_rt20(CLK := GVL.xButnFwd);
_rt21(CLK := GVL.xButnRev);
_rt22(CLK := GVL.xButnFwd);
_w2 := SEL(_rt17.Q OR _rt18.Q OR _rt19.Q OR GVL_LXM32i_Node11.diSetVeloMovVelo <> GVL_HmiVar.diSetMovVeloLXM32i11, GVL_LXM32i_Node11.diSetVeloMovVelo, SEL(_rt20.Q OR _rt21.Q, GVL_HmiVar.diSetMovVeloLXM32i11, SEL(_rt22.Q, ABS(GVL_HmiVar.diSetMovVeloLXM32i11) * -1, ABS(GVL_HmiVar.diSetMovVeloLXM32i11))));
GVL_LXM32i_Node11.diSetVeloMovVelo := _w2;
GVL_HmiVar.diSetMovVeloLXM32i11 := _w2;

// NETWORK 4
// Command to start the LXM32i_Node11 for relative positioning
//   GVL_HmiVar.xCmdMovRelLXM32i11: HMI command to start the drive with relative positioning
//   GVL_HmiVar.xCmdStopLXM32i11: HMI command to stop the axis
//   GVL.xButnStop: Red Button for stop command
//   GVL.xEStop: If EStop is OK xEstop = True
//   GVL_LXM32i_Node11.xCmdMovRel: Command to start the drive for relative positioning
_rt23(CLK := GVL_HmiVar.xCmdMovRelLXM32i11);
GVL_LXM32i_Node11.xCmdMovRel := _rt23.Q AND NOT GVL_HmiVar.xCmdStopLXM32i11 AND GVL.xButnStop AND GVL.xEStop;

// NETWORK 5
// Command to start the LXM32i_Node11 for absolute positioning
//   GVL_HmiVar.xCmdMovAbsLXM32i11: HMI command to start the drive with absolute positioning
//   GVL_HmiVar.xCmdStopLXM32i11: HMI command to stop the axis
//   GVL.xButnStop: Red Button for stop command
//   GVL.xEStop: If EStop is OK xEstop = True
//   GVL_LXM32i_Node11.xCmdMovAbs: Command to start the drive for absolute positioning
_rt24(CLK := GVL_HmiVar.xCmdMovAbsLXM32i11);
GVL_LXM32i_Node11.xCmdMovAbs := _rt24.Q AND NOT GVL_HmiVar.xCmdStopLXM32i11 AND GVL.xButnStop AND GVL.xEStop;

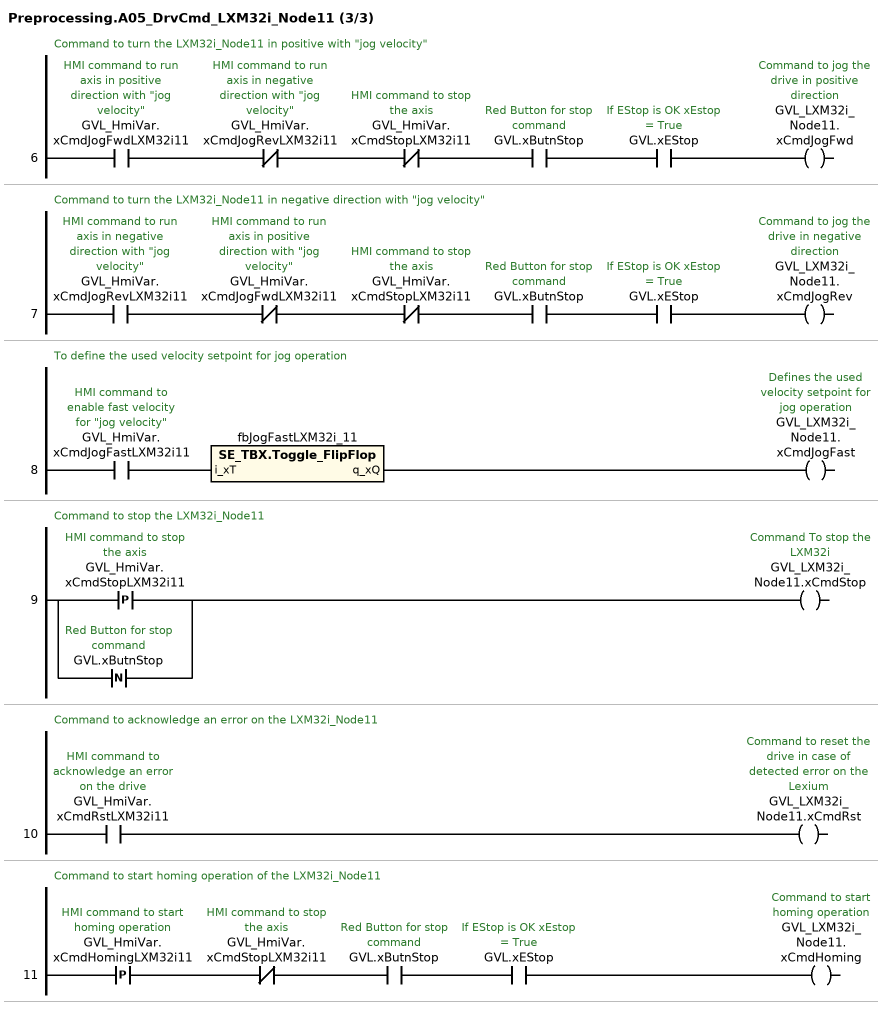
// NETWORK 6
// Command to turn the LXM32i_Node11 in positive with "jog velocity"
//   GVL_HmiVar.xCmdJogFwdLXM32i11: HMI command to run axis in positive direction with "jog velocity"
//   GVL_HmiVar.xCmdJogRevLXM32i11: HMI command to run axis in negative direction with "jog velocity"
//   GVL_HmiVar.xCmdStopLXM32i11: HMI command to stop the axis
//   GVL.xButnStop: Red Button for stop command
//   GVL.xEStop: If EStop is OK xEstop = True
//   GVL_LXM32i_Node11.xCmdJogFwd: Command to jog the drive in positive direction
GVL_LXM32i_Node11.xCmdJogFwd := GVL_HmiVar.xCmdJogFwdLXM32i11 AND NOT GVL_HmiVar.xCmdJogRevLXM32i11 AND NOT GVL_HmiVar.xCmdStopLXM32i11 AND GVL.xButnStop AND GVL.xEStop;

// NETWORK 7
// Command to turn the LXM32i_Node11 in negative direction with "jog velocity"
//   GVL_HmiVar.xCmdJogRevLXM32i11: HMI command to run axis in negative direction with "jog velocity"
//   GVL_HmiVar.xCmdJogFwdLXM32i11: HMI command to run axis in positive direction with "jog velocity"
//   GVL_HmiVar.xCmdStopLXM32i11: HMI command to stop the axis
//   GVL.xButnStop: Red Button for stop command
//   GVL.xEStop: If EStop is OK xEstop = True
//   GVL_LXM32i_Node11.xCmdJogRev: Command to jog the drive in negative direction
GVL_LXM32i_Node11.xCmdJogRev := GVL_HmiVar.xCmdJogRevLXM32i11 AND NOT GVL_HmiVar.xCmdJogFwdLXM32i11 AND NOT GVL_HmiVar.xCmdStopLXM32i11 AND GVL.xButnStop AND GVL.xEStop;

// NETWORK 8
// To define the used velocity setpoint for jog operation
//   fbJogFastLXM32i_11: FB instance command JogFast
//   GVL_HmiVar.xCmdJogFastLXM32i11: HMI command to enable fast velocity for "jog velocity"
//   GVL_LXM32i_Node11.xCmdJogFast: Defines the used velocity setpoint for jog operation
fbJogFastLXM32i_11(i_xT := GVL_HmiVar.xCmdJogFastLXM32i11); // SE_TBX.Toggle_FlipFlop
GVL_LXM32i_Node11.xCmdJogFast := fbJogFastLXM32i_11.q_xQ;

// NETWORK 9
// Command to stop the LXM32i_Node11
//   GVL_HmiVar.xCmdStopLXM32i11: HMI command to stop the axis
//   GVL.xButnStop: Red Button for stop command
//   GVL_LXM32i_Node11.xCmdStop: Command To stop the LXM32i
_rt25(CLK := GVL_HmiVar.xCmdStopLXM32i11);
_ft2(CLK := GVL.xButnStop);
GVL_LXM32i_Node11.xCmdStop := _rt25.Q OR _ft2.Q;

// NETWORK 10
// Command to acknowledge an error on the LXM32i_Node11
//   GVL_HmiVar.xCmdRstLXM32i11: HMI command to acknowledge an error on the drive
//   GVL_LXM32i_Node11.xCmdRst: Command to reset the drive in case of detected error on the Lexium
GVL_LXM32i_Node11.xCmdRst := GVL_HmiVar.xCmdRstLXM32i11;

// NETWORK 11
// Command to start homing operation of the LXM32i_Node11
//   GVL_HmiVar.xCmdHomingLXM32i11: HMI command to start homing operation
//   GVL_HmiVar.xCmdStopLXM32i11: HMI command to stop the axis
//   GVL.xButnStop: Red Button for stop command
//   GVL.xEStop: If EStop is OK xEstop = True
//   GVL_LXM32i_Node11.xCmdHoming: Command to start homing operation
_rt26(CLK := GVL_HmiVar.xCmdHomingLXM32i11);
GVL_LXM32i_Node11.xCmdHoming := _rt26.Q AND NOT GVL_HmiVar.xCmdStopLXM32i11 AND GVL.xButnStop AND GVL.xEStop;
END_ACTION

ACTION A03_DrvCmd_LXM28A_Node03:
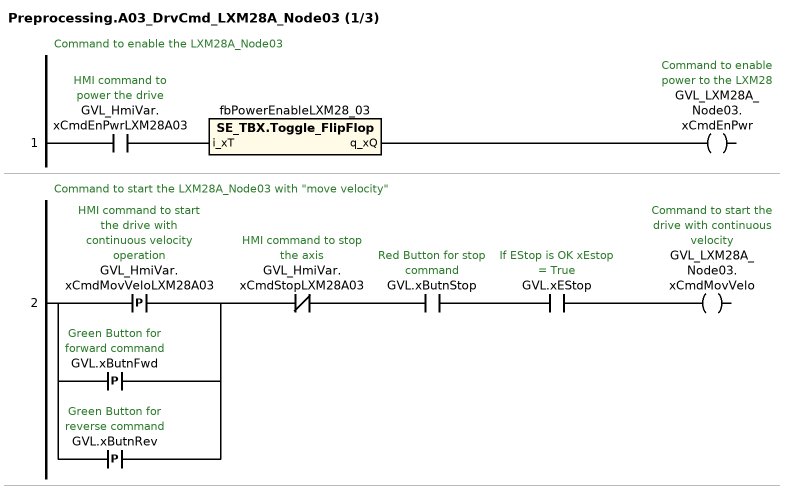
// NETWORK 1
// Command to enable the LXM28A_Node03
//   fbPowerEnableLXM28_03: FB instance command Power Enable
//   GVL_HmiVar.xCmdEnPwrLXM28A03: HMI command to power the drive
//   GVL_LXM28A_Node03.xCmdEnPwr: Command to enable power to the LXM28
fbPowerEnableLXM28_03(i_xT := GVL_HmiVar.xCmdEnPwrLXM28A03); // SE_TBX.Toggle_FlipFlop
GVL_LXM28A_Node03.xCmdEnPwr := fbPowerEnableLXM28_03.q_xQ;

// NETWORK 2
// Command to start the LXM28A_Node03 with "move velocity"
//   GVL_HmiVar.xCmdMovVeloLXM28A03: HMI command to start the drive with continuous velocity operation
//   GVL.xButnFwd: Green Button for forward command
//   GVL.xButnRev: Green Button for reverse command
//   GVL_HmiVar.xCmdStopLXM28A03: HMI command to stop the axis
//   GVL.xButnStop: Red Button for stop command
//   GVL.xEStop: If EStop is OK xEstop = True
//   GVL_LXM28A_Node03.xCmdMovVelo: Command to start the drive with continuous velocity
_rt27(CLK := GVL_HmiVar.xCmdMovVeloLXM28A03);
_rt28(CLK := GVL.xButnFwd);
_rt29(CLK := GVL.xButnRev);
GVL_LXM28A_Node03.xCmdMovVelo := (_rt27.Q OR _rt28.Q OR _rt29.Q) AND NOT GVL_HmiVar.xCmdStopLXM28A03 AND GVL.xButnStop AND GVL.xEStop;

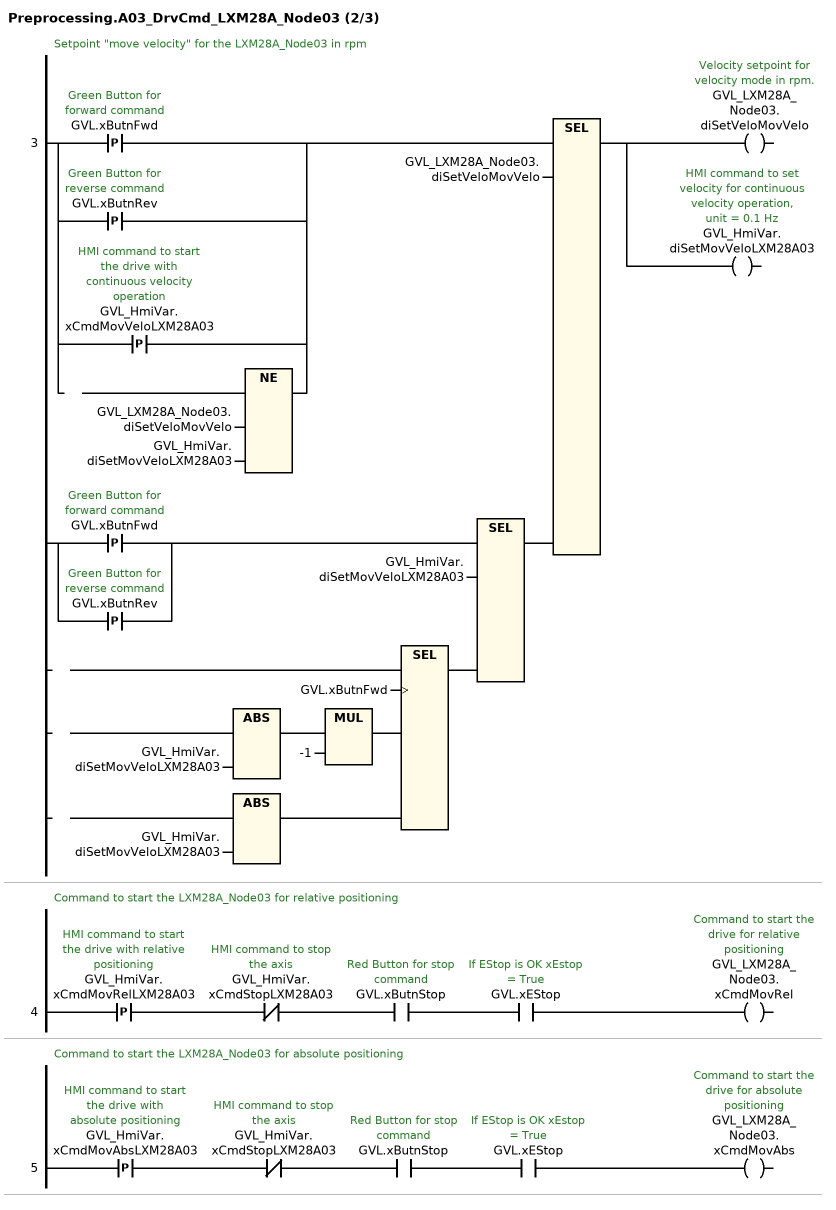
// NETWORK 3
// Setpoint "move velocity" for the LXM28A_Node03 in rpm
//   GVL.xButnFwd: Green Button for forward command
//   GVL.xButnRev: Green Button for reverse command
//   GVL_HmiVar.xCmdMovVeloLXM28A03: HMI command to start the drive with continuous velocity operation
//   GVL_LXM28A_Node03.diSetVeloMovVelo: Velocity setpoint for velocity mode in rpm.
//   GVL_HmiVar.diSetMovVeloLXM28A03: HMI command to set velocity for continuous velocity operation, unit = 0.1 Hz
_rt30(CLK := GVL.xButnFwd);
_rt31(CLK := GVL.xButnRev);
_rt32(CLK := GVL_HmiVar.xCmdMovVeloLXM28A03);
_rt33(CLK := GVL.xButnFwd);
_rt34(CLK := GVL.xButnRev);
_rt35(CLK := GVL.xButnFwd);
_w3 := SEL((_rt30.Q OR _rt31.Q OR _rt32.Q) OR GVL_LXM28A_Node03.diSetVeloMovVelo <> GVL_HmiVar.diSetMovVeloLXM28A03, GVL_LXM28A_Node03.diSetVeloMovVelo, SEL(_rt33.Q OR _rt34.Q, GVL_HmiVar.diSetMovVeloLXM28A03, SEL(_rt35.Q, ABS(GVL_HmiVar.diSetMovVeloLXM28A03) * -1, ABS(GVL_HmiVar.diSetMovVeloLXM28A03))));
GVL_LXM28A_Node03.diSetVeloMovVelo := _w3;
GVL_HmiVar.diSetMovVeloLXM28A03 := _w3;

// NETWORK 4
// Command to start the LXM28A_Node03 for relative positioning
//   GVL_HmiVar.xCmdMovRelLXM28A03: HMI command to start the drive with relative positioning
//   GVL_HmiVar.xCmdStopLXM28A03: HMI command to stop the axis
//   GVL.xButnStop: Red Button for stop command
//   GVL.xEStop: If EStop is OK xEstop = True
//   GVL_LXM28A_Node03.xCmdMovRel: Command to start the drive for relative positioning
_rt36(CLK := GVL_HmiVar.xCmdMovRelLXM28A03);
GVL_LXM28A_Node03.xCmdMovRel := _rt36.Q AND NOT GVL_HmiVar.xCmdStopLXM28A03 AND GVL.xButnStop AND GVL.xEStop;

// NETWORK 5
// Command to start the LXM28A_Node03 for absolute positioning
//   GVL_HmiVar.xCmdMovAbsLXM28A03: HMI command to start the drive with absolute positioning
//   GVL_HmiVar.xCmdStopLXM28A03: HMI command to stop the axis
//   GVL.xButnStop: Red Button for stop command
//   GVL.xEStop: If EStop is OK xEstop = True
//   GVL_LXM28A_Node03.xCmdMovAbs: Command to start the drive for absolute positioning
_rt37(CLK := GVL_HmiVar.xCmdMovAbsLXM28A03);
GVL_LXM28A_Node03.xCmdMovAbs := _rt37.Q AND NOT GVL_HmiVar.xCmdStopLXM28A03 AND GVL.xButnStop AND GVL.xEStop;

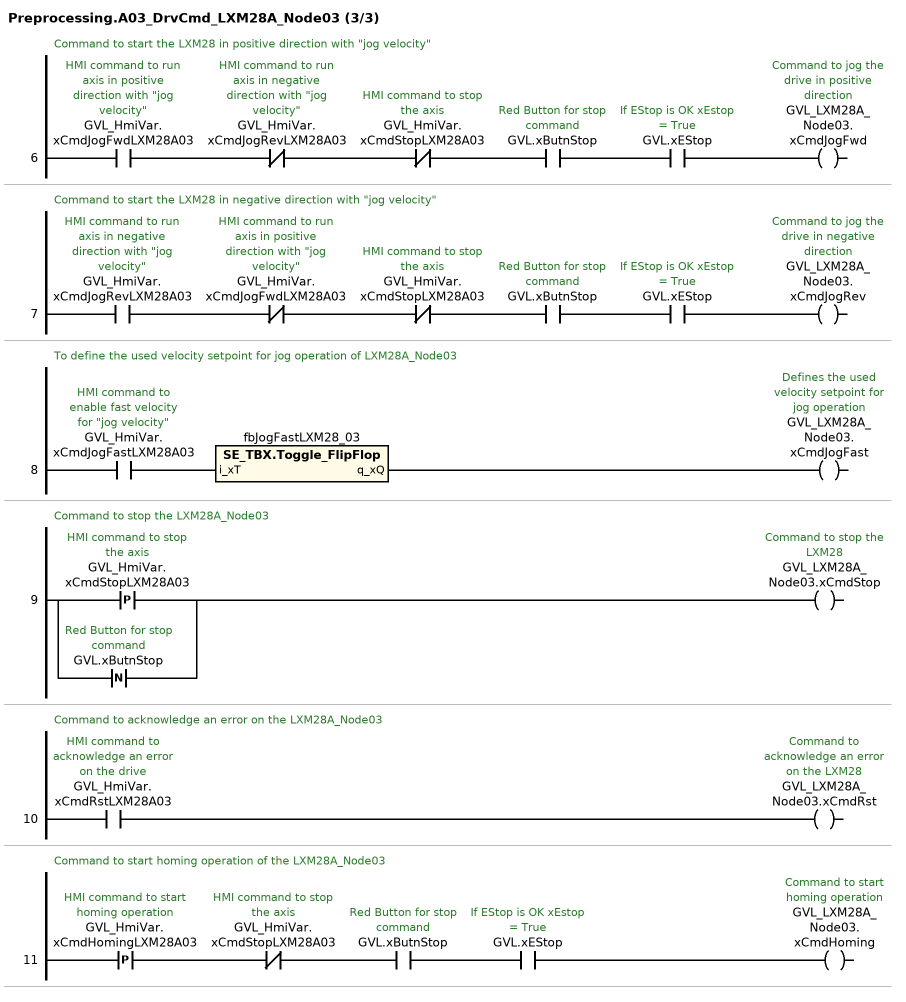
// NETWORK 6
// Command to start the LXM28 in positive direction with "jog velocity"
//   GVL_HmiVar.xCmdJogFwdLXM28A03: HMI command to run axis in positive direction with "jog velocity"
//   GVL_HmiVar.xCmdJogRevLXM28A03: HMI command to run axis in negative direction with "jog velocity"
//   GVL_HmiVar.xCmdStopLXM28A03: HMI command to stop the axis
//   GVL.xButnStop: Red Button for stop command
//   GVL.xEStop: If EStop is OK xEstop = True
//   GVL_LXM28A_Node03.xCmdJogFwd: Command to jog the drive in positive direction
GVL_LXM28A_Node03.xCmdJogFwd := GVL_HmiVar.xCmdJogFwdLXM28A03 AND NOT GVL_HmiVar.xCmdJogRevLXM28A03 AND NOT GVL_HmiVar.xCmdStopLXM28A03 AND GVL.xButnStop AND GVL.xEStop;

// NETWORK 7
// Command to start the LXM28 in negative direction with "jog velocity"
//   GVL_HmiVar.xCmdJogRevLXM28A03: HMI command to run axis in negative direction with "jog velocity"
//   GVL_HmiVar.xCmdJogFwdLXM28A03: HMI command to run axis in positive direction with "jog velocity"
//   GVL_HmiVar.xCmdStopLXM28A03: HMI command to stop the axis
//   GVL.xButnStop: Red Button for stop command
//   GVL.xEStop: If EStop is OK xEstop = True
//   GVL_LXM28A_Node03.xCmdJogRev: Command to jog the drive in negative direction
GVL_LXM28A_Node03.xCmdJogRev := GVL_HmiVar.xCmdJogRevLXM28A03 AND NOT GVL_HmiVar.xCmdJogFwdLXM28A03 AND NOT GVL_HmiVar.xCmdStopLXM28A03 AND GVL.xButnStop AND GVL.xEStop;

// NETWORK 8
// To define the used velocity setpoint for jog operation of LXM28A_Node03
//   fbJogFastLXM28_03: FB instance command JogFast
//   GVL_HmiVar.xCmdJogFastLXM28A03: HMI command to enable fast velocity for "jog velocity"
//   GVL_LXM28A_Node03.xCmdJogFast: Defines the used velocity setpoint for jog operation
fbJogFastLXM28_03(i_xT := GVL_HmiVar.xCmdJogFastLXM28A03); // SE_TBX.Toggle_FlipFlop
GVL_LXM28A_Node03.xCmdJogFast := fbJogFastLXM28_03.q_xQ;

// NETWORK 9
// Command to stop the LXM28A_Node03
//   GVL_HmiVar.xCmdStopLXM28A03: HMI command to stop the axis
//   GVL.xButnStop: Red Button for stop command
//   GVL_LXM28A_Node03.xCmdStop: Command to stop the LXM28
_rt38(CLK := GVL_HmiVar.xCmdStopLXM28A03);
_ft3(CLK := GVL.xButnStop);
GVL_LXM28A_Node03.xCmdStop := _rt38.Q OR _ft3.Q;

// NETWORK 10
// Command to acknowledge an error on the LXM28A_Node03
//   GVL_HmiVar.xCmdRstLXM28A03: HMI command to acknowledge an error on the drive
//   GVL_LXM28A_Node03.xCmdRst: Command to acknowledge an error on the LXM28
GVL_LXM28A_Node03.xCmdRst := GVL_HmiVar.xCmdRstLXM28A03;

// NETWORK 11
// Command to start homing operation of the LXM28A_Node03
//   GVL_HmiVar.xCmdHomingLXM28A03: HMI command to start homing operation
//   GVL_HmiVar.xCmdStopLXM28A03: HMI command to stop the axis
//   GVL.xButnStop: Red Button for stop command
//   GVL.xEStop: If EStop is OK xEstop = True
//   GVL_LXM28A_Node03.xCmdHoming: Command to start homing operation
_rt39(CLK := GVL_HmiVar.xCmdHomingLXM28A03);
GVL_LXM28A_Node03.xCmdHoming := _rt39.Q AND NOT GVL_HmiVar.xCmdStopLXM28A03 AND GVL.xButnStop AND GVL.xEStop;
END_ACTION

END_PROGRAM

// HMISAC/Application/Joystick_SD6000/Prg_Joystick6000
PROGRAM Prg_Joystick6000
VAR
	fbGetNodeStat     : CIA405.GET_STATE; // FB instance to get the state of the CANopen node
END_VAR
VAR CONSTANT
	c_udiTmotGetStat : UDINT := 4000; // Parameter timeout for FB GET_STATE in ms
	c_NodeID         : USINT := 2;
	c_Network        : USINT := 1; 
END_VAR
VAR // added by the converter: edge detectors and wires of the graphical bodies
    _w1, _w3 : ANY;
    _w2 : BOOL;
END_VAR

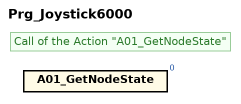
// Call of the Action "A01_GetNodeState"
A01_GetNodeState();

ACTION A01_GetNodeState:
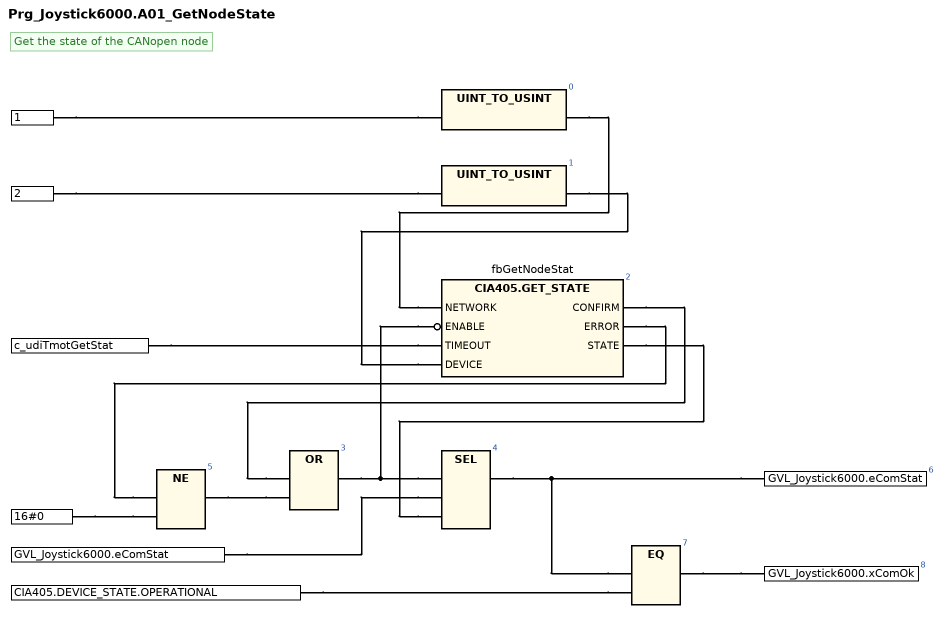
// Get the state of the CANopen node
fbGetNodeStat(
    NETWORK := UINT_TO_USINT(1),
    ENABLE := NOT _w1,
    TIMEOUT := c_udiTmotGetStat,
    DEVICE := UINT_TO_USINT(2)); // CIA405.GET_STATE
_w1 := fbGetNodeStat.CONFIRM OR _w2;
_w3 := SEL(_w1, GVL_Joystick6000.eComStat, fbGetNodeStat.STATE);
_w2 := fbGetNodeStat.ERROR <> 16#0;
GVL_Joystick6000.eComStat := _w3;
GVL_Joystick6000.xComOk := _w3 = CIA405.DEVICE_STATE.OPERATIONAL;
END_ACTION

END_PROGRAM

// HMISAC/Application/MicroCAN4aiBOX/Prg_MicroCAN
PROGRAM Prg_MicroCAN
VAR
	fbGetNodeStat     : CIA405.GET_STATE; // FB instance to get the state of the CANopen node
	END_VAR
VAR CONSTANT
	c_udiTmotGetStat : UDINT := 4000; // Parameter timeout for FB GET_STATE in ms
	c_NodeID         : USINT := 16;
	c_Network        : USINT := 1; 
END_VAR
VAR // added by the converter: edge detectors and wires of the graphical bodies
    _w1, _w3 : ANY;
    _w2 : BOOL;
END_VAR

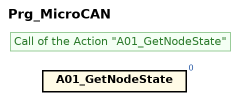
// Call of the Action "A01_GetNodeState"
A01_GetNodeState();

ACTION A01_GetNodeState:
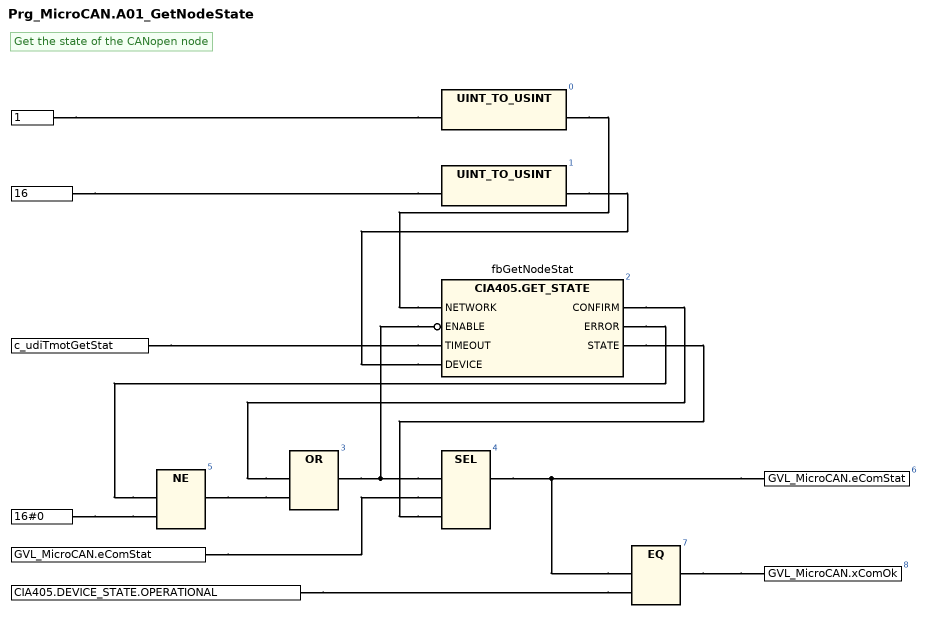
// Get the state of the CANopen node
fbGetNodeStat(
    NETWORK := UINT_TO_USINT(1),
    ENABLE := NOT _w1,
    TIMEOUT := c_udiTmotGetStat,
    DEVICE := UINT_TO_USINT(16)); // CIA405.GET_STATE
_w1 := fbGetNodeStat.CONFIRM OR _w2;
_w3 := SEL(_w1, GVL_MicroCAN.eComStat, fbGetNodeStat.STATE);
_w2 := fbGetNodeStat.ERROR <> 16#0;
GVL_MicroCAN.eComStat := _w3;
GVL_MicroCAN.xComOk := _w3 = CIA405.DEVICE_STATE.OPERATIONAL;
END_ACTION

END_PROGRAM

// HMISAC/Application/Dunker_0A/Prg_Dunker_0A
PROGRAM Prg_Dunker_0A
VAR
		fbGetNodeStat     : CIA405.GET_STATE;                   // FB instance to get the state of the CANopen node
	// FB instance to power the Dunkermotoren
 
	fbPwr_DK		  : MC_Power;
	Axis_Dunker_0A    : AXIS_REF_SM3;
 
END_VAR
VAR CONSTANT
	c_udiTmotGetStat : UDINT := 4000; // Parameter timeout for FB GET_STATE in ms
	c_NodeID         : USINT := 10;
	c_Network        : USINT := 1; 
END_VAR
VAR // added by the converter: edge detectors and wires of the graphical bodies
    _w1, _w3 : ANY;
    _w2 : BOOL;
END_VAR

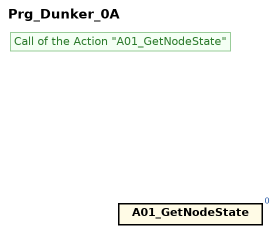
// Call of the Action "A01_GetNodeState"
A01_GetNodeState();

ACTION A01_GetNodeState:
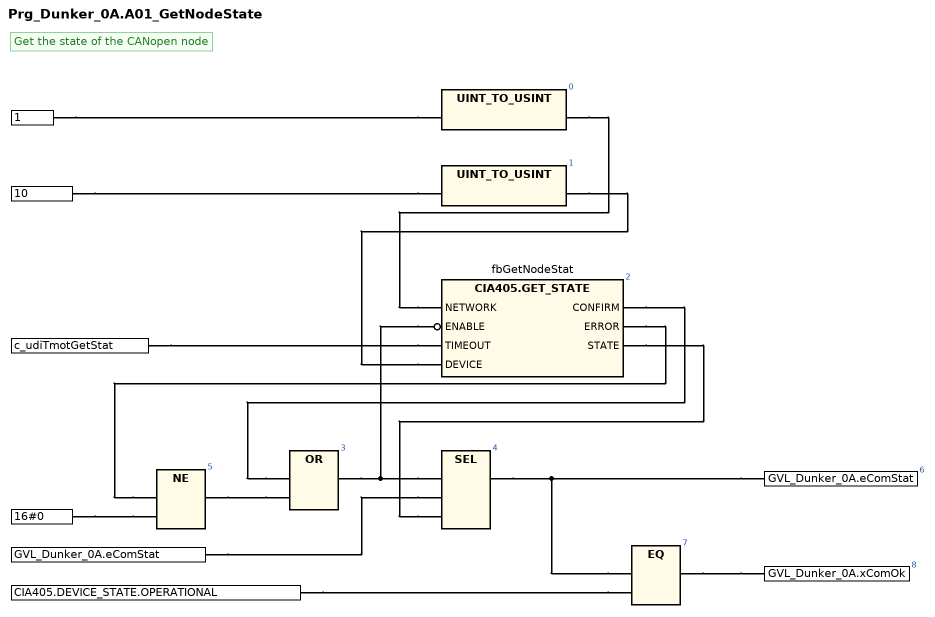
// Get the state of the CANopen node
fbGetNodeStat(
    NETWORK := UINT_TO_USINT(1),
    ENABLE := NOT _w1,
    TIMEOUT := c_udiTmotGetStat,
    DEVICE := UINT_TO_USINT(10)); // CIA405.GET_STATE
_w1 := fbGetNodeStat.CONFIRM OR _w2;
_w3 := SEL(_w1, GVL_Dunker_0A.eComStat, fbGetNodeStat.STATE);
_w2 := fbGetNodeStat.ERROR <> 16#0;
GVL_Dunker_0A.eComStat := _w3;
GVL_Dunker_0A.xComOk := _w3 = CIA405.DEVICE_STATE.OPERATIONAL;
END_ACTION

ACTION A02_Ctrl_Dunker_0A:
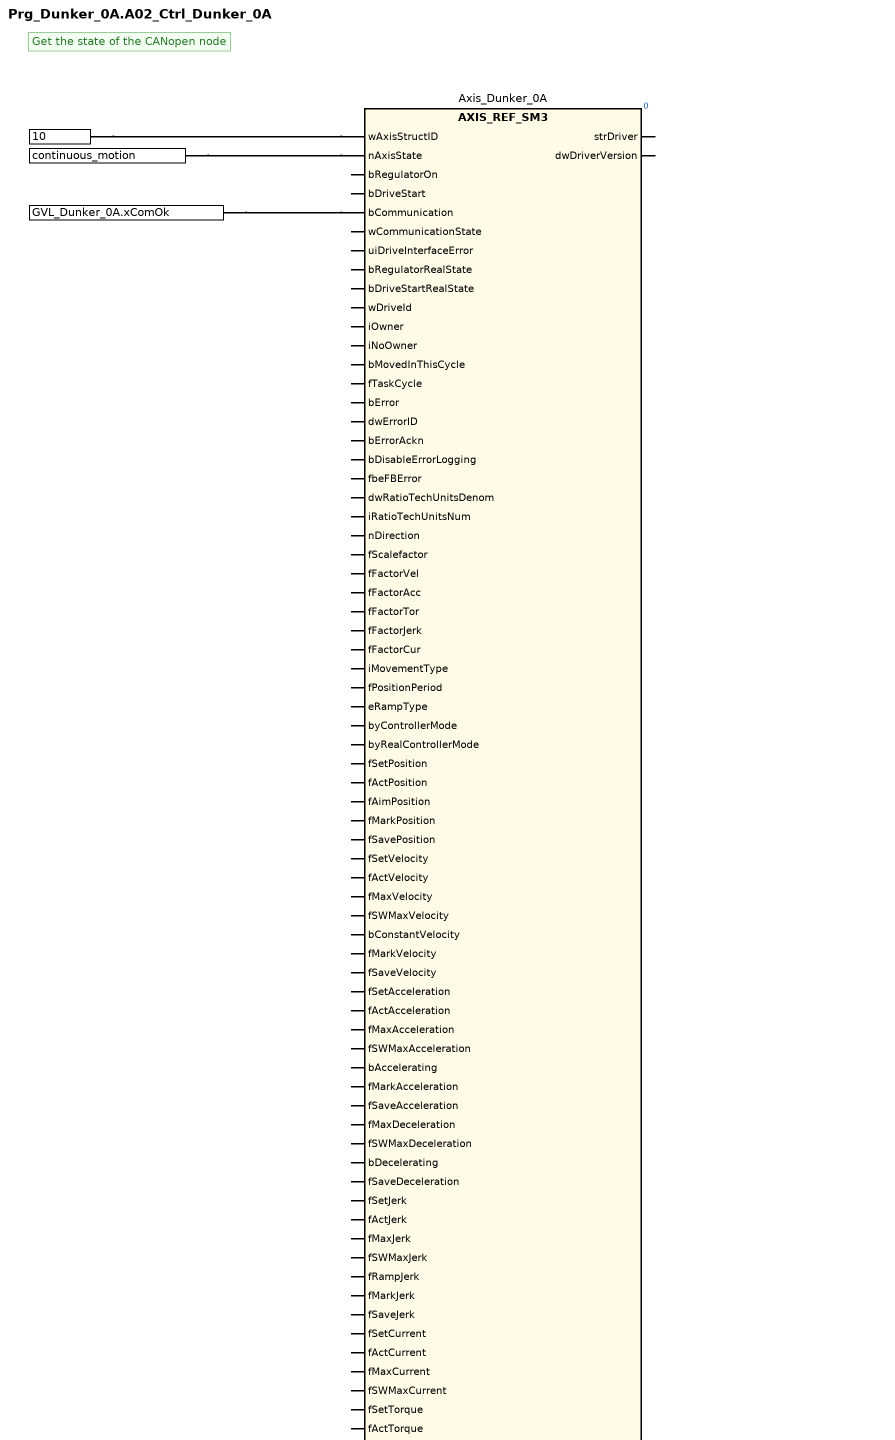
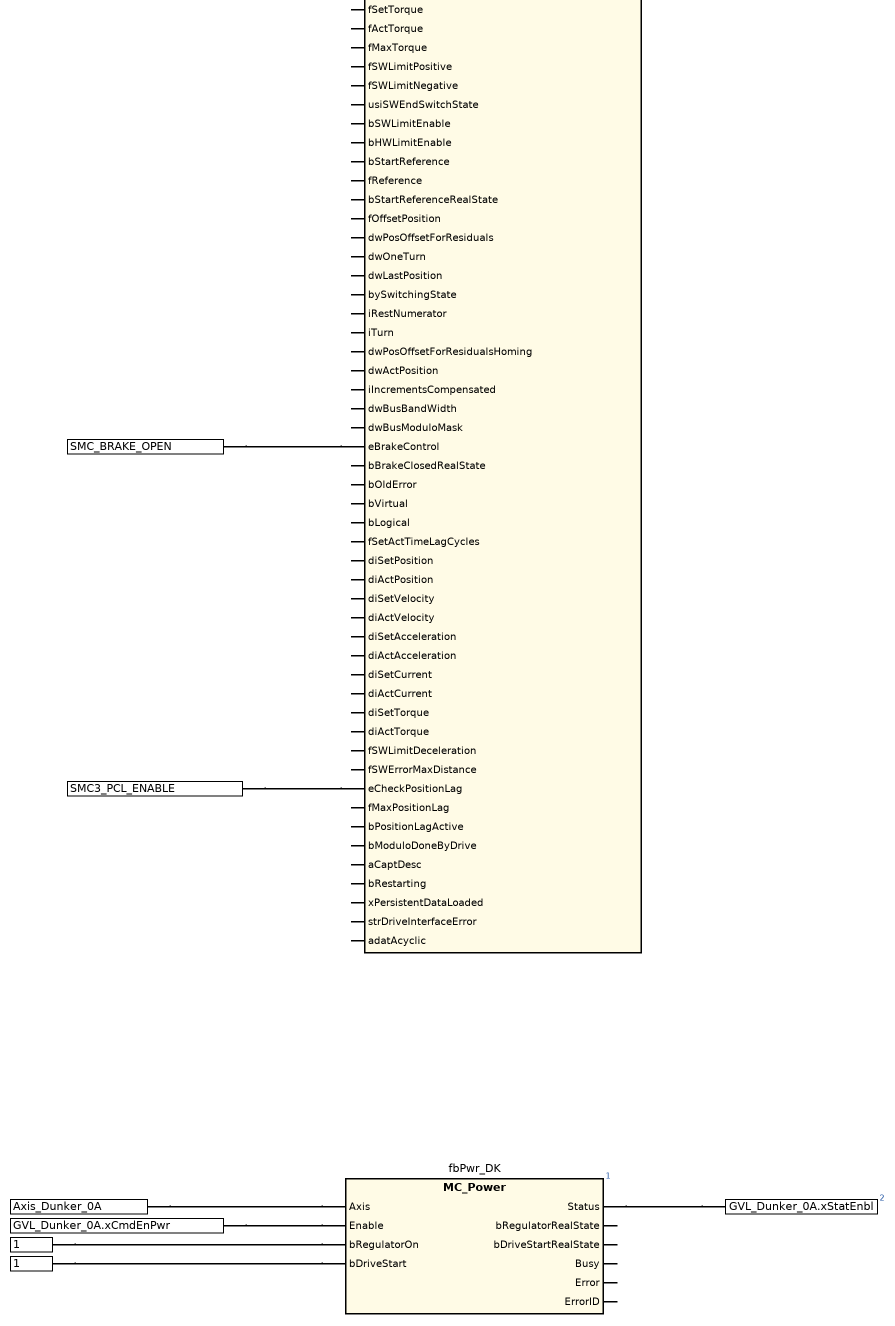
// Get the state of the CANopen node
Axis_Dunker_0A(
    wAxisStructID := 10,
    nAxisState := continuous_motion,
    bCommunication := GVL_Dunker_0A.xComOk,
    eBrakeControl := SMC_BRAKE_OPEN,
    eCheckPositionLag := SMC3_PCL_ENABLE); // AXIS_REF_SM3
fbPwr_DK(Axis := Axis_Dunker_0A, Enable := GVL_Dunker_0A.xCmdEnPwr, bRegulatorOn := 1, bDriveStart := 1); // MC_Power
GVL_Dunker_0A.xStatEnbl := fbPwr_DK.Status;
END_ACTION

END_PROGRAM

// HMISAC/Application/Dunker_0B/Prg_Dunker_0B
PROGRAM Prg_Dunker_0B
VAR
	fbGetNodeStat     : CIA405.GET_STATE; // FB instance to get the state of the CANopen node
END_VAR
VAR CONSTANT
	c_udiTmotGetStat : UDINT := 4000; // Parameter timeout for FB GET_STATE in ms
	c_NodeID         : USINT := 11;
	c_Network        : USINT := 1; 
END_VAR
VAR // added by the converter: edge detectors and wires of the graphical bodies
    _w1, _w3 : ANY;
    _w2 : BOOL;
END_VAR

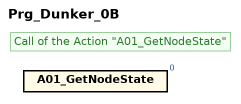
// Call of the Action "A01_GetNodeState"
A01_GetNodeState();

ACTION A01_GetNodeState:
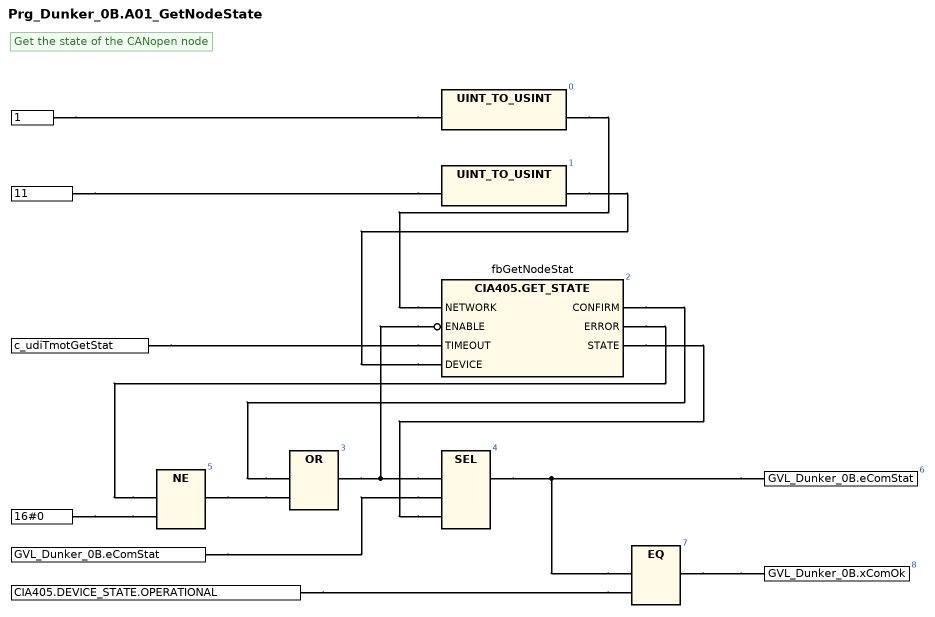
// Get the state of the CANopen node
fbGetNodeStat(
    NETWORK := UINT_TO_USINT(1),
    ENABLE := NOT _w1,
    TIMEOUT := c_udiTmotGetStat,
    DEVICE := UINT_TO_USINT(11)); // CIA405.GET_STATE
_w1 := fbGetNodeStat.CONFIRM OR _w2;
_w3 := SEL(_w1, GVL_Dunker_0B.eComStat, fbGetNodeStat.STATE);
_w2 := fbGetNodeStat.ERROR <> 16#0;
GVL_Dunker_0B.eComStat := _w3;
GVL_Dunker_0B.xComOk := _w3 = CIA405.DEVICE_STATE.OPERATIONAL;
END_ACTION

END_PROGRAM

// HMISAC/Application/Dunker_0C/Prg_Dunker_0C
PROGRAM Prg_Dunker_0C
VAR
	fbGetNodeStat     : CIA405.GET_STATE; // FB instance to get the state of the CANopen node
END_VAR
VAR CONSTANT
	c_udiTmotGetStat : UDINT := 4000; // Parameter timeout for FB GET_STATE in ms
	c_NodeID         : USINT := 12;
	c_Network        : USINT := 1; 
END_VAR
VAR // added by the converter: edge detectors and wires of the graphical bodies
    _w1, _w3 : ANY;
    _w2 : BOOL;
END_VAR

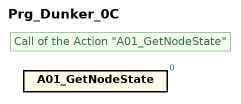
// Call of the Action "A01_GetNodeState"
A01_GetNodeState();

ACTION A01_getNodeState:
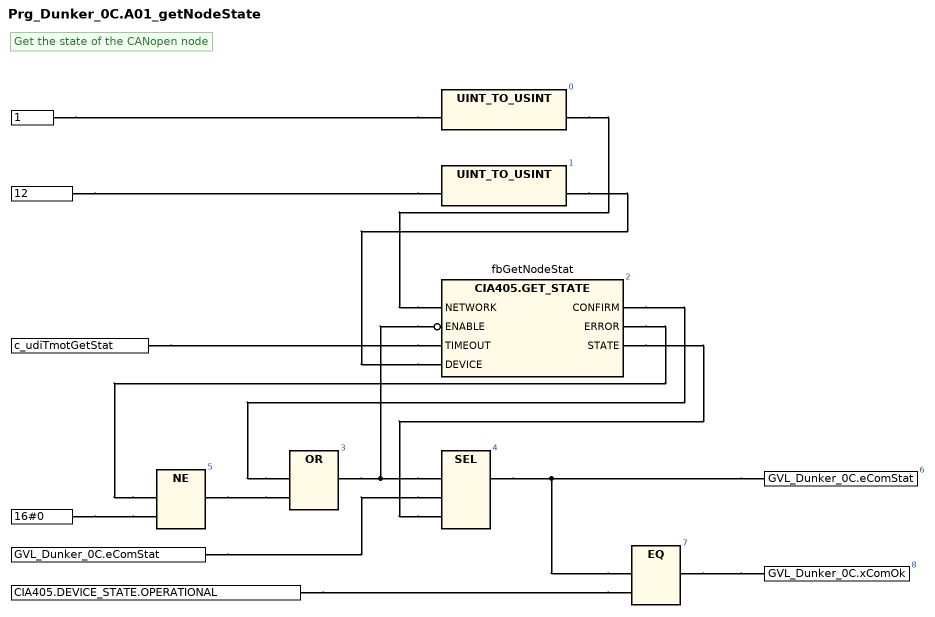
// Get the state of the CANopen node
fbGetNodeStat(
    NETWORK := UINT_TO_USINT(1),
    ENABLE := NOT _w1,
    TIMEOUT := c_udiTmotGetStat,
    DEVICE := UINT_TO_USINT(12)); // CIA405.GET_STATE
_w1 := fbGetNodeStat.CONFIRM OR _w2;
_w3 := SEL(_w1, GVL_Dunker_0C.eComStat, fbGetNodeStat.STATE);
_w2 := fbGetNodeStat.ERROR <> 16#0;
GVL_Dunker_0C.eComStat := _w3;
GVL_Dunker_0C.xComOk := _w3 = CIA405.DEVICE_STATE.OPERATIONAL;
END_ACTION

END_PROGRAM

// HMISAC/Application/Dunker_0D/Prg_Dunker_0D
PROGRAM Prg_Dunker_0D
VAR
	fbGetNodeStat     : CIA405.GET_STATE; // FB instance to get the state of the CANopen node
END_VAR
VAR CONSTANT
	c_udiTmotGetStat : UDINT := 4000; // Parameter timeout for FB GET_STATE in ms
	c_NodeID         : USINT := 13;
	c_Network        : USINT := 1; 
END_VAR
VAR // added by the converter: edge detectors and wires of the graphical bodies
    _w1, _w3 : ANY;
    _w2 : BOOL;
END_VAR

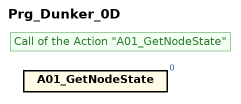
// Call of the Action "A01_GetNodeState"
A01_GetNodeState();

ACTION A01_GetNodeState:
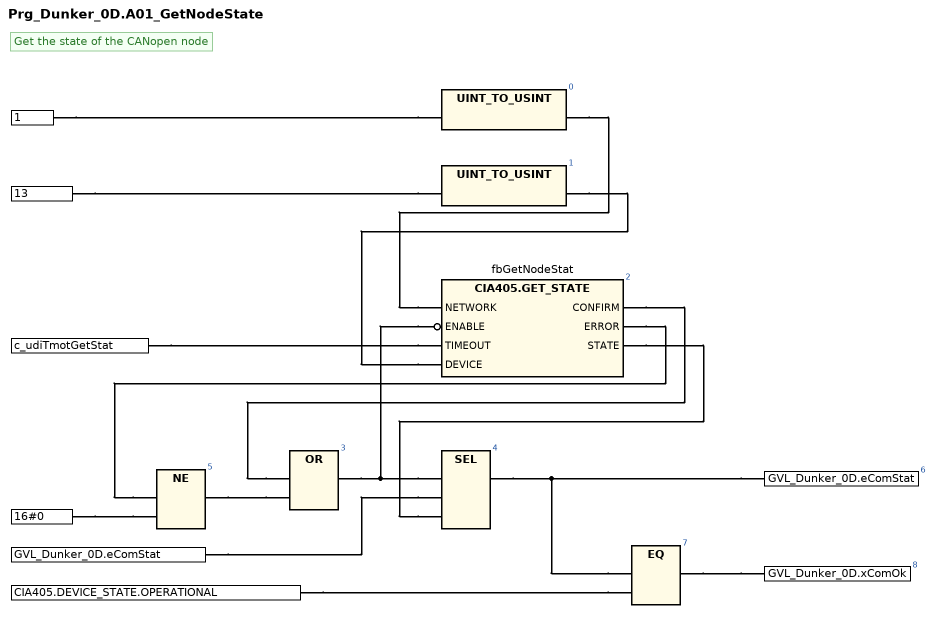
// Get the state of the CANopen node
fbGetNodeStat(
    NETWORK := UINT_TO_USINT(1),
    ENABLE := NOT _w1,
    TIMEOUT := c_udiTmotGetStat,
    DEVICE := UINT_TO_USINT(13)); // CIA405.GET_STATE
_w1 := fbGetNodeStat.CONFIRM OR _w2;
_w3 := SEL(_w1, GVL_Dunker_0D.eComStat, fbGetNodeStat.STATE);
_w2 := fbGetNodeStat.ERROR <> 16#0;
GVL_Dunker_0D.eComStat := _w3;
GVL_Dunker_0D.xComOk := _w3 = CIA405.DEVICE_STATE.OPERATIONAL;
END_ACTION

END_PROGRAM

// HMISAC/Application/Speedgoat/Prg_Speedgoat
PROGRAM Prg_Speedgoat
VAR
	fbGetNodeStat     : CIA405.GET_STATE; // FB instance to get the state of the CANopen node
END_VAR
VAR CONSTANT
	c_udiTmotGetStat : UDINT := 4000; // Parameter timeout for FB GET_STATE in ms
	c_NodeID         : USINT := 5;
	c_Network        : USINT := 1; 
END_VAR
VAR // added by the converter: edge detectors and wires of the graphical bodies
    _w1, _w3 : ANY;
    _w2 : BOOL;
END_VAR

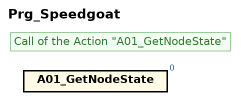
// Call of the Action "A01_GetNodeState"
A01_GetNodeState();

ACTION A01_GetNodeState:
